// TIA Portal V17 export
// export: Created 2025-07-01T14:26:10.6416357Z, ExportSetting WithDefaults, DisplayName Totally Integrated Automation Portal, DisplayVersion V17 Update 8, DisplayName TIA Portal Openness, DisplayVersion V17 Update 8, DisplayName TIA Portal Version Control Interface, DisplayVersion V17, DisplayName SINAMICS Startdrive Advanced, DisplayVersion V17 SP2, DisplayName SINAMICS Startdrive G110M, G120, G120C, G120D, G120P, G115D, DisplayVersion V17 SP2, DisplayName SINAMICS Startdrive G130, G150, S120, S150, SINAMICS MV, S210, DisplayVersion V17 SP2, DisplayName STEP 7 Professional, DisplayVersion V17 Update 8, DisplayName SINUMERIK ONE STEP 7 Toolbox, DisplayVersion V17 Update 12, DisplayName SINUMERIK ONE PLC Basic Program Plus, DisplayVersion V17 Update 12, DisplayName SINUMERIK 840D sl STEP 7 Toolbox, DisplayVersion V17 Update 12, DisplayName STEP 7 Safety, DisplayVersion V17 Update 6, DisplayName WinCC Advanced, DisplayVersion V17 Update 8
FUNCTION "FC16016_METHOD_CALLS_U3_MEAS_STA_MEAS_R" : Void   // FC16016, LAD
{ S7_Optimized_Access := 'FALSE' }
VERSION : 0.1
// STATUS VALUES:
// 0 = IDLE
// 1 = ANALYZING
// 2 = CALIBRATING
// -1 = ERROR
// stored: AutoNumber false, IsIECCheckEnabled false, SetENOAutomatically false, UDAEnableTagReadback false
   VAR_TEMP
      AUX_WSTRING_PART_ID_MEAS_STA : WString;
      AUX_WCHARS : Array[0..63] of WChar;
      index : Int;
      AUX_ALARMS : Bool;
      STATUS_BLKMOV : Int;   // STATUS BLKMOV
      ZERO : Int;
   END_VAR
   VAR CONSTANT
      VERSIONS_MAJOR : UInt := 2;
      VERSIONS_MINOR : UInt;
      FC_NUMBER : DInt := 16016;
   END_VAR
   VAR_TEMP   // added for the SCL form of the ladder/FBD networks
      _w1 : Bool;
      _w2 : Bool;
      _w3 : Bool;
   END_VAR
BEGIN

REGION Network 1: ZERO
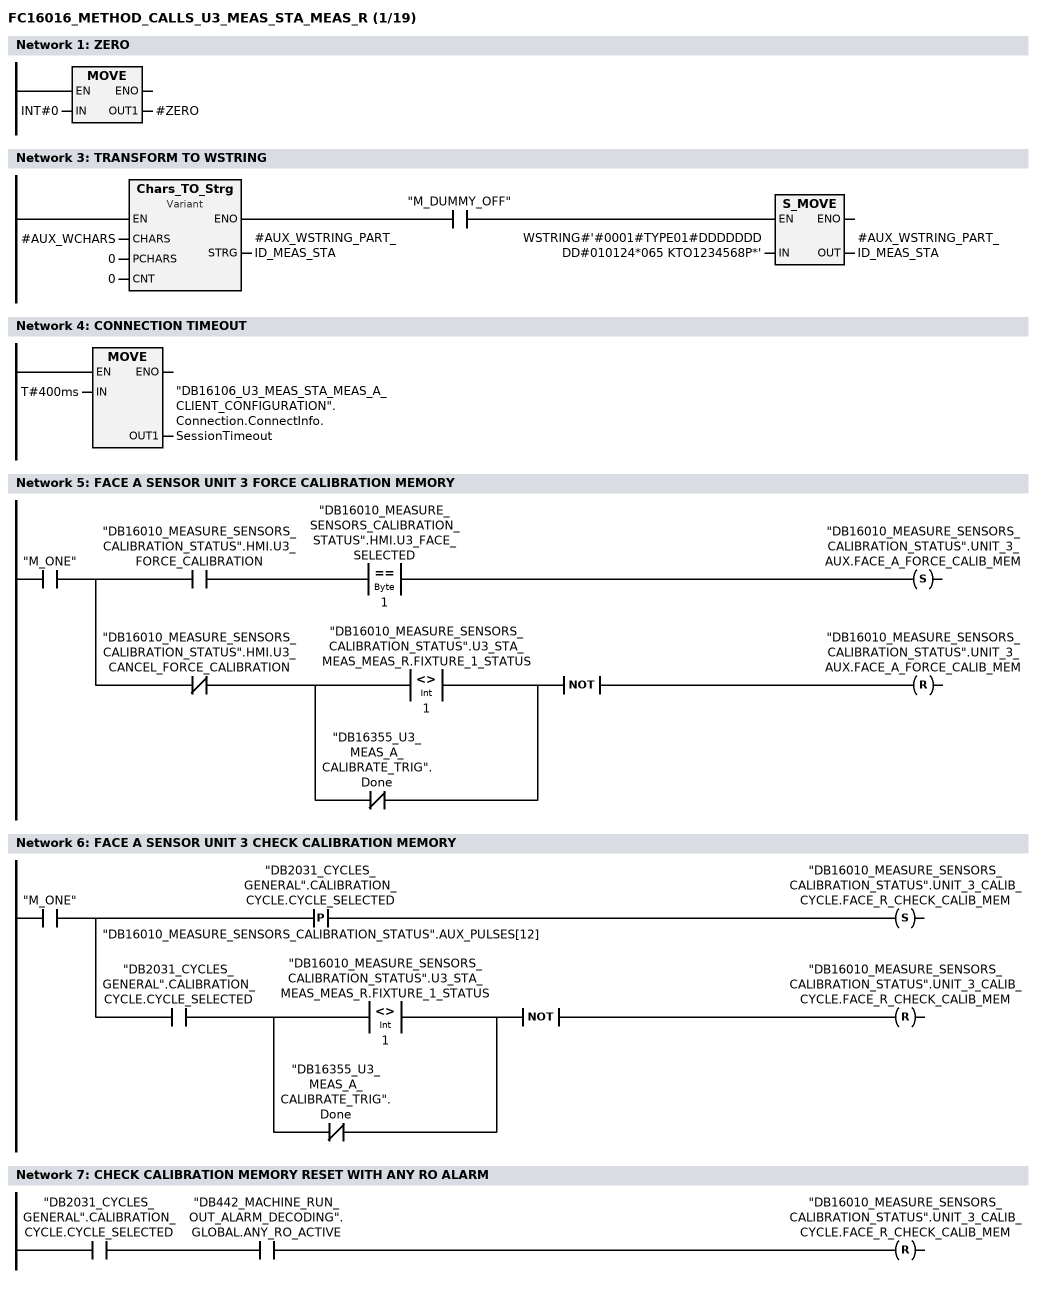
   RUNG wire#powerrail
      { S7_GenerateENO := "TRUE" } Move(in := INT#0, out1 => #ZERO)
   END_RUNG
   // the same network as SCL:
   #ZERO := INT#0;
END_REGION

REGION Network 2 (SCL): TRANSFORM TO WCHARS
   FOR #index := 0 TO 63 DO
       #AUX_WCHARS[#index] := CHAR_TO_WCHAR("DB8000_PART_STATUS".UNIT_3.FIXTURE_1.PART_A.PART_ID[#index]);
   END_FOR;
END_REGION

REGION Network 3: TRANSFORM TO WSTRING
   RUNG wire#powerrail
      { S7_Templates := "[ptr_type := Variant, str_type := WString]" } Chars_TO_Strg(Chars := #AUX_WCHARS, pChars := 0, Cnt := 0, Strg => #AUX_WSTRING_PART_ID_MEAS_STA)
      Contact( "M_DUMMY_OFF" )
      S_Move(in := WSTRING#'#0001#TYPE01#DDDDDDDDD#010124*065 KTO1234568P*', out => #AUX_WSTRING_PART_ID_MEAS_STA)
   END_RUNG
   // the same network as SCL:
   Chars_TO_Strg(Chars := #AUX_WCHARS,
                 pChars := 0,
                 Cnt := 0,
                 Strg => #AUX_WSTRING_PART_ID_MEAS_STA,
                 ENO => #_w1);
   IF #_w1 AND "M_DUMMY_OFF" THEN
       #AUX_WSTRING_PART_ID_MEAS_STA := WSTRING#'#0001#TYPE01#DDDDDDDDD#010124*065 KTO1234568P*';
   END_IF;
END_REGION

REGION Network 4: CONNECTION TIMEOUT
   RUNG wire#powerrail
      Move(in := T#400ms, out1 => "DB16106_U3_MEAS_STA_MEAS_A_CLIENT_CONFIGURATION".Connection.ConnectInfo.SessionTimeout)
   END_RUNG
   // the same network as SCL:
   "DB16106_U3_MEAS_STA_MEAS_A_CLIENT_CONFIGURATION".Connection.ConnectInfo.SessionTimeout := T#400ms;
END_REGION

REGION Network 5: FACE A SENSOR UNIT 3 FORCE CALIBRATION MEMORY
   RUNG wire#powerrail
      Contact( "M_ONE" )
      wire#w1
      Contact( "DB16010_MEASURE_SENSORS_CALIBRATION_STATUS".HMI.U3_FORCE_CALIBRATION )
      { S7_Templates := "SrcType := Byte" } EQ_Contact(in1 := "DB16010_MEASURE_SENSORS_CALIBRATION_STATUS".HMI.U3_FACE_SELECTED, in2 := 1)
      S_Coil( "DB16010_MEASURE_SENSORS_CALIBRATION_STATUS".UNIT_3_AUX.FACE_A_FORCE_CALIB_MEM )
   END_RUNG
   RUNG wire#w1
      I_Contact( "DB16010_MEASURE_SENSORS_CALIBRATION_STATUS".HMI.U3_CANCEL_FORCE_CALIBRATION )
      wire#w2
      { S7_Templates := "SrcType := Int" } NE_Contact(in1 := "DB16010_MEASURE_SENSORS_CALIBRATION_STATUS".U3_STA_MEAS_MEAS_R.FIXTURE_1_STATUS, in2 := 1)
      wire#w3
      Not()
      R_Coil( "DB16010_MEASURE_SENSORS_CALIBRATION_STATUS".UNIT_3_AUX.FACE_A_FORCE_CALIB_MEM )
   END_RUNG
   RUNG wire#w2
      I_Contact( "DB16355_U3_MEAS_A_CALIBRATE_TRIG".Done )
   END_RUNG wire#w3
   // the same network as SCL:
   IF "M_ONE" AND "DB16010_MEASURE_SENSORS_CALIBRATION_STATUS".HMI.U3_FORCE_CALIBRATION AND ("DB16010_MEASURE_SENSORS_CALIBRATION_STATUS".HMI.U3_FACE_SELECTED = 1) THEN
       "DB16010_MEASURE_SENSORS_CALIBRATION_STATUS".UNIT_3_AUX.FACE_A_FORCE_CALIB_MEM := TRUE;
   END_IF;
   IF NOT ("M_ONE" AND NOT "DB16010_MEASURE_SENSORS_CALIBRATION_STATUS".HMI.U3_CANCEL_FORCE_CALIBRATION AND (("DB16010_MEASURE_SENSORS_CALIBRATION_STATUS".U3_STA_MEAS_MEAS_R.FIXTURE_1_STATUS <> 1) OR NOT "DB16355_U3_MEAS_A_CALIBRATE_TRIG".Done)) THEN
       "DB16010_MEASURE_SENSORS_CALIBRATION_STATUS".UNIT_3_AUX.FACE_A_FORCE_CALIB_MEM := FALSE;
   END_IF;
END_REGION

REGION Network 6: FACE A SENSOR UNIT 3 CHECK CALIBRATION MEMORY
   RUNG wire#powerrail
      Contact( "M_ONE" )
      wire#w1
      P_Contact(operand := "DB2031_CYCLES_GENERAL".CALIBRATION_CYCLE.CYCLE_SELECTED, bit := "DB16010_MEASURE_SENSORS_CALIBRATION_STATUS".AUX_PULSES[12])
      S_Coil( "DB16010_MEASURE_SENSORS_CALIBRATION_STATUS".UNIT_3_CALIB_CYCLE.FACE_R_CHECK_CALIB_MEM )
   END_RUNG
   RUNG wire#w1
      Contact( "DB2031_CYCLES_GENERAL".CALIBRATION_CYCLE.CYCLE_SELECTED )
      wire#w2
      { S7_Templates := "SrcType := Int" } NE_Contact(in1 := "DB16010_MEASURE_SENSORS_CALIBRATION_STATUS".U3_STA_MEAS_MEAS_R.FIXTURE_1_STATUS, in2 := 1)
      wire#w3
      Not()
      R_Coil( "DB16010_MEASURE_SENSORS_CALIBRATION_STATUS".UNIT_3_CALIB_CYCLE.FACE_R_CHECK_CALIB_MEM )
   END_RUNG
   RUNG wire#w2
      I_Contact( "DB16355_U3_MEAS_A_CALIBRATE_TRIG".Done )
   END_RUNG wire#w3
   // the same network as SCL:
   #_w1 := "M_ONE" AND "DB2031_CYCLES_GENERAL".CALIBRATION_CYCLE.CYCLE_SELECTED AND NOT "DB16010_MEASURE_SENSORS_CALIBRATION_STATUS".AUX_PULSES[12];   // rising edge of "DB2031_CYCLES_GENERAL".CALIBRATION_CYCLE.CYCLE_SELECTED
   "DB16010_MEASURE_SENSORS_CALIBRATION_STATUS".AUX_PULSES[12] := "DB2031_CYCLES_GENERAL".CALIBRATION_CYCLE.CYCLE_SELECTED;
   IF #_w1 THEN
       "DB16010_MEASURE_SENSORS_CALIBRATION_STATUS".UNIT_3_CALIB_CYCLE.FACE_R_CHECK_CALIB_MEM := TRUE;
   END_IF;
   IF NOT ("M_ONE" AND "DB2031_CYCLES_GENERAL".CALIBRATION_CYCLE.CYCLE_SELECTED AND (("DB16010_MEASURE_SENSORS_CALIBRATION_STATUS".U3_STA_MEAS_MEAS_R.FIXTURE_1_STATUS <> 1) OR NOT "DB16355_U3_MEAS_A_CALIBRATE_TRIG".Done)) THEN
       "DB16010_MEASURE_SENSORS_CALIBRATION_STATUS".UNIT_3_CALIB_CYCLE.FACE_R_CHECK_CALIB_MEM := FALSE;
   END_IF;
END_REGION

REGION Network 7: CHECK CALIBRATION MEMORY RESET WITH ANY RO ALARM
   RUNG wire#powerrail
      Contact( "DB2031_CYCLES_GENERAL".CALIBRATION_CYCLE.CYCLE_SELECTED )
      Contact( "DB442_MACHINE_RUN_OUT_ALARM_DECODING".GLOBAL.ANY_RO_ACTIVE )
      R_Coil( "DB16010_MEASURE_SENSORS_CALIBRATION_STATUS".UNIT_3_CALIB_CYCLE.FACE_R_CHECK_CALIB_MEM )
   END_RUNG
   // the same network as SCL:
   IF "DB2031_CYCLES_GENERAL".CALIBRATION_CYCLE.CYCLE_SELECTED AND "DB442_MACHINE_RUN_OUT_ALARM_DECODING".GLOBAL.ANY_RO_ACTIVE THEN
       "DB16010_MEASURE_SENSORS_CALIBRATION_STATUS".UNIT_3_CALIB_CYCLE.FACE_R_CHECK_CALIB_MEM := FALSE;
   END_IF;
END_REGION

REGION Network 8: UNIT 3 MEASURING START CONNECTION TRIGGER
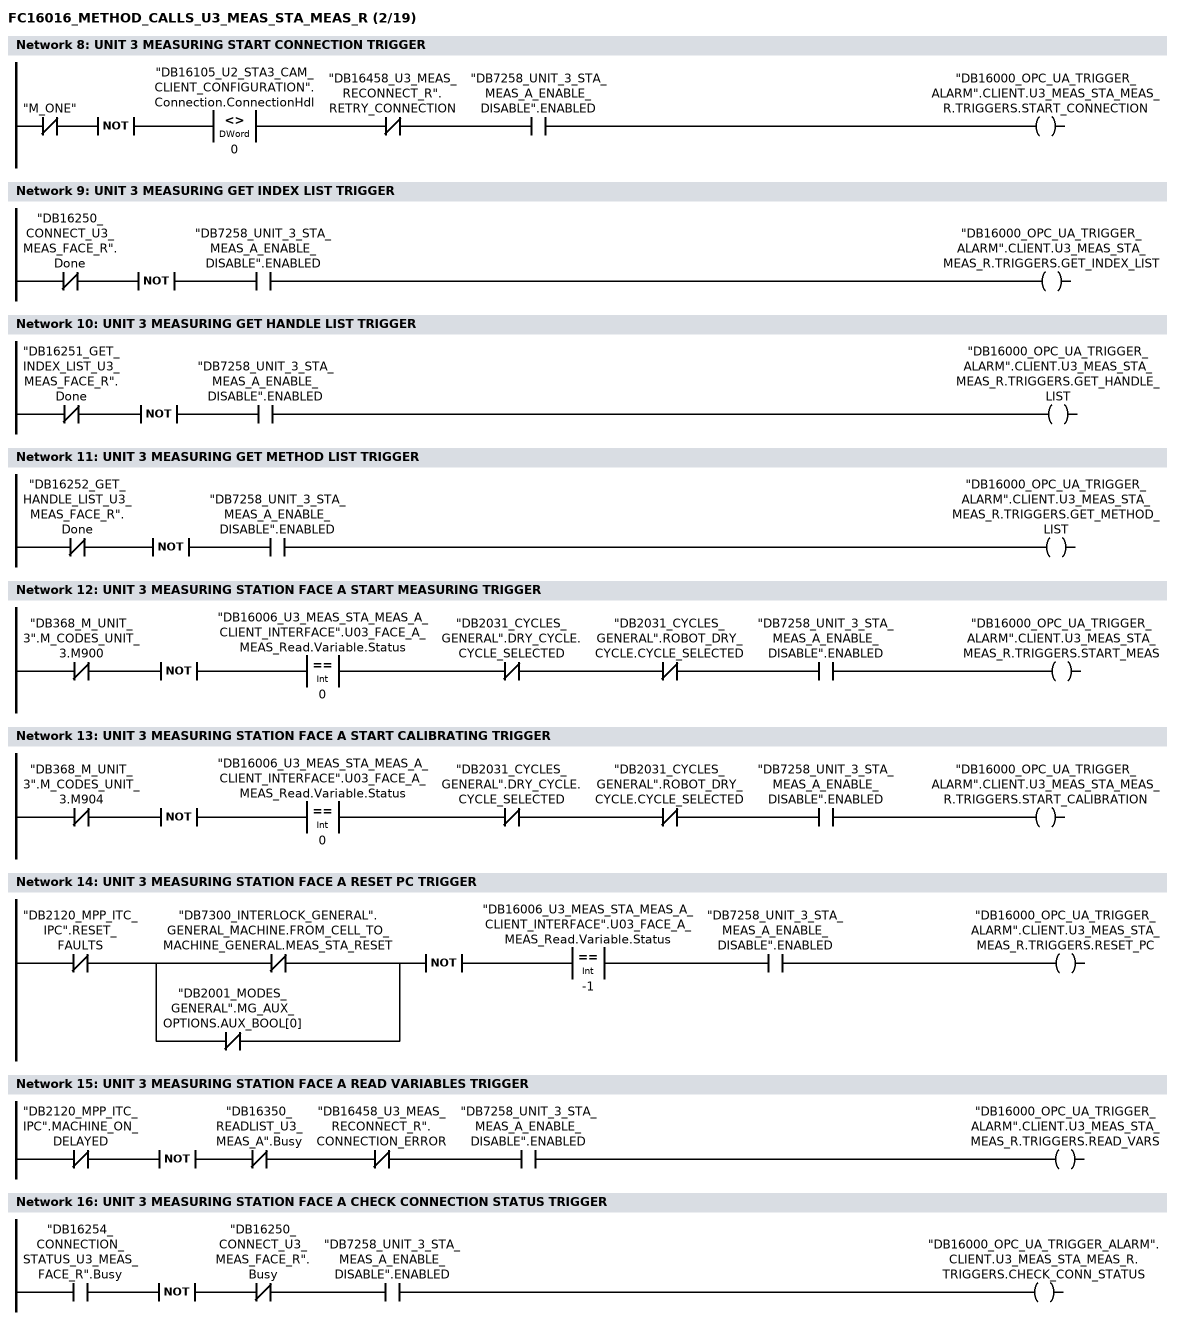
   RUNG wire#powerrail
      I_Contact( "M_ONE" )
      Not()
      { S7_Templates := "SrcType := DWord" } NE_Contact(in1 := "DB16105_U2_STA3_CAM_CLIENT_CONFIGURATION".Connection.ConnectionHdl, in2 := 0)
      I_Contact( "DB16458_U3_MEAS_RECONNECT_R".RETRY_CONNECTION )
      Contact( "DB7258_UNIT_3_STA_MEAS_A_ENABLE_DISABLE".ENABLED )
      Coil( "DB16000_OPC_UA_TRIGGER_ALARM".CLIENT.U3_MEAS_STA_MEAS_R.TRIGGERS.START_CONNECTION )
   END_RUNG
   // the same network as SCL:
   "DB16000_OPC_UA_TRIGGER_ALARM".CLIENT.U3_MEAS_STA_MEAS_R.TRIGGERS.START_CONNECTION := NOT (NOT "M_ONE") AND ("DB16105_U2_STA3_CAM_CLIENT_CONFIGURATION".Connection.ConnectionHdl <> 0) AND NOT "DB16458_U3_MEAS_RECONNECT_R".RETRY_CONNECTION AND "DB7258_UNIT_3_STA_MEAS_A_ENABLE_DISABLE".ENABLED;
END_REGION

REGION Network 9: UNIT 3 MEASURING GET INDEX LIST TRIGGER
   RUNG wire#powerrail
      I_Contact( "DB16250_CONNECT_U3_MEAS_FACE_R".Done )
      Not()
      Contact( "DB7258_UNIT_3_STA_MEAS_A_ENABLE_DISABLE".ENABLED )
      Coil( "DB16000_OPC_UA_TRIGGER_ALARM".CLIENT.U3_MEAS_STA_MEAS_R.TRIGGERS.GET_INDEX_LIST )
   END_RUNG
   // the same network as SCL:
   "DB16000_OPC_UA_TRIGGER_ALARM".CLIENT.U3_MEAS_STA_MEAS_R.TRIGGERS.GET_INDEX_LIST := NOT (NOT "DB16250_CONNECT_U3_MEAS_FACE_R".Done) AND "DB7258_UNIT_3_STA_MEAS_A_ENABLE_DISABLE".ENABLED;
END_REGION

REGION Network 10: UNIT 3 MEASURING GET HANDLE LIST TRIGGER
   RUNG wire#powerrail
      I_Contact( "DB16251_GET_INDEX_LIST_U3_MEAS_FACE_R".Done )
      Not()
      Contact( "DB7258_UNIT_3_STA_MEAS_A_ENABLE_DISABLE".ENABLED )
      Coil( "DB16000_OPC_UA_TRIGGER_ALARM".CLIENT.U3_MEAS_STA_MEAS_R.TRIGGERS.GET_HANDLE_LIST )
   END_RUNG
   // the same network as SCL:
   "DB16000_OPC_UA_TRIGGER_ALARM".CLIENT.U3_MEAS_STA_MEAS_R.TRIGGERS.GET_HANDLE_LIST := NOT (NOT "DB16251_GET_INDEX_LIST_U3_MEAS_FACE_R".Done) AND "DB7258_UNIT_3_STA_MEAS_A_ENABLE_DISABLE".ENABLED;
END_REGION

REGION Network 11: UNIT 3 MEASURING GET METHOD LIST TRIGGER
   RUNG wire#powerrail
      I_Contact( "DB16252_GET_HANDLE_LIST_U3_MEAS_FACE_R".Done )
      Not()
      Contact( "DB7258_UNIT_3_STA_MEAS_A_ENABLE_DISABLE".ENABLED )
      Coil( "DB16000_OPC_UA_TRIGGER_ALARM".CLIENT.U3_MEAS_STA_MEAS_R.TRIGGERS.GET_METHOD_LIST )
   END_RUNG
   // the same network as SCL:
   "DB16000_OPC_UA_TRIGGER_ALARM".CLIENT.U3_MEAS_STA_MEAS_R.TRIGGERS.GET_METHOD_LIST := NOT (NOT "DB16252_GET_HANDLE_LIST_U3_MEAS_FACE_R".Done) AND "DB7258_UNIT_3_STA_MEAS_A_ENABLE_DISABLE".ENABLED;
END_REGION

REGION Network 12: UNIT 3 MEASURING STATION FACE A START MEASURING TRIGGER
   RUNG wire#powerrail
      I_Contact( "DB368_M_UNIT_3".M_CODES_UNIT_3.M900 )
      Not()
      { S7_Templates := "SrcType := Int" } EQ_Contact(in1 := "DB16006_U3_MEAS_STA_MEAS_A_CLIENT_INTERFACE".U03_FACE_A_MEAS_Read.Variable.Status, in2 := 0)
      I_Contact( "DB2031_CYCLES_GENERAL".DRY_CYCLE.CYCLE_SELECTED )
      I_Contact( "DB2031_CYCLES_GENERAL".ROBOT_DRY_CYCLE.CYCLE_SELECTED )
      Contact( "DB7258_UNIT_3_STA_MEAS_A_ENABLE_DISABLE".ENABLED )
      Coil( "DB16000_OPC_UA_TRIGGER_ALARM".CLIENT.U3_MEAS_STA_MEAS_R.TRIGGERS.START_MEAS )
   END_RUNG
   // the same network as SCL:
   "DB16000_OPC_UA_TRIGGER_ALARM".CLIENT.U3_MEAS_STA_MEAS_R.TRIGGERS.START_MEAS := NOT (NOT "DB368_M_UNIT_3".M_CODES_UNIT_3.M900) AND ("DB16006_U3_MEAS_STA_MEAS_A_CLIENT_INTERFACE".U03_FACE_A_MEAS_Read.Variable.Status = 0) AND NOT "DB2031_CYCLES_GENERAL".DRY_CYCLE.CYCLE_SELECTED AND NOT "DB2031_CYCLES_GENERAL".ROBOT_DRY_CYCLE.CYCLE_SELECTED AND "DB7258_UNIT_3_STA_MEAS_A_ENABLE_DISABLE".ENABLED;
END_REGION

REGION Network 13: UNIT 3 MEASURING STATION FACE A START CALIBRATING TRIGGER
   RUNG wire#powerrail
      I_Contact( "DB368_M_UNIT_3".M_CODES_UNIT_3.M904 )
      Not()
      { S7_Templates := "SrcType := Int" } EQ_Contact(in1 := "DB16006_U3_MEAS_STA_MEAS_A_CLIENT_INTERFACE".U03_FACE_A_MEAS_Read.Variable.Status, in2 := 0)
      I_Contact( "DB2031_CYCLES_GENERAL".DRY_CYCLE.CYCLE_SELECTED )
      I_Contact( "DB2031_CYCLES_GENERAL".ROBOT_DRY_CYCLE.CYCLE_SELECTED )
      Contact( "DB7258_UNIT_3_STA_MEAS_A_ENABLE_DISABLE".ENABLED )
      Coil( "DB16000_OPC_UA_TRIGGER_ALARM".CLIENT.U3_MEAS_STA_MEAS_R.TRIGGERS.START_CALIBRATION )
   END_RUNG
   // the same network as SCL:
   "DB16000_OPC_UA_TRIGGER_ALARM".CLIENT.U3_MEAS_STA_MEAS_R.TRIGGERS.START_CALIBRATION := NOT (NOT "DB368_M_UNIT_3".M_CODES_UNIT_3.M904) AND ("DB16006_U3_MEAS_STA_MEAS_A_CLIENT_INTERFACE".U03_FACE_A_MEAS_Read.Variable.Status = 0) AND NOT "DB2031_CYCLES_GENERAL".DRY_CYCLE.CYCLE_SELECTED AND NOT "DB2031_CYCLES_GENERAL".ROBOT_DRY_CYCLE.CYCLE_SELECTED AND "DB7258_UNIT_3_STA_MEAS_A_ENABLE_DISABLE".ENABLED;
END_REGION

REGION Network 14: UNIT 3 MEASURING STATION FACE A RESET PC TRIGGER
   RUNG wire#powerrail
      I_Contact( "DB2120_MPP_ITC_IPC".RESET_FAULTS )
      wire#w1
      I_Contact( "DB7300_INTERLOCK_GENERAL".GENERAL_MACHINE.FROM_CELL_TO_MACHINE_GENERAL.MEAS_STA_RESET )
      wire#w2
      Not()
      { S7_Templates := "SrcType := Int" } EQ_Contact(in1 := "DB16006_U3_MEAS_STA_MEAS_A_CLIENT_INTERFACE".U03_FACE_A_MEAS_Read.Variable.Status, in2 := -1)
      Contact( "DB7258_UNIT_3_STA_MEAS_A_ENABLE_DISABLE".ENABLED )
      Coil( "DB16000_OPC_UA_TRIGGER_ALARM".CLIENT.U3_MEAS_STA_MEAS_R.TRIGGERS.RESET_PC )
   END_RUNG
   RUNG wire#w1
      I_Contact( "DB2001_MODES_GENERAL".MG_AUX_OPTIONS.AUX_BOOL[0] )
   END_RUNG wire#w2
   // the same network as SCL:
   "DB16000_OPC_UA_TRIGGER_ALARM".CLIENT.U3_MEAS_STA_MEAS_R.TRIGGERS.RESET_PC := NOT (NOT "DB2120_MPP_ITC_IPC".RESET_FAULTS AND (NOT "DB7300_INTERLOCK_GENERAL".GENERAL_MACHINE.FROM_CELL_TO_MACHINE_GENERAL.MEAS_STA_RESET OR NOT "DB2001_MODES_GENERAL".MG_AUX_OPTIONS.AUX_BOOL[0])) AND ("DB16006_U3_MEAS_STA_MEAS_A_CLIENT_INTERFACE".U03_FACE_A_MEAS_Read.Variable.Status = (-1)) AND "DB7258_UNIT_3_STA_MEAS_A_ENABLE_DISABLE".ENABLED;
END_REGION

REGION Network 15: UNIT 3 MEASURING STATION FACE A READ VARIABLES TRIGGER
   RUNG wire#powerrail
      I_Contact( "DB2120_MPP_ITC_IPC".MACHINE_ON_DELAYED )
      Not()
      I_Contact( "DB16350_READLIST_U3_MEAS_A".Busy )
      I_Contact( "DB16458_U3_MEAS_RECONNECT_R".CONNECTION_ERROR )
      Contact( "DB7258_UNIT_3_STA_MEAS_A_ENABLE_DISABLE".ENABLED )
      Coil( "DB16000_OPC_UA_TRIGGER_ALARM".CLIENT.U3_MEAS_STA_MEAS_R.TRIGGERS.READ_VARS )
   END_RUNG
   // the same network as SCL:
   "DB16000_OPC_UA_TRIGGER_ALARM".CLIENT.U3_MEAS_STA_MEAS_R.TRIGGERS.READ_VARS := NOT (NOT "DB2120_MPP_ITC_IPC".MACHINE_ON_DELAYED) AND NOT "DB16350_READLIST_U3_MEAS_A".Busy AND NOT "DB16458_U3_MEAS_RECONNECT_R".CONNECTION_ERROR AND "DB7258_UNIT_3_STA_MEAS_A_ENABLE_DISABLE".ENABLED;
END_REGION

REGION Network 16: UNIT 3 MEASURING STATION FACE A CHECK CONNECTION STATUS TRIGGER
   RUNG wire#powerrail
      Contact( "DB16254_CONNECTION_STATUS_U3_MEAS_FACE_R".Busy )
      Not()
      I_Contact( "DB16250_CONNECT_U3_MEAS_FACE_R".Busy )
      Contact( "DB7258_UNIT_3_STA_MEAS_A_ENABLE_DISABLE".ENABLED )
      Coil( "DB16000_OPC_UA_TRIGGER_ALARM".CLIENT.U3_MEAS_STA_MEAS_R.TRIGGERS.CHECK_CONN_STATUS )
   END_RUNG
   // the same network as SCL:
   "DB16000_OPC_UA_TRIGGER_ALARM".CLIENT.U3_MEAS_STA_MEAS_R.TRIGGERS.CHECK_CONN_STATUS := NOT "DB16254_CONNECTION_STATUS_U3_MEAS_FACE_R".Busy AND NOT "DB16250_CONNECT_U3_MEAS_FACE_R".Busy AND "DB7258_UNIT_3_STA_MEAS_A_ENABLE_DISABLE".ENABLED;
END_REGION

REGION Network 17: UNIT 3 MEASURING STATION FACE A RELEASE HANDLE LIST TRIGGER
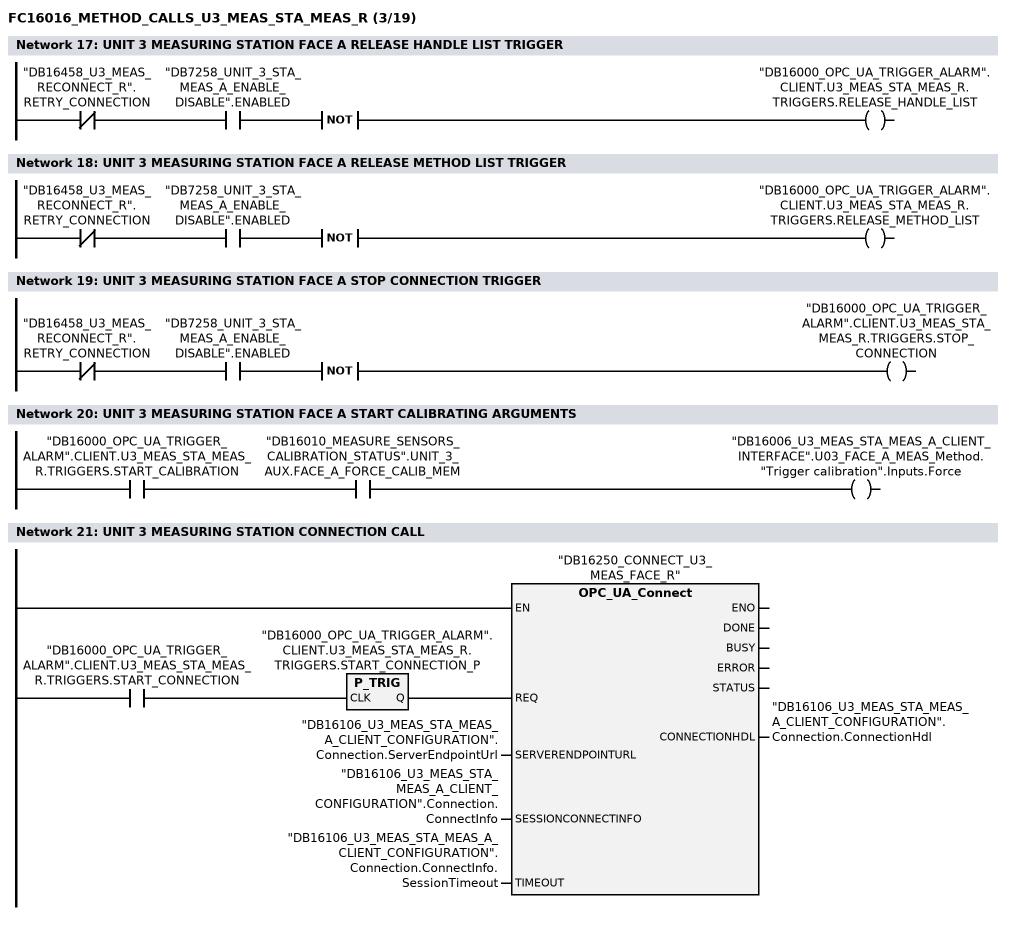
   RUNG wire#powerrail
      I_Contact( "DB16458_U3_MEAS_RECONNECT_R".RETRY_CONNECTION )
      Contact( "DB7258_UNIT_3_STA_MEAS_A_ENABLE_DISABLE".ENABLED )
      Not()
      Coil( "DB16000_OPC_UA_TRIGGER_ALARM".CLIENT.U3_MEAS_STA_MEAS_R.TRIGGERS.RELEASE_HANDLE_LIST )
   END_RUNG
   // the same network as SCL:
   "DB16000_OPC_UA_TRIGGER_ALARM".CLIENT.U3_MEAS_STA_MEAS_R.TRIGGERS.RELEASE_HANDLE_LIST := NOT (NOT "DB16458_U3_MEAS_RECONNECT_R".RETRY_CONNECTION AND "DB7258_UNIT_3_STA_MEAS_A_ENABLE_DISABLE".ENABLED);
END_REGION

REGION Network 18: UNIT 3 MEASURING STATION FACE A RELEASE METHOD LIST TRIGGER
   RUNG wire#powerrail
      I_Contact( "DB16458_U3_MEAS_RECONNECT_R".RETRY_CONNECTION )
      Contact( "DB7258_UNIT_3_STA_MEAS_A_ENABLE_DISABLE".ENABLED )
      Not()
      Coil( "DB16000_OPC_UA_TRIGGER_ALARM".CLIENT.U3_MEAS_STA_MEAS_R.TRIGGERS.RELEASE_METHOD_LIST )
   END_RUNG
   // the same network as SCL:
   "DB16000_OPC_UA_TRIGGER_ALARM".CLIENT.U3_MEAS_STA_MEAS_R.TRIGGERS.RELEASE_METHOD_LIST := NOT (NOT "DB16458_U3_MEAS_RECONNECT_R".RETRY_CONNECTION AND "DB7258_UNIT_3_STA_MEAS_A_ENABLE_DISABLE".ENABLED);
END_REGION

REGION Network 19: UNIT 3 MEASURING STATION FACE A STOP CONNECTION TRIGGER
   RUNG wire#powerrail
      I_Contact( "DB16458_U3_MEAS_RECONNECT_R".RETRY_CONNECTION )
      Contact( "DB7258_UNIT_3_STA_MEAS_A_ENABLE_DISABLE".ENABLED )
      Not()
      Coil( "DB16000_OPC_UA_TRIGGER_ALARM".CLIENT.U3_MEAS_STA_MEAS_R.TRIGGERS.STOP_CONNECTION )
   END_RUNG
   // the same network as SCL:
   "DB16000_OPC_UA_TRIGGER_ALARM".CLIENT.U3_MEAS_STA_MEAS_R.TRIGGERS.STOP_CONNECTION := NOT (NOT "DB16458_U3_MEAS_RECONNECT_R".RETRY_CONNECTION AND "DB7258_UNIT_3_STA_MEAS_A_ENABLE_DISABLE".ENABLED);
END_REGION

REGION Network 20: UNIT 3 MEASURING STATION FACE A START CALIBRATING ARGUMENTS
   RUNG wire#powerrail
      Contact( "DB16000_OPC_UA_TRIGGER_ALARM".CLIENT.U3_MEAS_STA_MEAS_R.TRIGGERS.START_CALIBRATION )
      Contact( "DB16010_MEASURE_SENSORS_CALIBRATION_STATUS".UNIT_3_AUX.FACE_A_FORCE_CALIB_MEM )
      Coil( "DB16006_U3_MEAS_STA_MEAS_A_CLIENT_INTERFACE".U03_FACE_A_MEAS_Method."Trigger calibration".Inputs.Force )
   END_RUNG
   // the same network as SCL:
   "DB16006_U3_MEAS_STA_MEAS_A_CLIENT_INTERFACE".U03_FACE_A_MEAS_Method."Trigger calibration".Inputs.Force := "DB16000_OPC_UA_TRIGGER_ALARM".CLIENT.U3_MEAS_STA_MEAS_R.TRIGGERS.START_CALIBRATION AND "DB16010_MEASURE_SENSORS_CALIBRATION_STATUS".UNIT_3_AUX.FACE_A_FORCE_CALIB_MEM;
END_REGION

REGION Network 21: UNIT 3 MEASURING STATION CONNECTION CALL
   RUNG wire#powerrail
      "DB16250_CONNECT_U3_MEAS_FACE_R".OPC_UA_Connect(REQ := wire#w1, ServerEndpointUrl := "DB16106_U3_MEAS_STA_MEAS_A_CLIENT_CONFIGURATION".Connection.ServerEndpointUrl, SessionConnectInfo := "DB16106_U3_MEAS_STA_MEAS_A_CLIENT_CONFIGURATION".Connection.ConnectInfo, Timeout := "DB16106_U3_MEAS_STA_MEAS_A_CLIENT_CONFIGURATION".Connection.ConnectInfo.SessionTimeout, Done =>, Busy =>, Error =>, Status =>, ConnectionHdl => "DB16106_U3_MEAS_STA_MEAS_A_CLIENT_CONFIGURATION".Connection.ConnectionHdl)
   END_RUNG
   RUNG wire#powerrail
      Contact( "DB16000_OPC_UA_TRIGGER_ALARM".CLIENT.U3_MEAS_STA_MEAS_R.TRIGGERS.START_CONNECTION )
      P_Trig( "DB16000_OPC_UA_TRIGGER_ALARM".CLIENT.U3_MEAS_STA_MEAS_R.TRIGGERS.START_CONNECTION_P )
   END_RUNG wire#w1
   // the same network as SCL:
   #_w1 := "DB16000_OPC_UA_TRIGGER_ALARM".CLIENT.U3_MEAS_STA_MEAS_R.TRIGGERS.START_CONNECTION AND NOT "DB16000_OPC_UA_TRIGGER_ALARM".CLIENT.U3_MEAS_STA_MEAS_R.TRIGGERS.START_CONNECTION_P;   // rising edge
   "DB16000_OPC_UA_TRIGGER_ALARM".CLIENT.U3_MEAS_STA_MEAS_R.TRIGGERS.START_CONNECTION_P := "DB16000_OPC_UA_TRIGGER_ALARM".CLIENT.U3_MEAS_STA_MEAS_R.TRIGGERS.START_CONNECTION;
   "DB16250_CONNECT_U3_MEAS_FACE_R"(REQ := #_w1,   // OPC_UA_Connect
                           ServerEndpointUrl := "DB16106_U3_MEAS_STA_MEAS_A_CLIENT_CONFIGURATION".Connection.ServerEndpointUrl,
                           SessionConnectInfo := "DB16106_U3_MEAS_STA_MEAS_A_CLIENT_CONFIGURATION".Connection.ConnectInfo,
                           Timeout := "DB16106_U3_MEAS_STA_MEAS_A_CLIENT_CONFIGURATION".Connection.ConnectInfo.SessionTimeout,
                           ConnectionHdl => "DB16106_U3_MEAS_STA_MEAS_A_CLIENT_CONFIGURATION".Connection.ConnectionHdl);
END_REGION

REGION Network 22: UNIT 3 MEASURING STATION FACE A GET INDEX LIST CALL
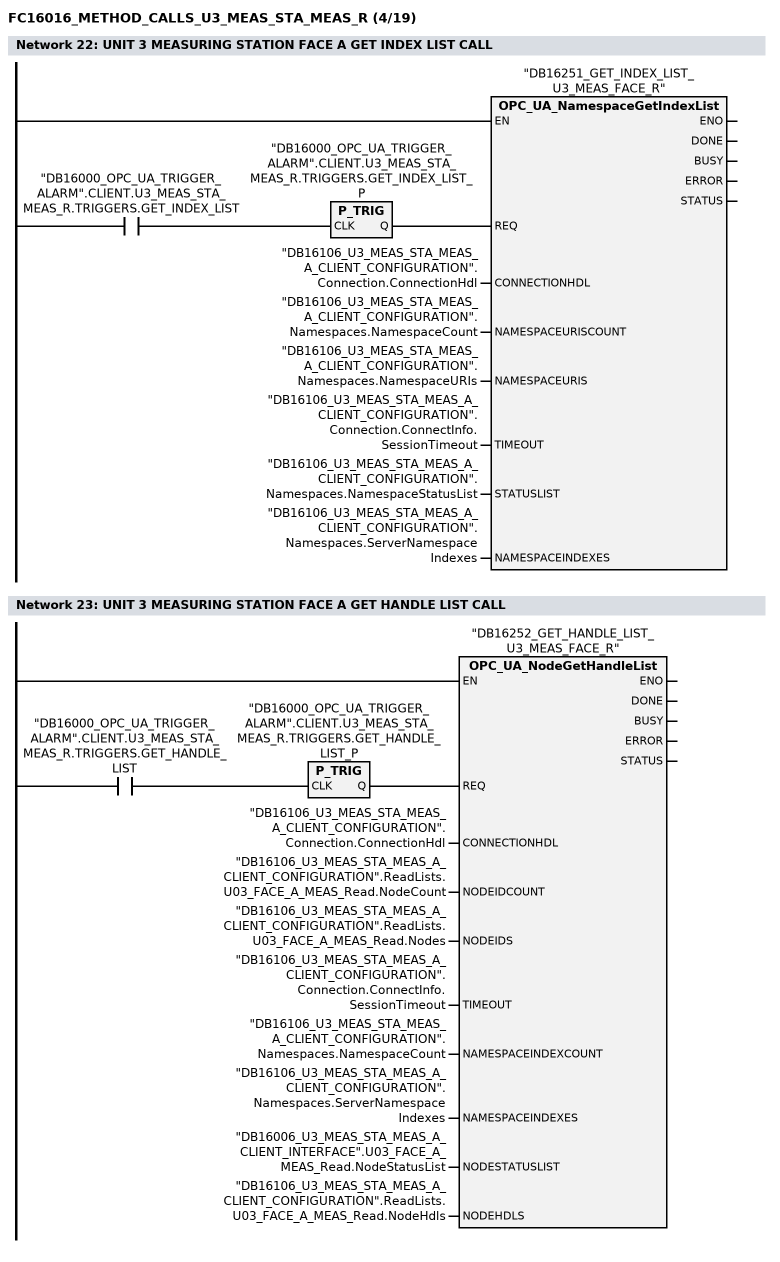
   RUNG wire#powerrail
      "DB16251_GET_INDEX_LIST_U3_MEAS_FACE_R".OPC_UA_NamespaceGetIndexList(REQ := wire#w1, ConnectionHdl := "DB16106_U3_MEAS_STA_MEAS_A_CLIENT_CONFIGURATION".Connection.ConnectionHdl, NamespaceUrisCount := "DB16106_U3_MEAS_STA_MEAS_A_CLIENT_CONFIGURATION".Namespaces.NamespaceCount, NamespaceUris := "DB16106_U3_MEAS_STA_MEAS_A_CLIENT_CONFIGURATION".Namespaces.NamespaceURIs, Timeout := "DB16106_U3_MEAS_STA_MEAS_A_CLIENT_CONFIGURATION".Connection.ConnectInfo.SessionTimeout, StatusList := "DB16106_U3_MEAS_STA_MEAS_A_CLIENT_CONFIGURATION".Namespaces.NamespaceStatusList, NamespaceIndexes := "DB16106_U3_MEAS_STA_MEAS_A_CLIENT_CONFIGURATION".Namespaces.ServerNamespaceIndexes, Done =>, Busy =>, Error =>, Status =>)
   END_RUNG
   RUNG wire#powerrail
      Contact( "DB16000_OPC_UA_TRIGGER_ALARM".CLIENT.U3_MEAS_STA_MEAS_R.TRIGGERS.GET_INDEX_LIST )
      P_Trig( "DB16000_OPC_UA_TRIGGER_ALARM".CLIENT.U3_MEAS_STA_MEAS_R.TRIGGERS.GET_INDEX_LIST_P )
   END_RUNG wire#w1
   // the same network as SCL:
   #_w1 := "DB16000_OPC_UA_TRIGGER_ALARM".CLIENT.U3_MEAS_STA_MEAS_R.TRIGGERS.GET_INDEX_LIST AND NOT "DB16000_OPC_UA_TRIGGER_ALARM".CLIENT.U3_MEAS_STA_MEAS_R.TRIGGERS.GET_INDEX_LIST_P;   // rising edge
   "DB16000_OPC_UA_TRIGGER_ALARM".CLIENT.U3_MEAS_STA_MEAS_R.TRIGGERS.GET_INDEX_LIST_P := "DB16000_OPC_UA_TRIGGER_ALARM".CLIENT.U3_MEAS_STA_MEAS_R.TRIGGERS.GET_INDEX_LIST;
   "DB16251_GET_INDEX_LIST_U3_MEAS_FACE_R"(REQ := #_w1,   // OPC_UA_NamespaceGetIndexList
                           ConnectionHdl := "DB16106_U3_MEAS_STA_MEAS_A_CLIENT_CONFIGURATION".Connection.ConnectionHdl,
                           NamespaceUrisCount := "DB16106_U3_MEAS_STA_MEAS_A_CLIENT_CONFIGURATION".Namespaces.NamespaceCount,
                           NamespaceUris := "DB16106_U3_MEAS_STA_MEAS_A_CLIENT_CONFIGURATION".Namespaces.NamespaceURIs,
                           Timeout := "DB16106_U3_MEAS_STA_MEAS_A_CLIENT_CONFIGURATION".Connection.ConnectInfo.SessionTimeout,
                           StatusList := "DB16106_U3_MEAS_STA_MEAS_A_CLIENT_CONFIGURATION".Namespaces.NamespaceStatusList,
                           NamespaceIndexes := "DB16106_U3_MEAS_STA_MEAS_A_CLIENT_CONFIGURATION".Namespaces.ServerNamespaceIndexes);
END_REGION

REGION Network 23: UNIT 3 MEASURING STATION FACE A GET HANDLE LIST CALL
   RUNG wire#powerrail
      "DB16252_GET_HANDLE_LIST_U3_MEAS_FACE_R".OPC_UA_NodeGetHandleList(REQ := wire#w1, ConnectionHdl := "DB16106_U3_MEAS_STA_MEAS_A_CLIENT_CONFIGURATION".Connection.ConnectionHdl, NodeIDCount := "DB16106_U3_MEAS_STA_MEAS_A_CLIENT_CONFIGURATION".ReadLists.U03_FACE_A_MEAS_Read.NodeCount, NodeIDs := "DB16106_U3_MEAS_STA_MEAS_A_CLIENT_CONFIGURATION".ReadLists.U03_FACE_A_MEAS_Read.Nodes, Timeout := "DB16106_U3_MEAS_STA_MEAS_A_CLIENT_CONFIGURATION".Connection.ConnectInfo.SessionTimeout, NamespaceIndexCount := "DB16106_U3_MEAS_STA_MEAS_A_CLIENT_CONFIGURATION".Namespaces.NamespaceCount, NamespaceIndexes := "DB16106_U3_MEAS_STA_MEAS_A_CLIENT_CONFIGURATION".Namespaces.ServerNamespaceIndexes, NodeStatusList := "DB16006_U3_MEAS_STA_MEAS_A_CLIENT_INTERFACE".U03_FACE_A_MEAS_Read.NodeStatusList, NodeHdls := "DB16106_U3_MEAS_STA_MEAS_A_CLIENT_CONFIGURATION".ReadLists.U03_FACE_A_MEAS_Read.NodeHdls, Done =>, Busy =>, Error =>, Status =>)
   END_RUNG
   RUNG wire#powerrail
      Contact( "DB16000_OPC_UA_TRIGGER_ALARM".CLIENT.U3_MEAS_STA_MEAS_R.TRIGGERS.GET_HANDLE_LIST )
      P_Trig( "DB16000_OPC_UA_TRIGGER_ALARM".CLIENT.U3_MEAS_STA_MEAS_R.TRIGGERS.GET_HANDLE_LIST_P )
   END_RUNG wire#w1
   // the same network as SCL:
   #_w1 := "DB16000_OPC_UA_TRIGGER_ALARM".CLIENT.U3_MEAS_STA_MEAS_R.TRIGGERS.GET_HANDLE_LIST AND NOT "DB16000_OPC_UA_TRIGGER_ALARM".CLIENT.U3_MEAS_STA_MEAS_R.TRIGGERS.GET_HANDLE_LIST_P;   // rising edge
   "DB16000_OPC_UA_TRIGGER_ALARM".CLIENT.U3_MEAS_STA_MEAS_R.TRIGGERS.GET_HANDLE_LIST_P := "DB16000_OPC_UA_TRIGGER_ALARM".CLIENT.U3_MEAS_STA_MEAS_R.TRIGGERS.GET_HANDLE_LIST;
   "DB16252_GET_HANDLE_LIST_U3_MEAS_FACE_R"(REQ := #_w1,   // OPC_UA_NodeGetHandleList
                           ConnectionHdl := "DB16106_U3_MEAS_STA_MEAS_A_CLIENT_CONFIGURATION".Connection.ConnectionHdl,
                           NodeIDCount := "DB16106_U3_MEAS_STA_MEAS_A_CLIENT_CONFIGURATION".ReadLists.U03_FACE_A_MEAS_Read.NodeCount,
                           NodeIDs := "DB16106_U3_MEAS_STA_MEAS_A_CLIENT_CONFIGURATION".ReadLists.U03_FACE_A_MEAS_Read.Nodes,
                           Timeout := "DB16106_U3_MEAS_STA_MEAS_A_CLIENT_CONFIGURATION".Connection.ConnectInfo.SessionTimeout,
                           NamespaceIndexCount := "DB16106_U3_MEAS_STA_MEAS_A_CLIENT_CONFIGURATION".Namespaces.NamespaceCount,
                           NamespaceIndexes := "DB16106_U3_MEAS_STA_MEAS_A_CLIENT_CONFIGURATION".Namespaces.ServerNamespaceIndexes,
                           NodeStatusList := "DB16006_U3_MEAS_STA_MEAS_A_CLIENT_INTERFACE".U03_FACE_A_MEAS_Read.NodeStatusList,
                           NodeHdls := "DB16106_U3_MEAS_STA_MEAS_A_CLIENT_CONFIGURATION".ReadLists.U03_FACE_A_MEAS_Read.NodeHdls);
END_REGION

REGION Network 24: UNIT 3 MEASURING STATION FACE A GET METHOD LIST CALL
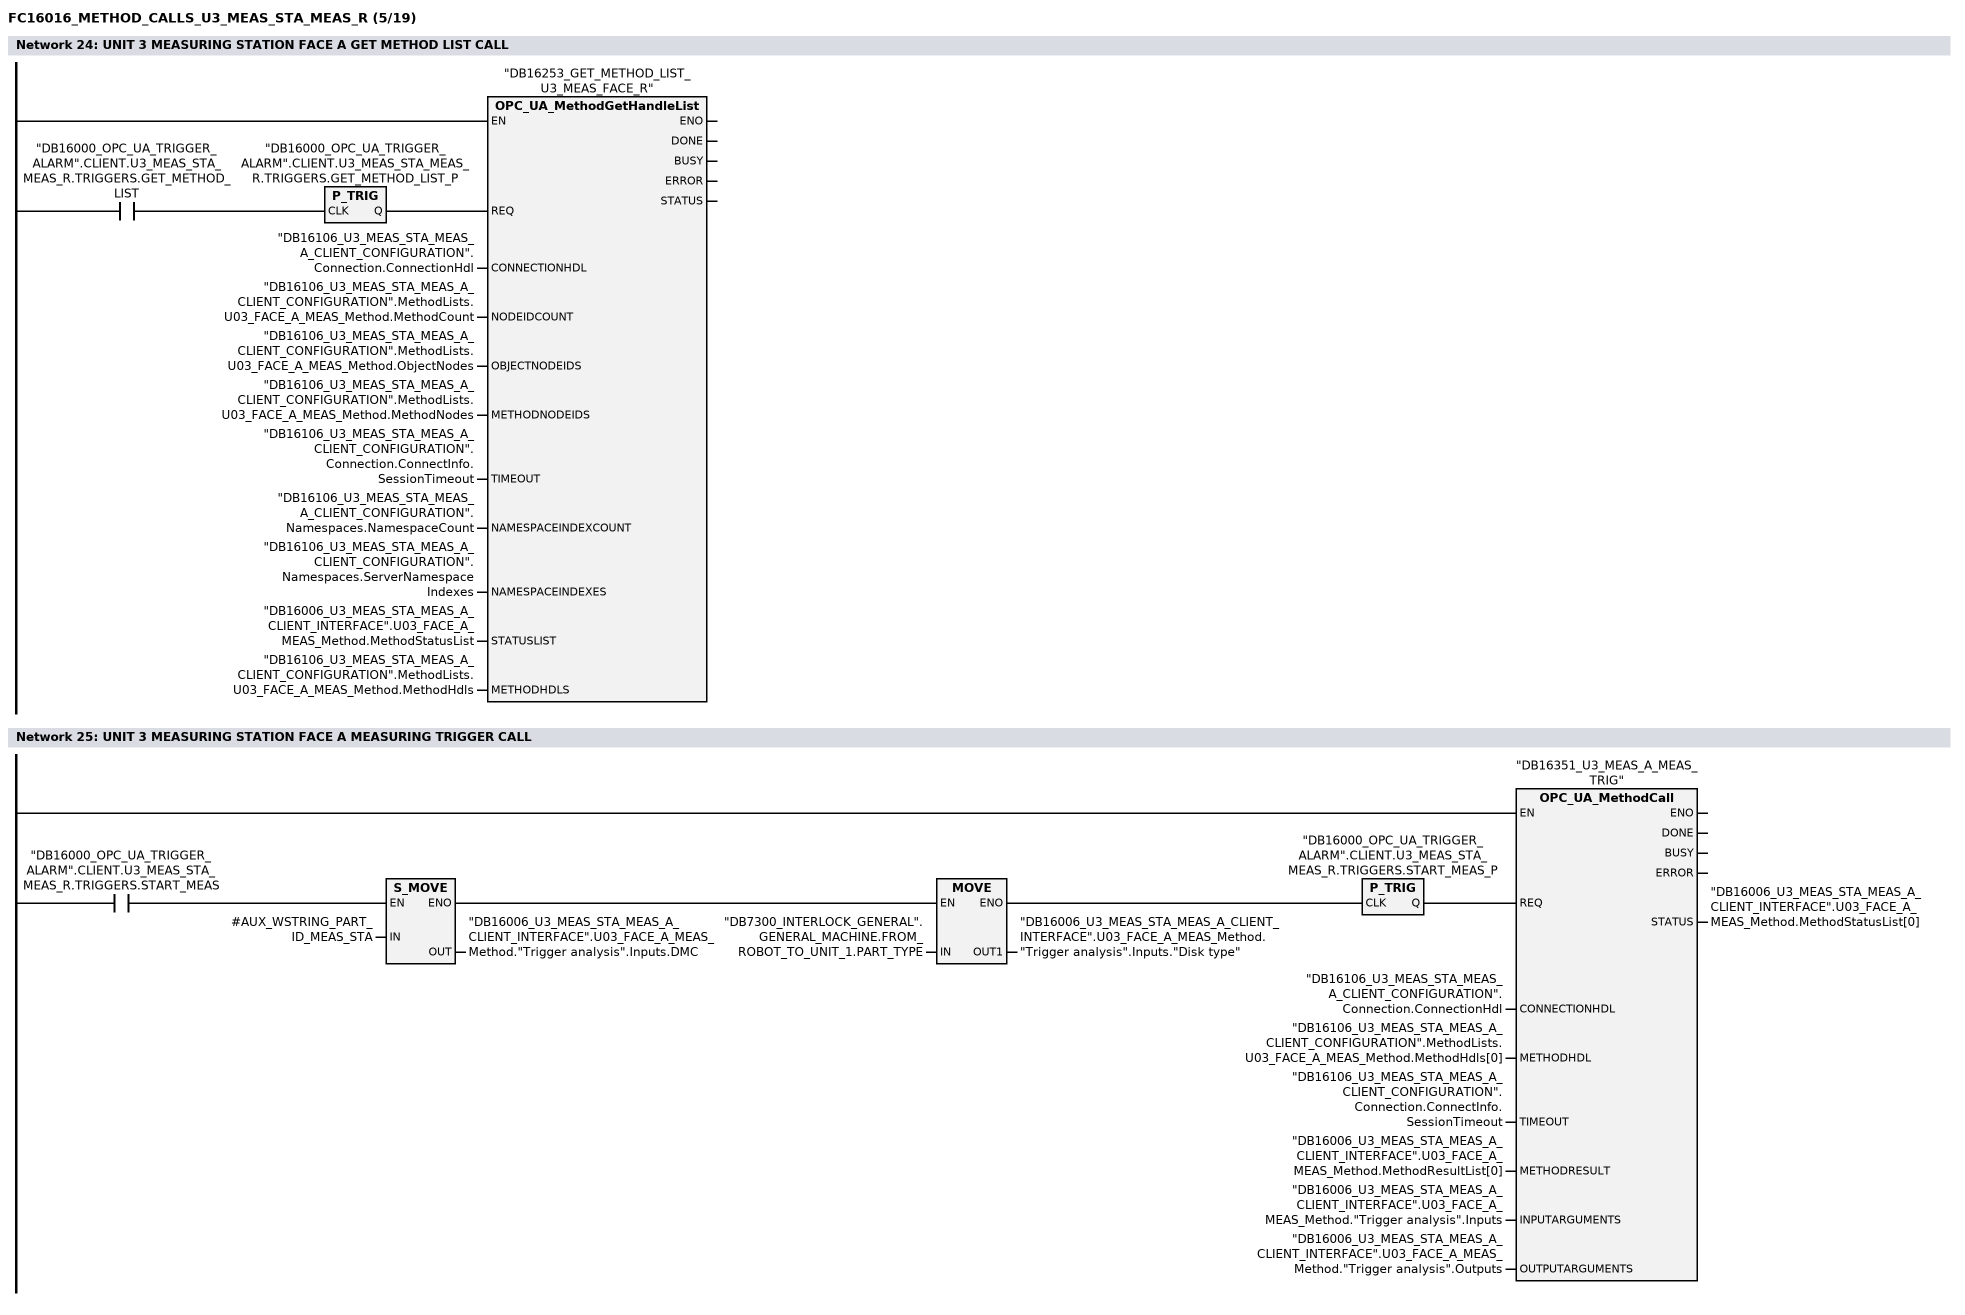
   RUNG wire#powerrail
      "DB16253_GET_METHOD_LIST_U3_MEAS_FACE_R".OPC_UA_MethodGetHandleList(REQ := wire#w1, ConnectionHdl := "DB16106_U3_MEAS_STA_MEAS_A_CLIENT_CONFIGURATION".Connection.ConnectionHdl, NodeIDCount := "DB16106_U3_MEAS_STA_MEAS_A_CLIENT_CONFIGURATION".MethodLists.U03_FACE_A_MEAS_Method.MethodCount, ObjectNodeIDs := "DB16106_U3_MEAS_STA_MEAS_A_CLIENT_CONFIGURATION".MethodLists.U03_FACE_A_MEAS_Method.ObjectNodes, MethodNodeIDs := "DB16106_U3_MEAS_STA_MEAS_A_CLIENT_CONFIGURATION".MethodLists.U03_FACE_A_MEAS_Method.MethodNodes, Timeout := "DB16106_U3_MEAS_STA_MEAS_A_CLIENT_CONFIGURATION".Connection.ConnectInfo.SessionTimeout, NamespaceIndexCount := "DB16106_U3_MEAS_STA_MEAS_A_CLIENT_CONFIGURATION".Namespaces.NamespaceCount, NamespaceIndexes := "DB16106_U3_MEAS_STA_MEAS_A_CLIENT_CONFIGURATION".Namespaces.ServerNamespaceIndexes, StatusList := "DB16006_U3_MEAS_STA_MEAS_A_CLIENT_INTERFACE".U03_FACE_A_MEAS_Method.MethodStatusList, MethodHdls := "DB16106_U3_MEAS_STA_MEAS_A_CLIENT_CONFIGURATION".MethodLists.U03_FACE_A_MEAS_Method.MethodHdls, Done =>, Busy =>, Error =>, Status =>)
   END_RUNG
   RUNG wire#powerrail
      Contact( "DB16000_OPC_UA_TRIGGER_ALARM".CLIENT.U3_MEAS_STA_MEAS_R.TRIGGERS.GET_METHOD_LIST )
      P_Trig( "DB16000_OPC_UA_TRIGGER_ALARM".CLIENT.U3_MEAS_STA_MEAS_R.TRIGGERS.GET_METHOD_LIST_P )
   END_RUNG wire#w1
   // the same network as SCL:
   #_w1 := "DB16000_OPC_UA_TRIGGER_ALARM".CLIENT.U3_MEAS_STA_MEAS_R.TRIGGERS.GET_METHOD_LIST AND NOT "DB16000_OPC_UA_TRIGGER_ALARM".CLIENT.U3_MEAS_STA_MEAS_R.TRIGGERS.GET_METHOD_LIST_P;   // rising edge
   "DB16000_OPC_UA_TRIGGER_ALARM".CLIENT.U3_MEAS_STA_MEAS_R.TRIGGERS.GET_METHOD_LIST_P := "DB16000_OPC_UA_TRIGGER_ALARM".CLIENT.U3_MEAS_STA_MEAS_R.TRIGGERS.GET_METHOD_LIST;
   "DB16253_GET_METHOD_LIST_U3_MEAS_FACE_R"(REQ := #_w1,   // OPC_UA_MethodGetHandleList
                           ConnectionHdl := "DB16106_U3_MEAS_STA_MEAS_A_CLIENT_CONFIGURATION".Connection.ConnectionHdl,
                           NodeIDCount := "DB16106_U3_MEAS_STA_MEAS_A_CLIENT_CONFIGURATION".MethodLists.U03_FACE_A_MEAS_Method.MethodCount,
                           ObjectNodeIDs := "DB16106_U3_MEAS_STA_MEAS_A_CLIENT_CONFIGURATION".MethodLists.U03_FACE_A_MEAS_Method.ObjectNodes,
                           MethodNodeIDs := "DB16106_U3_MEAS_STA_MEAS_A_CLIENT_CONFIGURATION".MethodLists.U03_FACE_A_MEAS_Method.MethodNodes,
                           Timeout := "DB16106_U3_MEAS_STA_MEAS_A_CLIENT_CONFIGURATION".Connection.ConnectInfo.SessionTimeout,
                           NamespaceIndexCount := "DB16106_U3_MEAS_STA_MEAS_A_CLIENT_CONFIGURATION".Namespaces.NamespaceCount,
                           NamespaceIndexes := "DB16106_U3_MEAS_STA_MEAS_A_CLIENT_CONFIGURATION".Namespaces.ServerNamespaceIndexes,
                           StatusList := "DB16006_U3_MEAS_STA_MEAS_A_CLIENT_INTERFACE".U03_FACE_A_MEAS_Method.MethodStatusList,
                           MethodHdls := "DB16106_U3_MEAS_STA_MEAS_A_CLIENT_CONFIGURATION".MethodLists.U03_FACE_A_MEAS_Method.MethodHdls);
END_REGION

REGION Network 25: UNIT 3 MEASURING STATION FACE A MEASURING TRIGGER CALL
   RUNG wire#powerrail
      "DB16351_U3_MEAS_A_MEAS_TRIG".OPC_UA_MethodCall(REQ := wire#w1, ConnectionHdl := "DB16106_U3_MEAS_STA_MEAS_A_CLIENT_CONFIGURATION".Connection.ConnectionHdl, MethodHdl := "DB16106_U3_MEAS_STA_MEAS_A_CLIENT_CONFIGURATION".MethodLists.U03_FACE_A_MEAS_Method.MethodHdls[0], Timeout := "DB16106_U3_MEAS_STA_MEAS_A_CLIENT_CONFIGURATION".Connection.ConnectInfo.SessionTimeout, MethodResult := "DB16006_U3_MEAS_STA_MEAS_A_CLIENT_INTERFACE".U03_FACE_A_MEAS_Method.MethodResultList[0], InputArguments := "DB16006_U3_MEAS_STA_MEAS_A_CLIENT_INTERFACE".U03_FACE_A_MEAS_Method."Trigger analysis".Inputs, OutputArguments := "DB16006_U3_MEAS_STA_MEAS_A_CLIENT_INTERFACE".U03_FACE_A_MEAS_Method."Trigger analysis".Outputs, Done =>, Busy =>, Error =>, Status => "DB16006_U3_MEAS_STA_MEAS_A_CLIENT_INTERFACE".U03_FACE_A_MEAS_Method.MethodStatusList[0])
   END_RUNG
   RUNG wire#powerrail
      Contact( "DB16000_OPC_UA_TRIGGER_ALARM".CLIENT.U3_MEAS_STA_MEAS_R.TRIGGERS.START_MEAS )
      S_Move(in := #AUX_WSTRING_PART_ID_MEAS_STA, out => "DB16006_U3_MEAS_STA_MEAS_A_CLIENT_INTERFACE".U03_FACE_A_MEAS_Method."Trigger analysis".Inputs.DMC)
      Move(in := "DB7300_INTERLOCK_GENERAL".GENERAL_MACHINE.FROM_ROBOT_TO_UNIT_1.PART_TYPE, out1 => "DB16006_U3_MEAS_STA_MEAS_A_CLIENT_INTERFACE".U03_FACE_A_MEAS_Method."Trigger analysis".Inputs."Disk type")
      P_Trig( "DB16000_OPC_UA_TRIGGER_ALARM".CLIENT.U3_MEAS_STA_MEAS_R.TRIGGERS.START_MEAS_P )
   END_RUNG wire#w1
   // the same network as SCL:
   IF "DB16000_OPC_UA_TRIGGER_ALARM".CLIENT.U3_MEAS_STA_MEAS_R.TRIGGERS.START_MEAS THEN
       "DB16006_U3_MEAS_STA_MEAS_A_CLIENT_INTERFACE".U03_FACE_A_MEAS_Method."Trigger analysis".Inputs.DMC := #AUX_WSTRING_PART_ID_MEAS_STA;
       "DB16006_U3_MEAS_STA_MEAS_A_CLIENT_INTERFACE".U03_FACE_A_MEAS_Method."Trigger analysis".Inputs."Disk type" := "DB7300_INTERLOCK_GENERAL".GENERAL_MACHINE.FROM_ROBOT_TO_UNIT_1.PART_TYPE;
   END_IF;
   #_w1 := "DB16000_OPC_UA_TRIGGER_ALARM".CLIENT.U3_MEAS_STA_MEAS_R.TRIGGERS.START_MEAS AND NOT "DB16000_OPC_UA_TRIGGER_ALARM".CLIENT.U3_MEAS_STA_MEAS_R.TRIGGERS.START_MEAS_P;   // rising edge
   "DB16000_OPC_UA_TRIGGER_ALARM".CLIENT.U3_MEAS_STA_MEAS_R.TRIGGERS.START_MEAS_P := "DB16000_OPC_UA_TRIGGER_ALARM".CLIENT.U3_MEAS_STA_MEAS_R.TRIGGERS.START_MEAS;
   "DB16351_U3_MEAS_A_MEAS_TRIG"(REQ := #_w1,   // OPC_UA_MethodCall
                           ConnectionHdl := "DB16106_U3_MEAS_STA_MEAS_A_CLIENT_CONFIGURATION".Connection.ConnectionHdl,
                           MethodHdl := "DB16106_U3_MEAS_STA_MEAS_A_CLIENT_CONFIGURATION".MethodLists.U03_FACE_A_MEAS_Method.MethodHdls[0],
                           Timeout := "DB16106_U3_MEAS_STA_MEAS_A_CLIENT_CONFIGURATION".Connection.ConnectInfo.SessionTimeout,
                           MethodResult := "DB16006_U3_MEAS_STA_MEAS_A_CLIENT_INTERFACE".U03_FACE_A_MEAS_Method.MethodResultList[0],
                           InputArguments := "DB16006_U3_MEAS_STA_MEAS_A_CLIENT_INTERFACE".U03_FACE_A_MEAS_Method."Trigger analysis".Inputs,
                           OutputArguments := "DB16006_U3_MEAS_STA_MEAS_A_CLIENT_INTERFACE".U03_FACE_A_MEAS_Method."Trigger analysis".Outputs,
                           Status => "DB16006_U3_MEAS_STA_MEAS_A_CLIENT_INTERFACE".U03_FACE_A_MEAS_Method.MethodStatusList[0]);
END_REGION

REGION Network 26: UNIT 3 MEASURING STATION FACE A CALIBRATING TRIGGER CALL
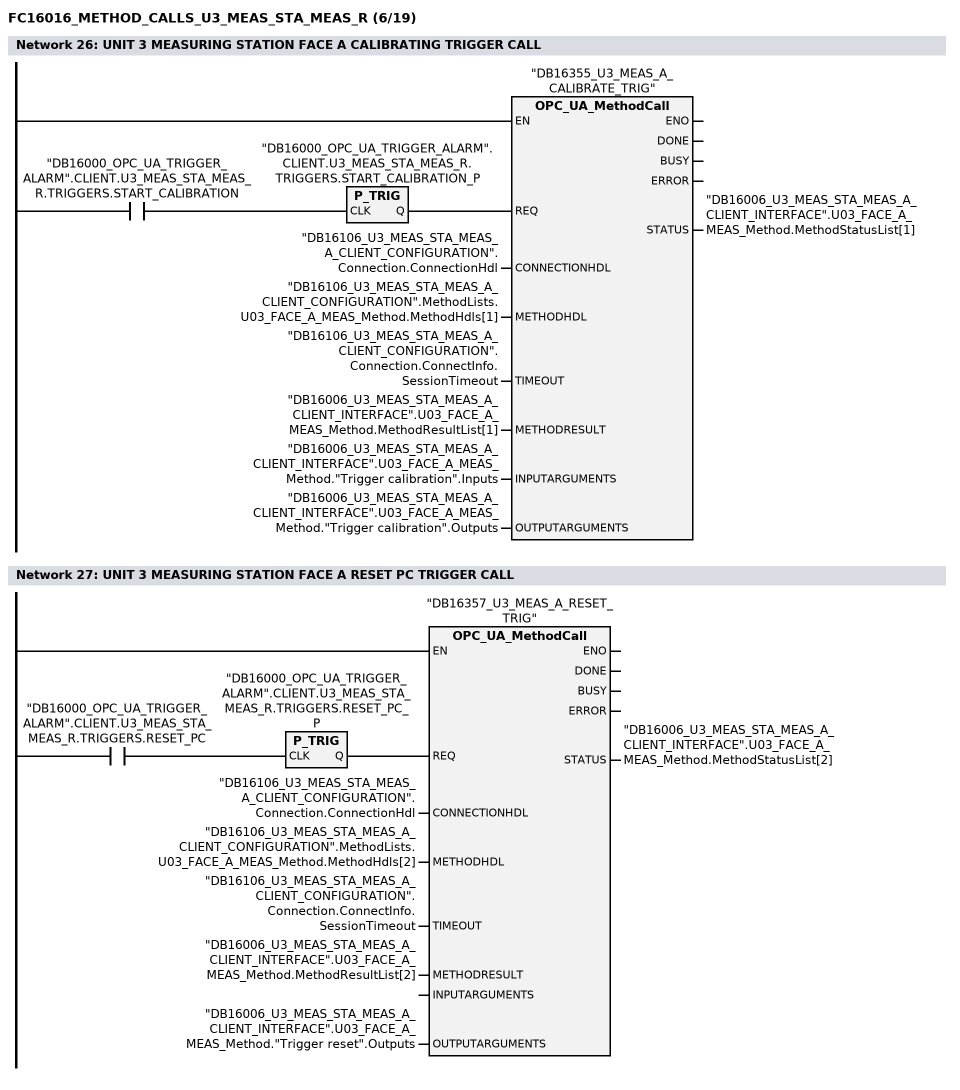
   RUNG wire#powerrail
      "DB16355_U3_MEAS_A_CALIBRATE_TRIG".OPC_UA_MethodCall(REQ := wire#w1, ConnectionHdl := "DB16106_U3_MEAS_STA_MEAS_A_CLIENT_CONFIGURATION".Connection.ConnectionHdl, MethodHdl := "DB16106_U3_MEAS_STA_MEAS_A_CLIENT_CONFIGURATION".MethodLists.U03_FACE_A_MEAS_Method.MethodHdls[1], Timeout := "DB16106_U3_MEAS_STA_MEAS_A_CLIENT_CONFIGURATION".Connection.ConnectInfo.SessionTimeout, MethodResult := "DB16006_U3_MEAS_STA_MEAS_A_CLIENT_INTERFACE".U03_FACE_A_MEAS_Method.MethodResultList[1], InputArguments := "DB16006_U3_MEAS_STA_MEAS_A_CLIENT_INTERFACE".U03_FACE_A_MEAS_Method."Trigger calibration".Inputs, OutputArguments := "DB16006_U3_MEAS_STA_MEAS_A_CLIENT_INTERFACE".U03_FACE_A_MEAS_Method."Trigger calibration".Outputs, Done =>, Busy =>, Error =>, Status => "DB16006_U3_MEAS_STA_MEAS_A_CLIENT_INTERFACE".U03_FACE_A_MEAS_Method.MethodStatusList[1])
   END_RUNG
   RUNG wire#powerrail
      Contact( "DB16000_OPC_UA_TRIGGER_ALARM".CLIENT.U3_MEAS_STA_MEAS_R.TRIGGERS.START_CALIBRATION )
      P_Trig( "DB16000_OPC_UA_TRIGGER_ALARM".CLIENT.U3_MEAS_STA_MEAS_R.TRIGGERS.START_CALIBRATION_P )
   END_RUNG wire#w1
   // the same network as SCL:
   #_w1 := "DB16000_OPC_UA_TRIGGER_ALARM".CLIENT.U3_MEAS_STA_MEAS_R.TRIGGERS.START_CALIBRATION AND NOT "DB16000_OPC_UA_TRIGGER_ALARM".CLIENT.U3_MEAS_STA_MEAS_R.TRIGGERS.START_CALIBRATION_P;   // rising edge
   "DB16000_OPC_UA_TRIGGER_ALARM".CLIENT.U3_MEAS_STA_MEAS_R.TRIGGERS.START_CALIBRATION_P := "DB16000_OPC_UA_TRIGGER_ALARM".CLIENT.U3_MEAS_STA_MEAS_R.TRIGGERS.START_CALIBRATION;
   "DB16355_U3_MEAS_A_CALIBRATE_TRIG"(REQ := #_w1,   // OPC_UA_MethodCall
                           ConnectionHdl := "DB16106_U3_MEAS_STA_MEAS_A_CLIENT_CONFIGURATION".Connection.ConnectionHdl,
                           MethodHdl := "DB16106_U3_MEAS_STA_MEAS_A_CLIENT_CONFIGURATION".MethodLists.U03_FACE_A_MEAS_Method.MethodHdls[1],
                           Timeout := "DB16106_U3_MEAS_STA_MEAS_A_CLIENT_CONFIGURATION".Connection.ConnectInfo.SessionTimeout,
                           MethodResult := "DB16006_U3_MEAS_STA_MEAS_A_CLIENT_INTERFACE".U03_FACE_A_MEAS_Method.MethodResultList[1],
                           InputArguments := "DB16006_U3_MEAS_STA_MEAS_A_CLIENT_INTERFACE".U03_FACE_A_MEAS_Method."Trigger calibration".Inputs,
                           OutputArguments := "DB16006_U3_MEAS_STA_MEAS_A_CLIENT_INTERFACE".U03_FACE_A_MEAS_Method."Trigger calibration".Outputs,
                           Status => "DB16006_U3_MEAS_STA_MEAS_A_CLIENT_INTERFACE".U03_FACE_A_MEAS_Method.MethodStatusList[1]);
END_REGION

REGION Network 27: UNIT 3 MEASURING STATION FACE A RESET PC TRIGGER CALL
   RUNG wire#powerrail
      "DB16357_U3_MEAS_A_RESET_TRIG".OPC_UA_MethodCall(REQ := wire#w1, ConnectionHdl := "DB16106_U3_MEAS_STA_MEAS_A_CLIENT_CONFIGURATION".Connection.ConnectionHdl, MethodHdl := "DB16106_U3_MEAS_STA_MEAS_A_CLIENT_CONFIGURATION".MethodLists.U03_FACE_A_MEAS_Method.MethodHdls[2], Timeout := "DB16106_U3_MEAS_STA_MEAS_A_CLIENT_CONFIGURATION".Connection.ConnectInfo.SessionTimeout, MethodResult := "DB16006_U3_MEAS_STA_MEAS_A_CLIENT_INTERFACE".U03_FACE_A_MEAS_Method.MethodResultList[2], InputArguments :=, OutputArguments := "DB16006_U3_MEAS_STA_MEAS_A_CLIENT_INTERFACE".U03_FACE_A_MEAS_Method."Trigger reset".Outputs, Done =>, Busy =>, Error =>, Status => "DB16006_U3_MEAS_STA_MEAS_A_CLIENT_INTERFACE".U03_FACE_A_MEAS_Method.MethodStatusList[2])
   END_RUNG
   RUNG wire#powerrail
      Contact( "DB16000_OPC_UA_TRIGGER_ALARM".CLIENT.U3_MEAS_STA_MEAS_R.TRIGGERS.RESET_PC )
      P_Trig( "DB16000_OPC_UA_TRIGGER_ALARM".CLIENT.U3_MEAS_STA_MEAS_R.TRIGGERS.RESET_PC_P )
   END_RUNG wire#w1
   // the same network as SCL:
   #_w1 := "DB16000_OPC_UA_TRIGGER_ALARM".CLIENT.U3_MEAS_STA_MEAS_R.TRIGGERS.RESET_PC AND NOT "DB16000_OPC_UA_TRIGGER_ALARM".CLIENT.U3_MEAS_STA_MEAS_R.TRIGGERS.RESET_PC_P;   // rising edge
   "DB16000_OPC_UA_TRIGGER_ALARM".CLIENT.U3_MEAS_STA_MEAS_R.TRIGGERS.RESET_PC_P := "DB16000_OPC_UA_TRIGGER_ALARM".CLIENT.U3_MEAS_STA_MEAS_R.TRIGGERS.RESET_PC;
   "DB16357_U3_MEAS_A_RESET_TRIG"(REQ := #_w1,   // OPC_UA_MethodCall
                           ConnectionHdl := "DB16106_U3_MEAS_STA_MEAS_A_CLIENT_CONFIGURATION".Connection.ConnectionHdl,
                           MethodHdl := "DB16106_U3_MEAS_STA_MEAS_A_CLIENT_CONFIGURATION".MethodLists.U03_FACE_A_MEAS_Method.MethodHdls[2],
                           Timeout := "DB16106_U3_MEAS_STA_MEAS_A_CLIENT_CONFIGURATION".Connection.ConnectInfo.SessionTimeout,
                           MethodResult := "DB16006_U3_MEAS_STA_MEAS_A_CLIENT_INTERFACE".U03_FACE_A_MEAS_Method.MethodResultList[2],
                           OutputArguments := "DB16006_U3_MEAS_STA_MEAS_A_CLIENT_INTERFACE".U03_FACE_A_MEAS_Method."Trigger reset".Outputs,
                           Status => "DB16006_U3_MEAS_STA_MEAS_A_CLIENT_INTERFACE".U03_FACE_A_MEAS_Method.MethodStatusList[2]);
END_REGION

REGION Network 28: UNIT 3 MEASURING STATION FACE A READ VARIABLES TRIGGER CALL
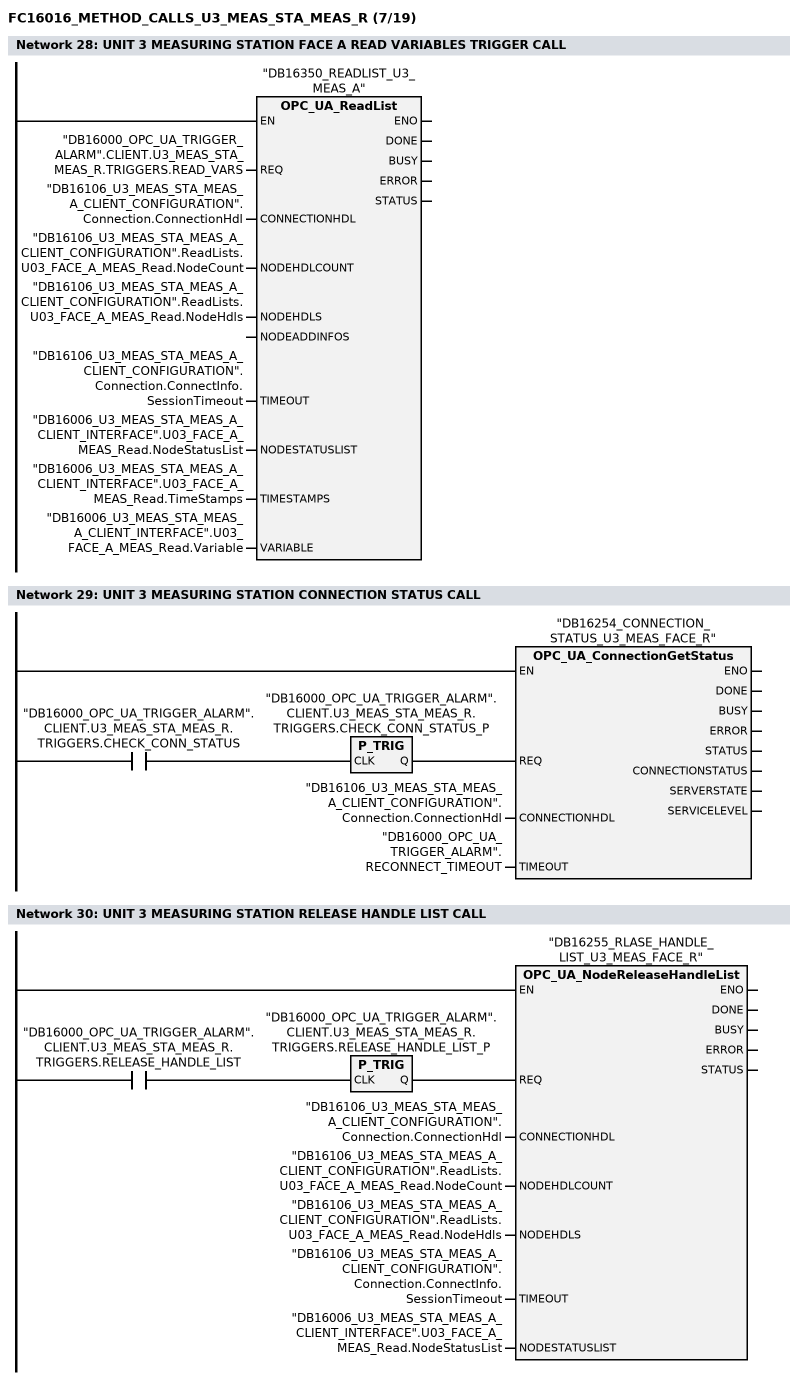
   RUNG wire#powerrail
      "DB16350_READLIST_U3_MEAS_A".OPC_UA_ReadList(REQ := "DB16000_OPC_UA_TRIGGER_ALARM".CLIENT.U3_MEAS_STA_MEAS_R.TRIGGERS.READ_VARS, ConnectionHdl := "DB16106_U3_MEAS_STA_MEAS_A_CLIENT_CONFIGURATION".Connection.ConnectionHdl, NodeHdlCount := "DB16106_U3_MEAS_STA_MEAS_A_CLIENT_CONFIGURATION".ReadLists.U03_FACE_A_MEAS_Read.NodeCount, NodeHdls := "DB16106_U3_MEAS_STA_MEAS_A_CLIENT_CONFIGURATION".ReadLists.U03_FACE_A_MEAS_Read.NodeHdls, NodeAddInfos :=, Timeout := "DB16106_U3_MEAS_STA_MEAS_A_CLIENT_CONFIGURATION".Connection.ConnectInfo.SessionTimeout, NodeStatusList := "DB16006_U3_MEAS_STA_MEAS_A_CLIENT_INTERFACE".U03_FACE_A_MEAS_Read.NodeStatusList, TimeStamps := "DB16006_U3_MEAS_STA_MEAS_A_CLIENT_INTERFACE".U03_FACE_A_MEAS_Read.TimeStamps, Variable := "DB16006_U3_MEAS_STA_MEAS_A_CLIENT_INTERFACE".U03_FACE_A_MEAS_Read.Variable, Done =>, Busy =>, Error =>, Status =>)
   END_RUNG
   // the same network as SCL:
   "DB16350_READLIST_U3_MEAS_A"(REQ := "DB16000_OPC_UA_TRIGGER_ALARM".CLIENT.U3_MEAS_STA_MEAS_R.TRIGGERS.READ_VARS,   // OPC_UA_ReadList
                           ConnectionHdl := "DB16106_U3_MEAS_STA_MEAS_A_CLIENT_CONFIGURATION".Connection.ConnectionHdl,
                           NodeHdlCount := "DB16106_U3_MEAS_STA_MEAS_A_CLIENT_CONFIGURATION".ReadLists.U03_FACE_A_MEAS_Read.NodeCount,
                           NodeHdls := "DB16106_U3_MEAS_STA_MEAS_A_CLIENT_CONFIGURATION".ReadLists.U03_FACE_A_MEAS_Read.NodeHdls,
                           Timeout := "DB16106_U3_MEAS_STA_MEAS_A_CLIENT_CONFIGURATION".Connection.ConnectInfo.SessionTimeout,
                           NodeStatusList := "DB16006_U3_MEAS_STA_MEAS_A_CLIENT_INTERFACE".U03_FACE_A_MEAS_Read.NodeStatusList,
                           TimeStamps := "DB16006_U3_MEAS_STA_MEAS_A_CLIENT_INTERFACE".U03_FACE_A_MEAS_Read.TimeStamps,
                           Variable := "DB16006_U3_MEAS_STA_MEAS_A_CLIENT_INTERFACE".U03_FACE_A_MEAS_Read.Variable);
END_REGION

REGION Network 29: UNIT 3 MEASURING STATION CONNECTION STATUS CALL
   RUNG wire#powerrail
      "DB16254_CONNECTION_STATUS_U3_MEAS_FACE_R".OPC_UA_ConnectionGetStatus(REQ := wire#w1, ConnectionHdl := "DB16106_U3_MEAS_STA_MEAS_A_CLIENT_CONFIGURATION".Connection.ConnectionHdl, Timeout := "DB16000_OPC_UA_TRIGGER_ALARM".RECONNECT_TIMEOUT, Done =>, Busy =>, Error =>, Status =>, ConnectionStatus =>, ServerState =>, ServiceLevel =>)
   END_RUNG
   RUNG wire#powerrail
      Contact( "DB16000_OPC_UA_TRIGGER_ALARM".CLIENT.U3_MEAS_STA_MEAS_R.TRIGGERS.CHECK_CONN_STATUS )
      P_Trig( "DB16000_OPC_UA_TRIGGER_ALARM".CLIENT.U3_MEAS_STA_MEAS_R.TRIGGERS.CHECK_CONN_STATUS_P )
   END_RUNG wire#w1
   // the same network as SCL:
   #_w1 := "DB16000_OPC_UA_TRIGGER_ALARM".CLIENT.U3_MEAS_STA_MEAS_R.TRIGGERS.CHECK_CONN_STATUS AND NOT "DB16000_OPC_UA_TRIGGER_ALARM".CLIENT.U3_MEAS_STA_MEAS_R.TRIGGERS.CHECK_CONN_STATUS_P;   // rising edge
   "DB16000_OPC_UA_TRIGGER_ALARM".CLIENT.U3_MEAS_STA_MEAS_R.TRIGGERS.CHECK_CONN_STATUS_P := "DB16000_OPC_UA_TRIGGER_ALARM".CLIENT.U3_MEAS_STA_MEAS_R.TRIGGERS.CHECK_CONN_STATUS;
   "DB16254_CONNECTION_STATUS_U3_MEAS_FACE_R"(REQ := #_w1,   // OPC_UA_ConnectionGetStatus
                           ConnectionHdl := "DB16106_U3_MEAS_STA_MEAS_A_CLIENT_CONFIGURATION".Connection.ConnectionHdl,
                           Timeout := "DB16000_OPC_UA_TRIGGER_ALARM".RECONNECT_TIMEOUT);
END_REGION

REGION Network 30: UNIT 3 MEASURING STATION RELEASE HANDLE LIST CALL
   RUNG wire#powerrail
      "DB16255_RLASE_HANDLE_LIST_U3_MEAS_FACE_R".OPC_UA_NodeReleaseHandleList(REQ := wire#w1, ConnectionHdl := "DB16106_U3_MEAS_STA_MEAS_A_CLIENT_CONFIGURATION".Connection.ConnectionHdl, NodeHdlCount := "DB16106_U3_MEAS_STA_MEAS_A_CLIENT_CONFIGURATION".ReadLists.U03_FACE_A_MEAS_Read.NodeCount, NodeHdls := "DB16106_U3_MEAS_STA_MEAS_A_CLIENT_CONFIGURATION".ReadLists.U03_FACE_A_MEAS_Read.NodeHdls, Timeout := "DB16106_U3_MEAS_STA_MEAS_A_CLIENT_CONFIGURATION".Connection.ConnectInfo.SessionTimeout, NodeStatusList := "DB16006_U3_MEAS_STA_MEAS_A_CLIENT_INTERFACE".U03_FACE_A_MEAS_Read.NodeStatusList, Done =>, Busy =>, Error =>, Status =>)
   END_RUNG
   RUNG wire#powerrail
      Contact( "DB16000_OPC_UA_TRIGGER_ALARM".CLIENT.U3_MEAS_STA_MEAS_R.TRIGGERS.RELEASE_HANDLE_LIST )
      P_Trig( "DB16000_OPC_UA_TRIGGER_ALARM".CLIENT.U3_MEAS_STA_MEAS_R.TRIGGERS.RELEASE_HANDLE_LIST_P )
   END_RUNG wire#w1
   // the same network as SCL:
   #_w1 := "DB16000_OPC_UA_TRIGGER_ALARM".CLIENT.U3_MEAS_STA_MEAS_R.TRIGGERS.RELEASE_HANDLE_LIST AND NOT "DB16000_OPC_UA_TRIGGER_ALARM".CLIENT.U3_MEAS_STA_MEAS_R.TRIGGERS.RELEASE_HANDLE_LIST_P;   // rising edge
   "DB16000_OPC_UA_TRIGGER_ALARM".CLIENT.U3_MEAS_STA_MEAS_R.TRIGGERS.RELEASE_HANDLE_LIST_P := "DB16000_OPC_UA_TRIGGER_ALARM".CLIENT.U3_MEAS_STA_MEAS_R.TRIGGERS.RELEASE_HANDLE_LIST;
   "DB16255_RLASE_HANDLE_LIST_U3_MEAS_FACE_R"(REQ := #_w1,   // OPC_UA_NodeReleaseHandleList
                           ConnectionHdl := "DB16106_U3_MEAS_STA_MEAS_A_CLIENT_CONFIGURATION".Connection.ConnectionHdl,
                           NodeHdlCount := "DB16106_U3_MEAS_STA_MEAS_A_CLIENT_CONFIGURATION".ReadLists.U03_FACE_A_MEAS_Read.NodeCount,
                           NodeHdls := "DB16106_U3_MEAS_STA_MEAS_A_CLIENT_CONFIGURATION".ReadLists.U03_FACE_A_MEAS_Read.NodeHdls,
                           Timeout := "DB16106_U3_MEAS_STA_MEAS_A_CLIENT_CONFIGURATION".Connection.ConnectInfo.SessionTimeout,
                           NodeStatusList := "DB16006_U3_MEAS_STA_MEAS_A_CLIENT_INTERFACE".U03_FACE_A_MEAS_Read.NodeStatusList);
END_REGION

REGION Network 31: UNIT 3 MEASURING STATION RELEASE METHOD HANDLE LIST CALL
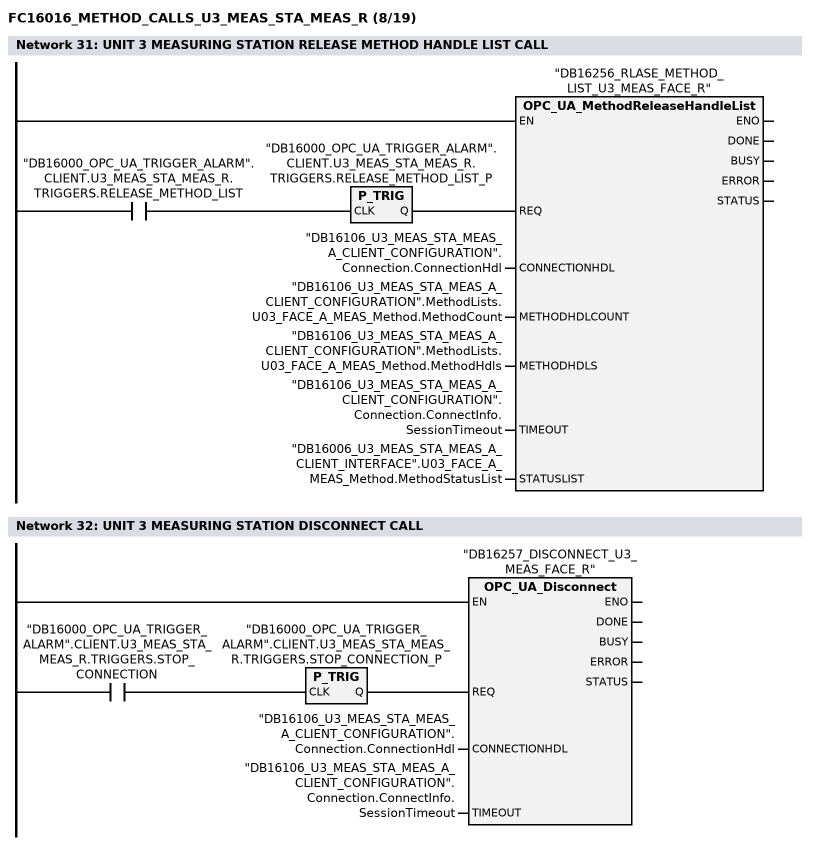
   RUNG wire#powerrail
      "DB16256_RLASE_METHOD_LIST_U3_MEAS_FACE_R".OPC_UA_MethodReleaseHandleList(REQ := wire#w1, ConnectionHdl := "DB16106_U3_MEAS_STA_MEAS_A_CLIENT_CONFIGURATION".Connection.ConnectionHdl, MethodHdlCount := "DB16106_U3_MEAS_STA_MEAS_A_CLIENT_CONFIGURATION".MethodLists.U03_FACE_A_MEAS_Method.MethodCount, MethodHdls := "DB16106_U3_MEAS_STA_MEAS_A_CLIENT_CONFIGURATION".MethodLists.U03_FACE_A_MEAS_Method.MethodHdls, Timeout := "DB16106_U3_MEAS_STA_MEAS_A_CLIENT_CONFIGURATION".Connection.ConnectInfo.SessionTimeout, StatusList := "DB16006_U3_MEAS_STA_MEAS_A_CLIENT_INTERFACE".U03_FACE_A_MEAS_Method.MethodStatusList, Done =>, Busy =>, Error =>, Status =>)
   END_RUNG
   RUNG wire#powerrail
      Contact( "DB16000_OPC_UA_TRIGGER_ALARM".CLIENT.U3_MEAS_STA_MEAS_R.TRIGGERS.RELEASE_METHOD_LIST )
      P_Trig( "DB16000_OPC_UA_TRIGGER_ALARM".CLIENT.U3_MEAS_STA_MEAS_R.TRIGGERS.RELEASE_METHOD_LIST_P )
   END_RUNG wire#w1
   // the same network as SCL:
   #_w1 := "DB16000_OPC_UA_TRIGGER_ALARM".CLIENT.U3_MEAS_STA_MEAS_R.TRIGGERS.RELEASE_METHOD_LIST AND NOT "DB16000_OPC_UA_TRIGGER_ALARM".CLIENT.U3_MEAS_STA_MEAS_R.TRIGGERS.RELEASE_METHOD_LIST_P;   // rising edge
   "DB16000_OPC_UA_TRIGGER_ALARM".CLIENT.U3_MEAS_STA_MEAS_R.TRIGGERS.RELEASE_METHOD_LIST_P := "DB16000_OPC_UA_TRIGGER_ALARM".CLIENT.U3_MEAS_STA_MEAS_R.TRIGGERS.RELEASE_METHOD_LIST;
   "DB16256_RLASE_METHOD_LIST_U3_MEAS_FACE_R"(REQ := #_w1,   // OPC_UA_MethodReleaseHandleList
                           ConnectionHdl := "DB16106_U3_MEAS_STA_MEAS_A_CLIENT_CONFIGURATION".Connection.ConnectionHdl,
                           MethodHdlCount := "DB16106_U3_MEAS_STA_MEAS_A_CLIENT_CONFIGURATION".MethodLists.U03_FACE_A_MEAS_Method.MethodCount,
                           MethodHdls := "DB16106_U3_MEAS_STA_MEAS_A_CLIENT_CONFIGURATION".MethodLists.U03_FACE_A_MEAS_Method.MethodHdls,
                           Timeout := "DB16106_U3_MEAS_STA_MEAS_A_CLIENT_CONFIGURATION".Connection.ConnectInfo.SessionTimeout,
                           StatusList := "DB16006_U3_MEAS_STA_MEAS_A_CLIENT_INTERFACE".U03_FACE_A_MEAS_Method.MethodStatusList);
END_REGION

REGION Network 32: UNIT 3 MEASURING STATION DISCONNECT CALL
   RUNG wire#powerrail
      "DB16257_DISCONNECT_U3_MEAS_FACE_R".OPC_UA_Disconnect(REQ := wire#w1, ConnectionHdl := "DB16106_U3_MEAS_STA_MEAS_A_CLIENT_CONFIGURATION".Connection.ConnectionHdl, Timeout := "DB16106_U3_MEAS_STA_MEAS_A_CLIENT_CONFIGURATION".Connection.ConnectInfo.SessionTimeout, Done =>, Busy =>, Error =>, Status =>)
   END_RUNG
   RUNG wire#powerrail
      Contact( "DB16000_OPC_UA_TRIGGER_ALARM".CLIENT.U3_MEAS_STA_MEAS_R.TRIGGERS.STOP_CONNECTION )
      P_Trig( "DB16000_OPC_UA_TRIGGER_ALARM".CLIENT.U3_MEAS_STA_MEAS_R.TRIGGERS.STOP_CONNECTION_P )
   END_RUNG wire#w1
   // the same network as SCL:
   #_w1 := "DB16000_OPC_UA_TRIGGER_ALARM".CLIENT.U3_MEAS_STA_MEAS_R.TRIGGERS.STOP_CONNECTION AND NOT "DB16000_OPC_UA_TRIGGER_ALARM".CLIENT.U3_MEAS_STA_MEAS_R.TRIGGERS.STOP_CONNECTION_P;   // rising edge
   "DB16000_OPC_UA_TRIGGER_ALARM".CLIENT.U3_MEAS_STA_MEAS_R.TRIGGERS.STOP_CONNECTION_P := "DB16000_OPC_UA_TRIGGER_ALARM".CLIENT.U3_MEAS_STA_MEAS_R.TRIGGERS.STOP_CONNECTION;
   "DB16257_DISCONNECT_U3_MEAS_FACE_R"(REQ := #_w1,   // OPC_UA_Disconnect
                           ConnectionHdl := "DB16106_U3_MEAS_STA_MEAS_A_CLIENT_CONFIGURATION".Connection.ConnectionHdl,
                           Timeout := "DB16106_U3_MEAS_STA_MEAS_A_CLIENT_CONFIGURATION".Connection.ConnectInfo.SessionTimeout);
END_REGION

REGION Network 33: UNIT 3 STATION 2 MEAS RECONNECT
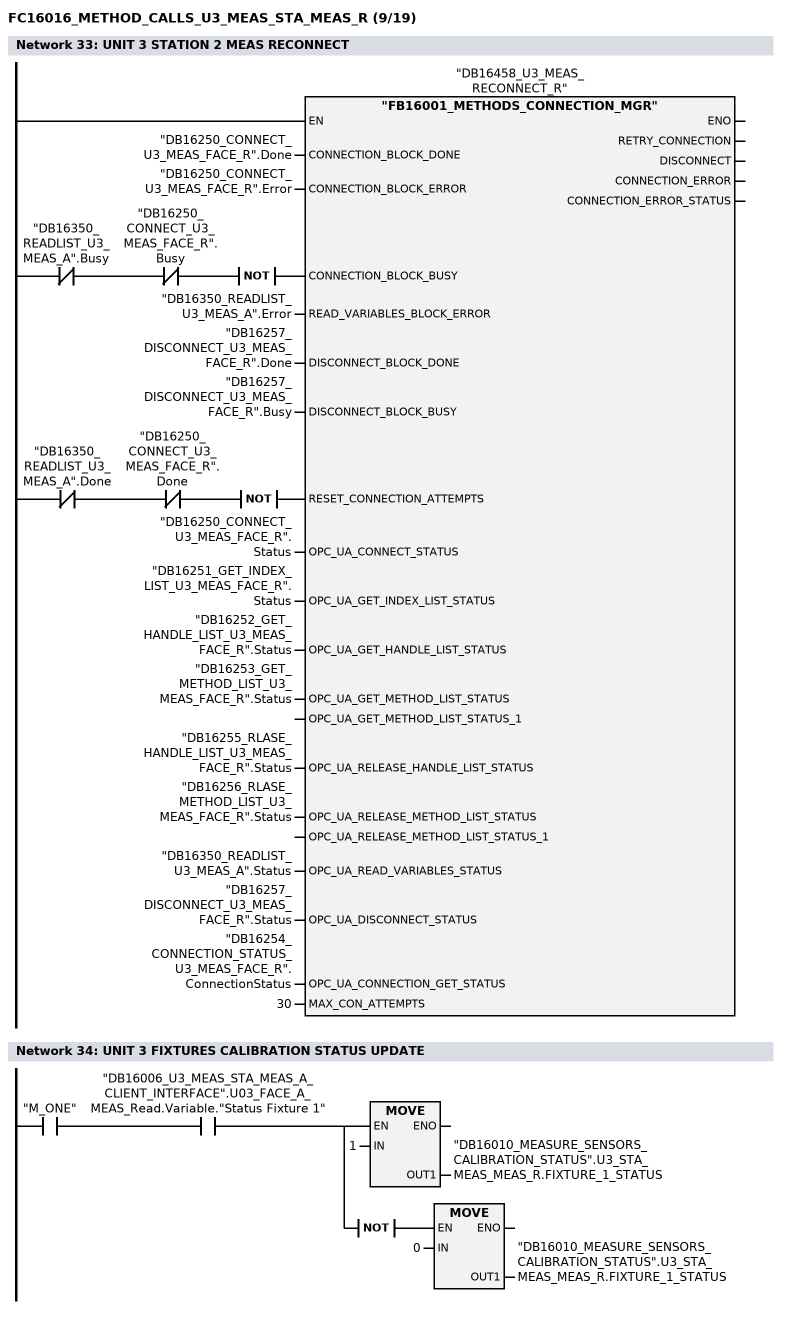
   RUNG wire#powerrail
      "DB16458_U3_MEAS_RECONNECT_R"(CONNECTION_BLOCK_BUSY := wire#w1, RESET_CONNECTION_ATTEMPTS := wire#w2, CONNECTION_BLOCK_DONE := "DB16250_CONNECT_U3_MEAS_FACE_R".Done, CONNECTION_BLOCK_ERROR := "DB16250_CONNECT_U3_MEAS_FACE_R".Error, READ_VARIABLES_BLOCK_ERROR := "DB16350_READLIST_U3_MEAS_A".Error, DISCONNECT_BLOCK_DONE := "DB16257_DISCONNECT_U3_MEAS_FACE_R".Done, DISCONNECT_BLOCK_BUSY := "DB16257_DISCONNECT_U3_MEAS_FACE_R".Busy, OPC_UA_CONNECT_STATUS := "DB16250_CONNECT_U3_MEAS_FACE_R".Status, OPC_UA_GET_INDEX_LIST_STATUS := "DB16251_GET_INDEX_LIST_U3_MEAS_FACE_R".Status, OPC_UA_GET_HANDLE_LIST_STATUS := "DB16252_GET_HANDLE_LIST_U3_MEAS_FACE_R".Status, OPC_UA_GET_METHOD_LIST_STATUS := "DB16253_GET_METHOD_LIST_U3_MEAS_FACE_R".Status, OPC_UA_GET_METHOD_LIST_STATUS_1 :=, OPC_UA_RELEASE_HANDLE_LIST_STATUS := "DB16255_RLASE_HANDLE_LIST_U3_MEAS_FACE_R".Status, OPC_UA_RELEASE_METHOD_LIST_STATUS := "DB16256_RLASE_METHOD_LIST_U3_MEAS_FACE_R".Status, OPC_UA_RELEASE_METHOD_LIST_STATUS_1 :=, OPC_UA_READ_VARIABLES_STATUS := "DB16350_READLIST_U3_MEAS_A".Status, OPC_UA_DISCONNECT_STATUS := "DB16257_DISCONNECT_U3_MEAS_FACE_R".Status, OPC_UA_CONNECTION_GET_STATUS := "DB16254_CONNECTION_STATUS_U3_MEAS_FACE_R".ConnectionStatus, MAX_CON_ATTEMPTS := 30, RETRY_CONNECTION =>, DISCONNECT =>, CONNECTION_ERROR =>, CONNECTION_ERROR_STATUS =>)
   END_RUNG
   RUNG wire#powerrail
      I_Contact( "DB16350_READLIST_U3_MEAS_A".Busy )
      I_Contact( "DB16250_CONNECT_U3_MEAS_FACE_R".Busy )
      Not()
   END_RUNG wire#w1
   RUNG wire#powerrail
      I_Contact( "DB16350_READLIST_U3_MEAS_A".Done )
      I_Contact( "DB16250_CONNECT_U3_MEAS_FACE_R".Done )
      Not()
   END_RUNG wire#w2
   // the same network as SCL:
   "DB16458_U3_MEAS_RECONNECT_R"(CONNECTION_BLOCK_DONE := "DB16250_CONNECT_U3_MEAS_FACE_R".Done,   // "FB16001_METHODS_CONNECTION_MGR"
                           CONNECTION_BLOCK_ERROR := "DB16250_CONNECT_U3_MEAS_FACE_R".Error,
                           CONNECTION_BLOCK_BUSY := NOT (NOT "DB16350_READLIST_U3_MEAS_A".Busy AND NOT "DB16250_CONNECT_U3_MEAS_FACE_R".Busy),
                           READ_VARIABLES_BLOCK_ERROR := "DB16350_READLIST_U3_MEAS_A".Error,
                           DISCONNECT_BLOCK_DONE := "DB16257_DISCONNECT_U3_MEAS_FACE_R".Done,
                           DISCONNECT_BLOCK_BUSY := "DB16257_DISCONNECT_U3_MEAS_FACE_R".Busy,
                           RESET_CONNECTION_ATTEMPTS := NOT (NOT "DB16350_READLIST_U3_MEAS_A".Done AND NOT "DB16250_CONNECT_U3_MEAS_FACE_R".Done),
                           OPC_UA_CONNECT_STATUS := "DB16250_CONNECT_U3_MEAS_FACE_R".Status,
                           OPC_UA_GET_INDEX_LIST_STATUS := "DB16251_GET_INDEX_LIST_U3_MEAS_FACE_R".Status,
                           OPC_UA_GET_HANDLE_LIST_STATUS := "DB16252_GET_HANDLE_LIST_U3_MEAS_FACE_R".Status,
                           OPC_UA_GET_METHOD_LIST_STATUS := "DB16253_GET_METHOD_LIST_U3_MEAS_FACE_R".Status,
                           OPC_UA_RELEASE_HANDLE_LIST_STATUS := "DB16255_RLASE_HANDLE_LIST_U3_MEAS_FACE_R".Status,
                           OPC_UA_RELEASE_METHOD_LIST_STATUS := "DB16256_RLASE_METHOD_LIST_U3_MEAS_FACE_R".Status,
                           OPC_UA_READ_VARIABLES_STATUS := "DB16350_READLIST_U3_MEAS_A".Status,
                           OPC_UA_DISCONNECT_STATUS := "DB16257_DISCONNECT_U3_MEAS_FACE_R".Status,
                           OPC_UA_CONNECTION_GET_STATUS := "DB16254_CONNECTION_STATUS_U3_MEAS_FACE_R".ConnectionStatus,
                           MAX_CON_ATTEMPTS := 30);
END_REGION

REGION Network 34: UNIT 3 FIXTURES CALIBRATION STATUS UPDATE
   RUNG wire#powerrail
      Contact( "M_ONE" )
      Contact( "DB16006_U3_MEAS_STA_MEAS_A_CLIENT_INTERFACE".U03_FACE_A_MEAS_Read.Variable."Status Fixture 1" )
      wire#w1
      Move(in := 1, out1 => "DB16010_MEASURE_SENSORS_CALIBRATION_STATUS".U3_STA_MEAS_MEAS_R.FIXTURE_1_STATUS)
   END_RUNG
   RUNG wire#w1
      Not()
      Move(in := 0, out1 => "DB16010_MEASURE_SENSORS_CALIBRATION_STATUS".U3_STA_MEAS_MEAS_R.FIXTURE_1_STATUS)
   END_RUNG
   // the same network as SCL:
   #_w1 := "M_ONE" AND "DB16006_U3_MEAS_STA_MEAS_A_CLIENT_INTERFACE".U03_FACE_A_MEAS_Read.Variable."Status Fixture 1";
   IF #_w1 THEN
       "DB16010_MEASURE_SENSORS_CALIBRATION_STATUS".U3_STA_MEAS_MEAS_R.FIXTURE_1_STATUS := 1;
   END_IF;
   IF NOT #_w1 THEN
       "DB16010_MEASURE_SENSORS_CALIBRATION_STATUS".U3_STA_MEAS_MEAS_R.FIXTURE_1_STATUS := 0;
   END_IF;
END_REGION

REGION Network 35: UNIT 3 MEASURING STATION FACE A COMPUTER CONNECTION ALARM
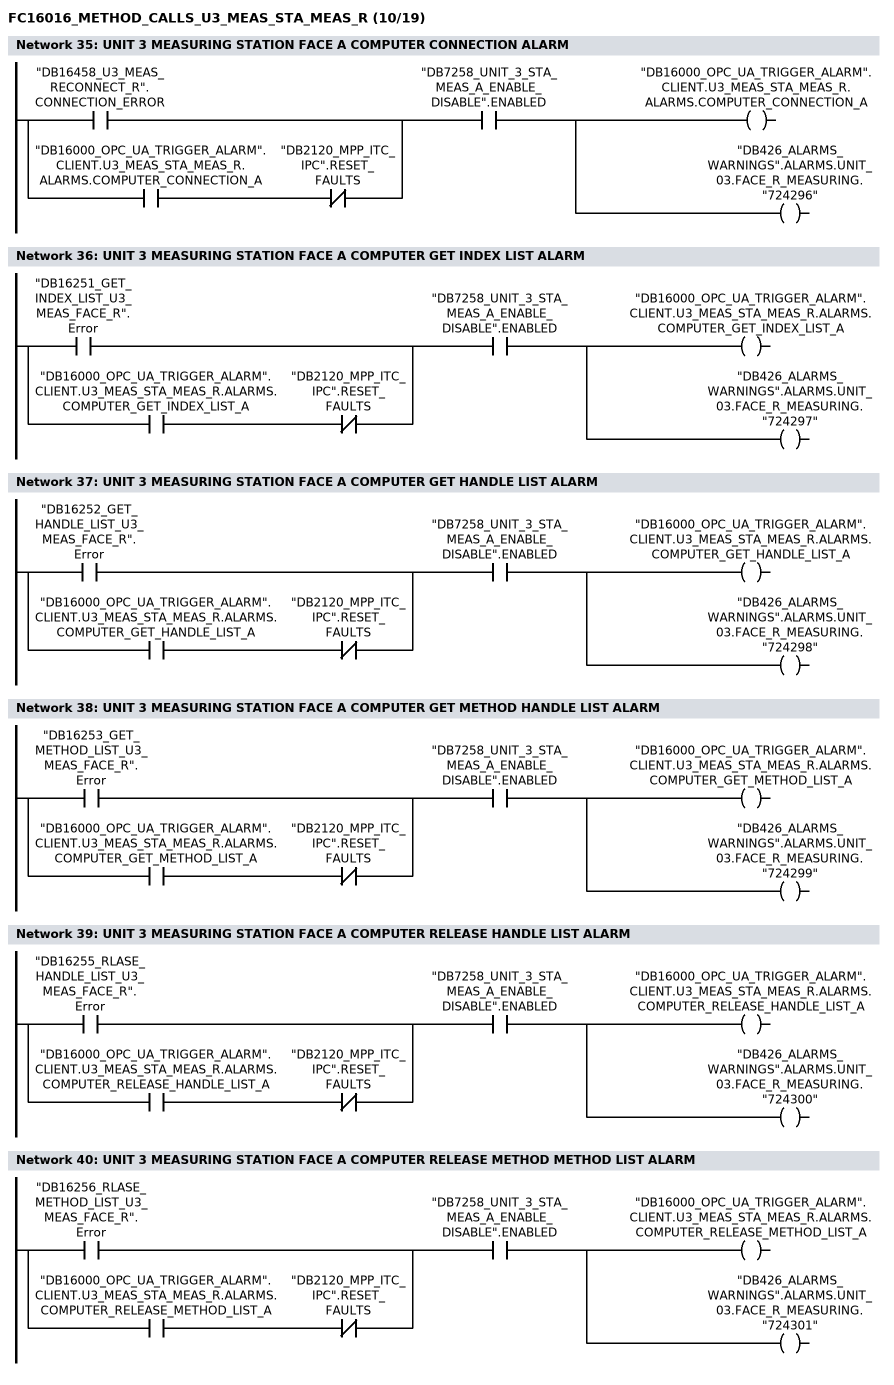
   RUNG wire#powerrail
      Contact( "DB16458_U3_MEAS_RECONNECT_R".CONNECTION_ERROR )
      wire#w1
      Contact( "DB7258_UNIT_3_STA_MEAS_A_ENABLE_DISABLE".ENABLED )
      wire#w2
      Coil( "DB16000_OPC_UA_TRIGGER_ALARM".CLIENT.U3_MEAS_STA_MEAS_R.ALARMS.COMPUTER_CONNECTION_A )
   END_RUNG
   RUNG wire#powerrail
      Contact( "DB16000_OPC_UA_TRIGGER_ALARM".CLIENT.U3_MEAS_STA_MEAS_R.ALARMS.COMPUTER_CONNECTION_A )
      I_Contact( "DB2120_MPP_ITC_IPC".RESET_FAULTS )
   END_RUNG wire#w1
   RUNG wire#w2
      Coil( "DB426_ALARMS_WARNINGS".ALARMS.UNIT_03.FACE_R_MEASURING."724296" )
   END_RUNG
   // the same network as SCL:
   "DB16000_OPC_UA_TRIGGER_ALARM".CLIENT.U3_MEAS_STA_MEAS_R.ALARMS.COMPUTER_CONNECTION_A := ("DB16458_U3_MEAS_RECONNECT_R".CONNECTION_ERROR OR ("DB16000_OPC_UA_TRIGGER_ALARM".CLIENT.U3_MEAS_STA_MEAS_R.ALARMS.COMPUTER_CONNECTION_A AND NOT "DB2120_MPP_ITC_IPC".RESET_FAULTS)) AND "DB7258_UNIT_3_STA_MEAS_A_ENABLE_DISABLE".ENABLED;
   "DB426_ALARMS_WARNINGS".ALARMS.UNIT_03.FACE_R_MEASURING."724296" := "DB16000_OPC_UA_TRIGGER_ALARM".CLIENT.U3_MEAS_STA_MEAS_R.ALARMS.COMPUTER_CONNECTION_A;
END_REGION

REGION Network 36: UNIT 3 MEASURING STATION FACE A COMPUTER GET INDEX LIST ALARM
   RUNG wire#powerrail
      Contact( "DB16251_GET_INDEX_LIST_U3_MEAS_FACE_R".Error )
      wire#w1
      Contact( "DB7258_UNIT_3_STA_MEAS_A_ENABLE_DISABLE".ENABLED )
      wire#w2
      Coil( "DB16000_OPC_UA_TRIGGER_ALARM".CLIENT.U3_MEAS_STA_MEAS_R.ALARMS.COMPUTER_GET_INDEX_LIST_A )
   END_RUNG
   RUNG wire#powerrail
      Contact( "DB16000_OPC_UA_TRIGGER_ALARM".CLIENT.U3_MEAS_STA_MEAS_R.ALARMS.COMPUTER_GET_INDEX_LIST_A )
      I_Contact( "DB2120_MPP_ITC_IPC".RESET_FAULTS )
   END_RUNG wire#w1
   RUNG wire#w2
      Coil( "DB426_ALARMS_WARNINGS".ALARMS.UNIT_03.FACE_R_MEASURING."724297" )
   END_RUNG
   // the same network as SCL:
   "DB16000_OPC_UA_TRIGGER_ALARM".CLIENT.U3_MEAS_STA_MEAS_R.ALARMS.COMPUTER_GET_INDEX_LIST_A := ("DB16251_GET_INDEX_LIST_U3_MEAS_FACE_R".Error OR ("DB16000_OPC_UA_TRIGGER_ALARM".CLIENT.U3_MEAS_STA_MEAS_R.ALARMS.COMPUTER_GET_INDEX_LIST_A AND NOT "DB2120_MPP_ITC_IPC".RESET_FAULTS)) AND "DB7258_UNIT_3_STA_MEAS_A_ENABLE_DISABLE".ENABLED;
   "DB426_ALARMS_WARNINGS".ALARMS.UNIT_03.FACE_R_MEASURING."724297" := "DB16000_OPC_UA_TRIGGER_ALARM".CLIENT.U3_MEAS_STA_MEAS_R.ALARMS.COMPUTER_GET_INDEX_LIST_A;
END_REGION

REGION Network 37: UNIT 3 MEASURING STATION FACE A COMPUTER GET HANDLE LIST ALARM
   RUNG wire#powerrail
      Contact( "DB16252_GET_HANDLE_LIST_U3_MEAS_FACE_R".Error )
      wire#w1
      Contact( "DB7258_UNIT_3_STA_MEAS_A_ENABLE_DISABLE".ENABLED )
      wire#w2
      Coil( "DB16000_OPC_UA_TRIGGER_ALARM".CLIENT.U3_MEAS_STA_MEAS_R.ALARMS.COMPUTER_GET_HANDLE_LIST_A )
   END_RUNG
   RUNG wire#powerrail
      Contact( "DB16000_OPC_UA_TRIGGER_ALARM".CLIENT.U3_MEAS_STA_MEAS_R.ALARMS.COMPUTER_GET_HANDLE_LIST_A )
      I_Contact( "DB2120_MPP_ITC_IPC".RESET_FAULTS )
   END_RUNG wire#w1
   RUNG wire#w2
      Coil( "DB426_ALARMS_WARNINGS".ALARMS.UNIT_03.FACE_R_MEASURING."724298" )
   END_RUNG
   // the same network as SCL:
   "DB16000_OPC_UA_TRIGGER_ALARM".CLIENT.U3_MEAS_STA_MEAS_R.ALARMS.COMPUTER_GET_HANDLE_LIST_A := ("DB16252_GET_HANDLE_LIST_U3_MEAS_FACE_R".Error OR ("DB16000_OPC_UA_TRIGGER_ALARM".CLIENT.U3_MEAS_STA_MEAS_R.ALARMS.COMPUTER_GET_HANDLE_LIST_A AND NOT "DB2120_MPP_ITC_IPC".RESET_FAULTS)) AND "DB7258_UNIT_3_STA_MEAS_A_ENABLE_DISABLE".ENABLED;
   "DB426_ALARMS_WARNINGS".ALARMS.UNIT_03.FACE_R_MEASURING."724298" := "DB16000_OPC_UA_TRIGGER_ALARM".CLIENT.U3_MEAS_STA_MEAS_R.ALARMS.COMPUTER_GET_HANDLE_LIST_A;
END_REGION

REGION Network 38: UNIT 3 MEASURING STATION FACE A COMPUTER GET METHOD HANDLE LIST ALARM
   RUNG wire#powerrail
      Contact( "DB16253_GET_METHOD_LIST_U3_MEAS_FACE_R".Error )
      wire#w1
      Contact( "DB7258_UNIT_3_STA_MEAS_A_ENABLE_DISABLE".ENABLED )
      wire#w2
      Coil( "DB16000_OPC_UA_TRIGGER_ALARM".CLIENT.U3_MEAS_STA_MEAS_R.ALARMS.COMPUTER_GET_METHOD_LIST_A )
   END_RUNG
   RUNG wire#powerrail
      Contact( "DB16000_OPC_UA_TRIGGER_ALARM".CLIENT.U3_MEAS_STA_MEAS_R.ALARMS.COMPUTER_GET_METHOD_LIST_A )
      I_Contact( "DB2120_MPP_ITC_IPC".RESET_FAULTS )
   END_RUNG wire#w1
   RUNG wire#w2
      Coil( "DB426_ALARMS_WARNINGS".ALARMS.UNIT_03.FACE_R_MEASURING."724299" )
   END_RUNG
   // the same network as SCL:
   "DB16000_OPC_UA_TRIGGER_ALARM".CLIENT.U3_MEAS_STA_MEAS_R.ALARMS.COMPUTER_GET_METHOD_LIST_A := ("DB16253_GET_METHOD_LIST_U3_MEAS_FACE_R".Error OR ("DB16000_OPC_UA_TRIGGER_ALARM".CLIENT.U3_MEAS_STA_MEAS_R.ALARMS.COMPUTER_GET_METHOD_LIST_A AND NOT "DB2120_MPP_ITC_IPC".RESET_FAULTS)) AND "DB7258_UNIT_3_STA_MEAS_A_ENABLE_DISABLE".ENABLED;
   "DB426_ALARMS_WARNINGS".ALARMS.UNIT_03.FACE_R_MEASURING."724299" := "DB16000_OPC_UA_TRIGGER_ALARM".CLIENT.U3_MEAS_STA_MEAS_R.ALARMS.COMPUTER_GET_METHOD_LIST_A;
END_REGION

REGION Network 39: UNIT 3 MEASURING STATION FACE A COMPUTER RELEASE HANDLE LIST ALARM
   RUNG wire#powerrail
      Contact( "DB16255_RLASE_HANDLE_LIST_U3_MEAS_FACE_R".Error )
      wire#w1
      Contact( "DB7258_UNIT_3_STA_MEAS_A_ENABLE_DISABLE".ENABLED )
      wire#w2
      Coil( "DB16000_OPC_UA_TRIGGER_ALARM".CLIENT.U3_MEAS_STA_MEAS_R.ALARMS.COMPUTER_RELEASE_HANDLE_LIST_A )
   END_RUNG
   RUNG wire#powerrail
      Contact( "DB16000_OPC_UA_TRIGGER_ALARM".CLIENT.U3_MEAS_STA_MEAS_R.ALARMS.COMPUTER_RELEASE_HANDLE_LIST_A )
      I_Contact( "DB2120_MPP_ITC_IPC".RESET_FAULTS )
   END_RUNG wire#w1
   RUNG wire#w2
      Coil( "DB426_ALARMS_WARNINGS".ALARMS.UNIT_03.FACE_R_MEASURING."724300" )
   END_RUNG
   // the same network as SCL:
   "DB16000_OPC_UA_TRIGGER_ALARM".CLIENT.U3_MEAS_STA_MEAS_R.ALARMS.COMPUTER_RELEASE_HANDLE_LIST_A := ("DB16255_RLASE_HANDLE_LIST_U3_MEAS_FACE_R".Error OR ("DB16000_OPC_UA_TRIGGER_ALARM".CLIENT.U3_MEAS_STA_MEAS_R.ALARMS.COMPUTER_RELEASE_HANDLE_LIST_A AND NOT "DB2120_MPP_ITC_IPC".RESET_FAULTS)) AND "DB7258_UNIT_3_STA_MEAS_A_ENABLE_DISABLE".ENABLED;
   "DB426_ALARMS_WARNINGS".ALARMS.UNIT_03.FACE_R_MEASURING."724300" := "DB16000_OPC_UA_TRIGGER_ALARM".CLIENT.U3_MEAS_STA_MEAS_R.ALARMS.COMPUTER_RELEASE_HANDLE_LIST_A;
END_REGION

REGION Network 40: UNIT 3 MEASURING STATION FACE A COMPUTER RELEASE METHOD METHOD LIST ALARM
   RUNG wire#powerrail
      Contact( "DB16256_RLASE_METHOD_LIST_U3_MEAS_FACE_R".Error )
      wire#w1
      Contact( "DB7258_UNIT_3_STA_MEAS_A_ENABLE_DISABLE".ENABLED )
      wire#w2
      Coil( "DB16000_OPC_UA_TRIGGER_ALARM".CLIENT.U3_MEAS_STA_MEAS_R.ALARMS.COMPUTER_RELEASE_METHOD_LIST_A )
   END_RUNG
   RUNG wire#powerrail
      Contact( "DB16000_OPC_UA_TRIGGER_ALARM".CLIENT.U3_MEAS_STA_MEAS_R.ALARMS.COMPUTER_RELEASE_METHOD_LIST_A )
      I_Contact( "DB2120_MPP_ITC_IPC".RESET_FAULTS )
   END_RUNG wire#w1
   RUNG wire#w2
      Coil( "DB426_ALARMS_WARNINGS".ALARMS.UNIT_03.FACE_R_MEASURING."724301" )
   END_RUNG
   // the same network as SCL:
   "DB16000_OPC_UA_TRIGGER_ALARM".CLIENT.U3_MEAS_STA_MEAS_R.ALARMS.COMPUTER_RELEASE_METHOD_LIST_A := ("DB16256_RLASE_METHOD_LIST_U3_MEAS_FACE_R".Error OR ("DB16000_OPC_UA_TRIGGER_ALARM".CLIENT.U3_MEAS_STA_MEAS_R.ALARMS.COMPUTER_RELEASE_METHOD_LIST_A AND NOT "DB2120_MPP_ITC_IPC".RESET_FAULTS)) AND "DB7258_UNIT_3_STA_MEAS_A_ENABLE_DISABLE".ENABLED;
   "DB426_ALARMS_WARNINGS".ALARMS.UNIT_03.FACE_R_MEASURING."724301" := "DB16000_OPC_UA_TRIGGER_ALARM".CLIENT.U3_MEAS_STA_MEAS_R.ALARMS.COMPUTER_RELEASE_METHOD_LIST_A;
END_REGION

REGION Network 41: UNIT 3 MEASURING STATION FACE A COMPUTER DISCONNECT ALARM
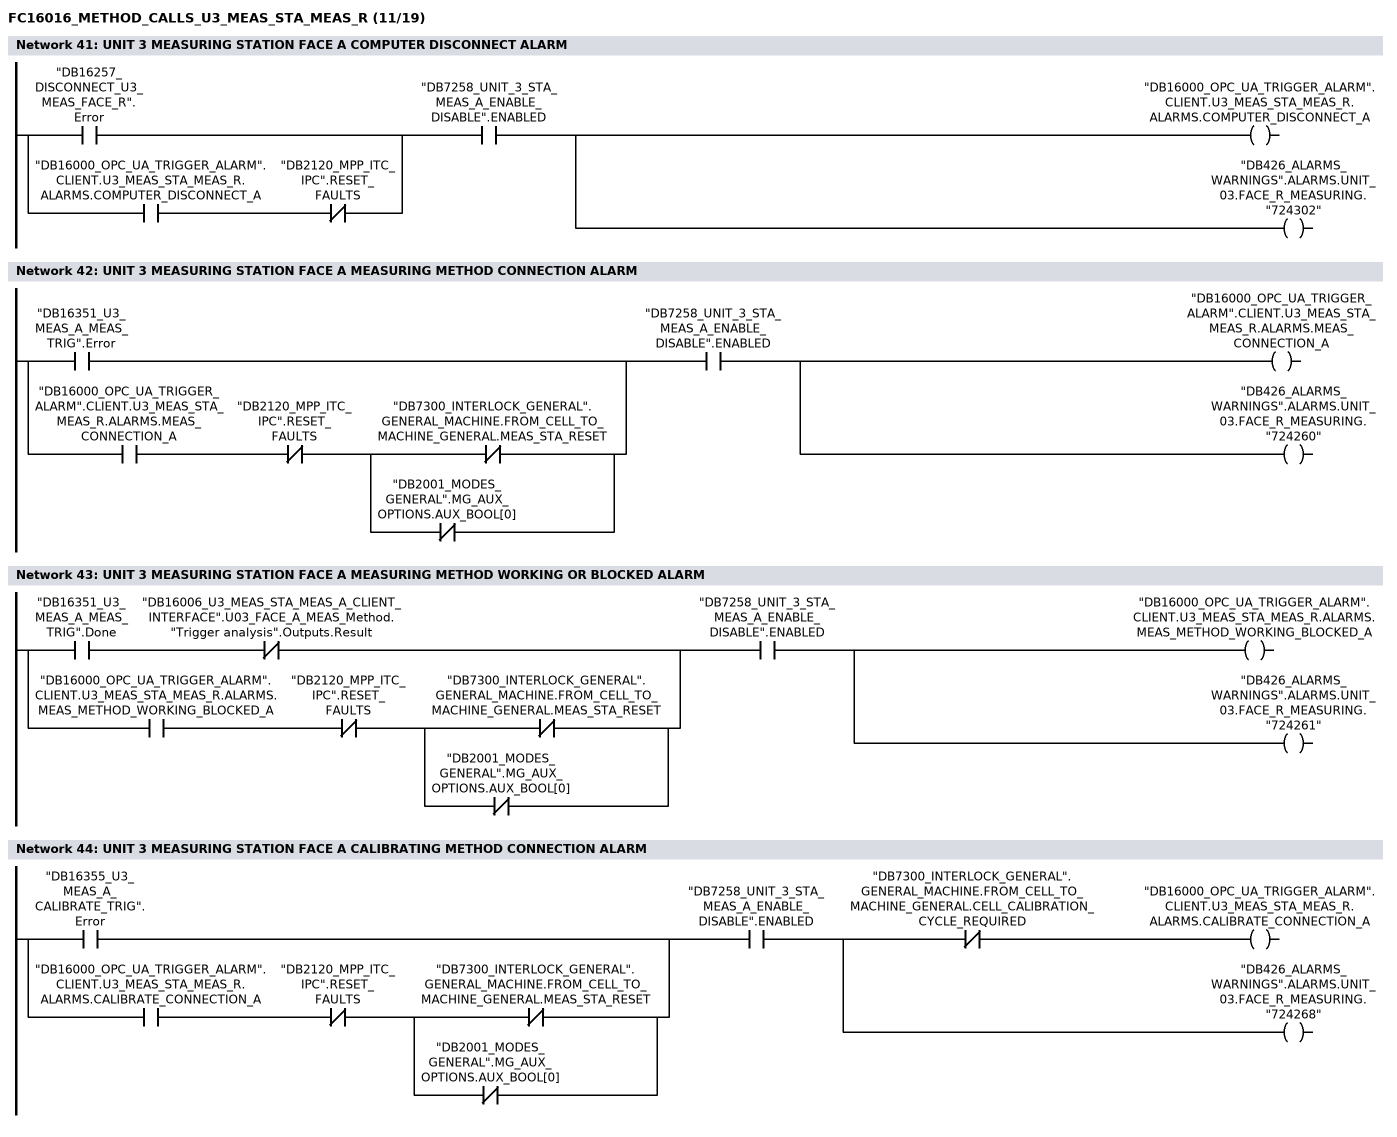
   RUNG wire#powerrail
      Contact( "DB16257_DISCONNECT_U3_MEAS_FACE_R".Error )
      wire#w1
      Contact( "DB7258_UNIT_3_STA_MEAS_A_ENABLE_DISABLE".ENABLED )
      wire#w2
      Coil( "DB16000_OPC_UA_TRIGGER_ALARM".CLIENT.U3_MEAS_STA_MEAS_R.ALARMS.COMPUTER_DISCONNECT_A )
   END_RUNG
   RUNG wire#powerrail
      Contact( "DB16000_OPC_UA_TRIGGER_ALARM".CLIENT.U3_MEAS_STA_MEAS_R.ALARMS.COMPUTER_DISCONNECT_A )
      I_Contact( "DB2120_MPP_ITC_IPC".RESET_FAULTS )
   END_RUNG wire#w1
   RUNG wire#w2
      Coil( "DB426_ALARMS_WARNINGS".ALARMS.UNIT_03.FACE_R_MEASURING."724302" )
   END_RUNG
   // the same network as SCL:
   "DB16000_OPC_UA_TRIGGER_ALARM".CLIENT.U3_MEAS_STA_MEAS_R.ALARMS.COMPUTER_DISCONNECT_A := ("DB16257_DISCONNECT_U3_MEAS_FACE_R".Error OR ("DB16000_OPC_UA_TRIGGER_ALARM".CLIENT.U3_MEAS_STA_MEAS_R.ALARMS.COMPUTER_DISCONNECT_A AND NOT "DB2120_MPP_ITC_IPC".RESET_FAULTS)) AND "DB7258_UNIT_3_STA_MEAS_A_ENABLE_DISABLE".ENABLED;
   "DB426_ALARMS_WARNINGS".ALARMS.UNIT_03.FACE_R_MEASURING."724302" := "DB16000_OPC_UA_TRIGGER_ALARM".CLIENT.U3_MEAS_STA_MEAS_R.ALARMS.COMPUTER_DISCONNECT_A;
END_REGION

REGION Network 42: UNIT 3 MEASURING STATION FACE A MEASURING METHOD CONNECTION ALARM
   RUNG wire#powerrail
      Contact( "DB16351_U3_MEAS_A_MEAS_TRIG".Error )
      wire#w1
      Contact( "DB7258_UNIT_3_STA_MEAS_A_ENABLE_DISABLE".ENABLED )
      wire#w3
      Coil( "DB16000_OPC_UA_TRIGGER_ALARM".CLIENT.U3_MEAS_STA_MEAS_R.ALARMS.MEAS_CONNECTION_A )
   END_RUNG
   RUNG wire#powerrail
      Contact( "DB16000_OPC_UA_TRIGGER_ALARM".CLIENT.U3_MEAS_STA_MEAS_R.ALARMS.MEAS_CONNECTION_A )
      I_Contact( "DB2120_MPP_ITC_IPC".RESET_FAULTS )
      wire#w2
      I_Contact( "DB7300_INTERLOCK_GENERAL".GENERAL_MACHINE.FROM_CELL_TO_MACHINE_GENERAL.MEAS_STA_RESET )
   END_RUNG wire#w1
   RUNG wire#w2
      I_Contact( "DB2001_MODES_GENERAL".MG_AUX_OPTIONS.AUX_BOOL[0] )
   END_RUNG wire#w1
   RUNG wire#w3
      Coil( "DB426_ALARMS_WARNINGS".ALARMS.UNIT_03.FACE_R_MEASURING."724260" )
   END_RUNG
   // the same network as SCL:
   "DB16000_OPC_UA_TRIGGER_ALARM".CLIENT.U3_MEAS_STA_MEAS_R.ALARMS.MEAS_CONNECTION_A := ("DB16351_U3_MEAS_A_MEAS_TRIG".Error OR ("DB16000_OPC_UA_TRIGGER_ALARM".CLIENT.U3_MEAS_STA_MEAS_R.ALARMS.MEAS_CONNECTION_A AND NOT "DB2120_MPP_ITC_IPC".RESET_FAULTS AND (NOT "DB7300_INTERLOCK_GENERAL".GENERAL_MACHINE.FROM_CELL_TO_MACHINE_GENERAL.MEAS_STA_RESET OR NOT "DB2001_MODES_GENERAL".MG_AUX_OPTIONS.AUX_BOOL[0]))) AND "DB7258_UNIT_3_STA_MEAS_A_ENABLE_DISABLE".ENABLED;
   "DB426_ALARMS_WARNINGS".ALARMS.UNIT_03.FACE_R_MEASURING."724260" := "DB16000_OPC_UA_TRIGGER_ALARM".CLIENT.U3_MEAS_STA_MEAS_R.ALARMS.MEAS_CONNECTION_A;
END_REGION

REGION Network 43: UNIT 3 MEASURING STATION FACE A MEASURING METHOD WORKING OR BLOCKED ALARM
   RUNG wire#powerrail
      Contact( "DB16351_U3_MEAS_A_MEAS_TRIG".Done )
      I_Contact( "DB16006_U3_MEAS_STA_MEAS_A_CLIENT_INTERFACE".U03_FACE_A_MEAS_Method."Trigger analysis".Outputs.Result )
      wire#w1
      Contact( "DB7258_UNIT_3_STA_MEAS_A_ENABLE_DISABLE".ENABLED )
      wire#w3
      Coil( "DB16000_OPC_UA_TRIGGER_ALARM".CLIENT.U3_MEAS_STA_MEAS_R.ALARMS.MEAS_METHOD_WORKING_BLOCKED_A )
   END_RUNG
   RUNG wire#powerrail
      Contact( "DB16000_OPC_UA_TRIGGER_ALARM".CLIENT.U3_MEAS_STA_MEAS_R.ALARMS.MEAS_METHOD_WORKING_BLOCKED_A )
      I_Contact( "DB2120_MPP_ITC_IPC".RESET_FAULTS )
      wire#w2
      I_Contact( "DB7300_INTERLOCK_GENERAL".GENERAL_MACHINE.FROM_CELL_TO_MACHINE_GENERAL.MEAS_STA_RESET )
   END_RUNG wire#w1
   RUNG wire#w2
      I_Contact( "DB2001_MODES_GENERAL".MG_AUX_OPTIONS.AUX_BOOL[0] )
   END_RUNG wire#w1
   RUNG wire#w3
      Coil( "DB426_ALARMS_WARNINGS".ALARMS.UNIT_03.FACE_R_MEASURING."724261" )
   END_RUNG
   // the same network as SCL:
   "DB16000_OPC_UA_TRIGGER_ALARM".CLIENT.U3_MEAS_STA_MEAS_R.ALARMS.MEAS_METHOD_WORKING_BLOCKED_A := (("DB16351_U3_MEAS_A_MEAS_TRIG".Done AND NOT "DB16006_U3_MEAS_STA_MEAS_A_CLIENT_INTERFACE".U03_FACE_A_MEAS_Method."Trigger analysis".Outputs.Result) OR ("DB16000_OPC_UA_TRIGGER_ALARM".CLIENT.U3_MEAS_STA_MEAS_R.ALARMS.MEAS_METHOD_WORKING_BLOCKED_A AND NOT "DB2120_MPP_ITC_IPC".RESET_FAULTS AND (NOT "DB7300_INTERLOCK_GENERAL".GENERAL_MACHINE.FROM_CELL_TO_MACHINE_GENERAL.MEAS_STA_RESET OR NOT "DB2001_MODES_GENERAL".MG_AUX_OPTIONS.AUX_BOOL[0]))) AND "DB7258_UNIT_3_STA_MEAS_A_ENABLE_DISABLE".ENABLED;
   "DB426_ALARMS_WARNINGS".ALARMS.UNIT_03.FACE_R_MEASURING."724261" := "DB16000_OPC_UA_TRIGGER_ALARM".CLIENT.U3_MEAS_STA_MEAS_R.ALARMS.MEAS_METHOD_WORKING_BLOCKED_A;
END_REGION

REGION Network 44: UNIT 3 MEASURING STATION FACE A CALIBRATING METHOD CONNECTION ALARM
   RUNG wire#powerrail
      Contact( "DB16355_U3_MEAS_A_CALIBRATE_TRIG".Error )
      wire#w1
      Contact( "DB7258_UNIT_3_STA_MEAS_A_ENABLE_DISABLE".ENABLED )
      wire#w3
      I_Contact( "DB7300_INTERLOCK_GENERAL".GENERAL_MACHINE.FROM_CELL_TO_MACHINE_GENERAL.CELL_CALIBRATION_CYCLE_REQUIRED )
      Coil( "DB16000_OPC_UA_TRIGGER_ALARM".CLIENT.U3_MEAS_STA_MEAS_R.ALARMS.CALIBRATE_CONNECTION_A )
   END_RUNG
   RUNG wire#powerrail
      Contact( "DB16000_OPC_UA_TRIGGER_ALARM".CLIENT.U3_MEAS_STA_MEAS_R.ALARMS.CALIBRATE_CONNECTION_A )
      I_Contact( "DB2120_MPP_ITC_IPC".RESET_FAULTS )
      wire#w2
      I_Contact( "DB7300_INTERLOCK_GENERAL".GENERAL_MACHINE.FROM_CELL_TO_MACHINE_GENERAL.MEAS_STA_RESET )
   END_RUNG wire#w1
   RUNG wire#w2
      I_Contact( "DB2001_MODES_GENERAL".MG_AUX_OPTIONS.AUX_BOOL[0] )
   END_RUNG wire#w1
   RUNG wire#w3
      Coil( "DB426_ALARMS_WARNINGS".ALARMS.UNIT_03.FACE_R_MEASURING."724268" )
   END_RUNG
   // the same network as SCL:
   #_w1 := ("DB16355_U3_MEAS_A_CALIBRATE_TRIG".Error OR ("DB16000_OPC_UA_TRIGGER_ALARM".CLIENT.U3_MEAS_STA_MEAS_R.ALARMS.CALIBRATE_CONNECTION_A AND NOT "DB2120_MPP_ITC_IPC".RESET_FAULTS AND (NOT "DB7300_INTERLOCK_GENERAL".GENERAL_MACHINE.FROM_CELL_TO_MACHINE_GENERAL.MEAS_STA_RESET OR NOT "DB2001_MODES_GENERAL".MG_AUX_OPTIONS.AUX_BOOL[0]))) AND "DB7258_UNIT_3_STA_MEAS_A_ENABLE_DISABLE".ENABLED;
   "DB16000_OPC_UA_TRIGGER_ALARM".CLIENT.U3_MEAS_STA_MEAS_R.ALARMS.CALIBRATE_CONNECTION_A := #_w1 AND NOT "DB7300_INTERLOCK_GENERAL".GENERAL_MACHINE.FROM_CELL_TO_MACHINE_GENERAL.CELL_CALIBRATION_CYCLE_REQUIRED;
   "DB426_ALARMS_WARNINGS".ALARMS.UNIT_03.FACE_R_MEASURING."724268" := #_w1;
END_REGION

REGION Network 45: UNIT 3 MEASURING STATION FACE A CALIBRATING METHOD WORKING OR BLOCKED ALARM
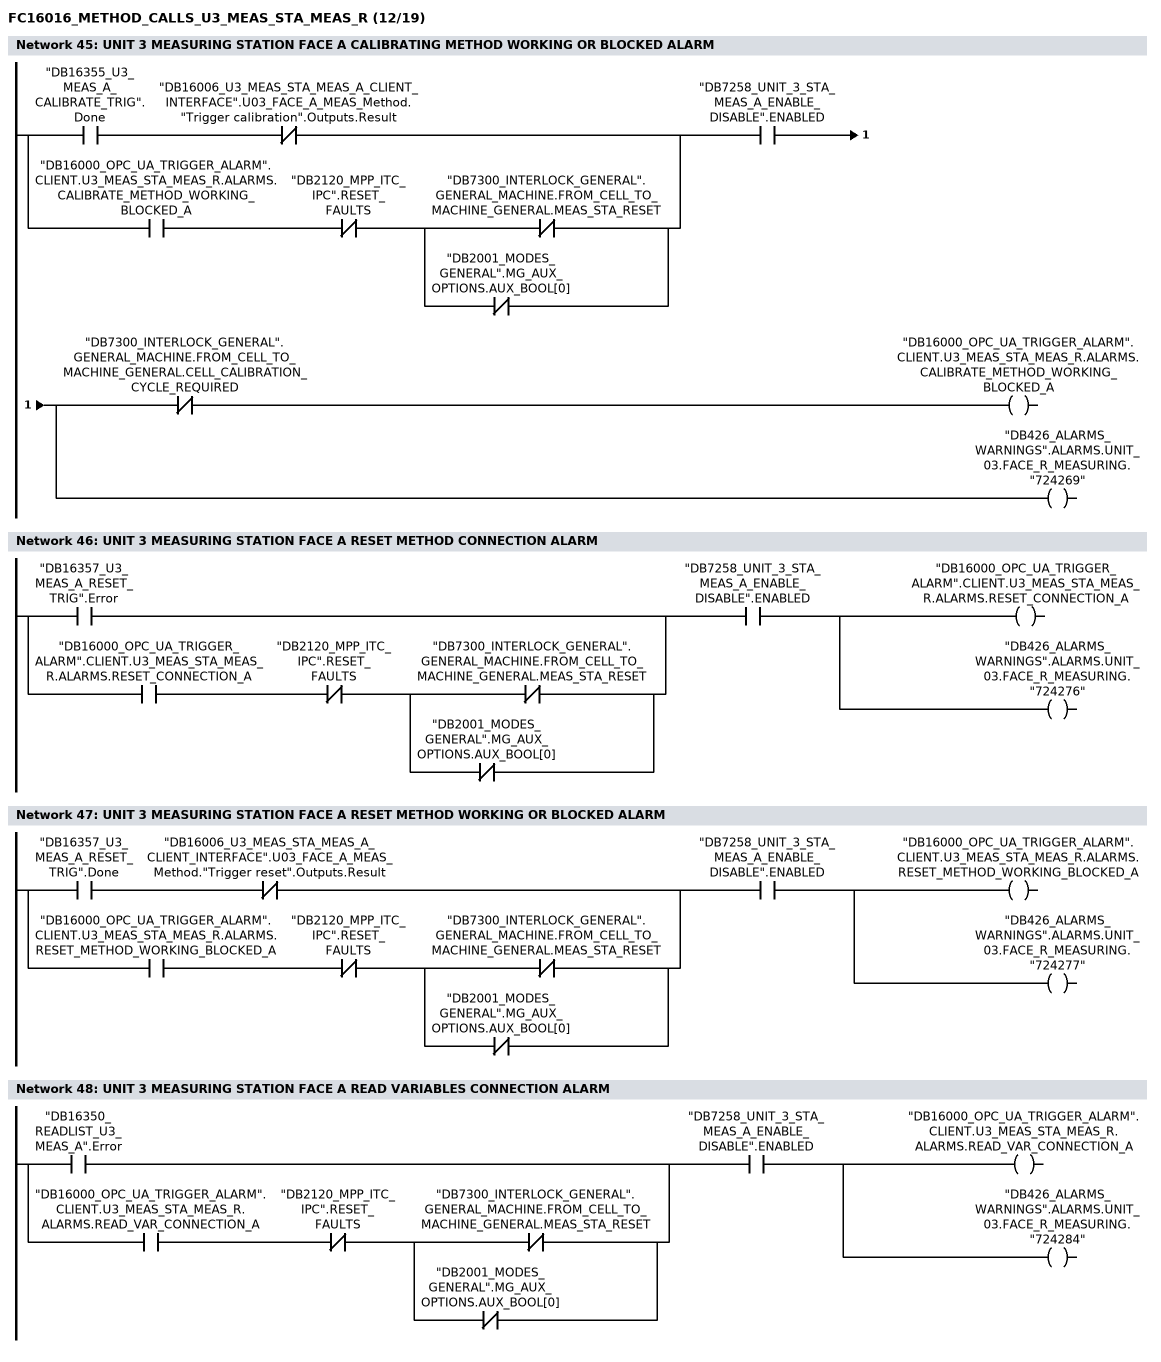
   RUNG wire#powerrail
      Contact( "DB16355_U3_MEAS_A_CALIBRATE_TRIG".Done )
      I_Contact( "DB16006_U3_MEAS_STA_MEAS_A_CLIENT_INTERFACE".U03_FACE_A_MEAS_Method."Trigger calibration".Outputs.Result )
      wire#w1
      Contact( "DB7258_UNIT_3_STA_MEAS_A_ENABLE_DISABLE".ENABLED )
      wire#w3
      I_Contact( "DB7300_INTERLOCK_GENERAL".GENERAL_MACHINE.FROM_CELL_TO_MACHINE_GENERAL.CELL_CALIBRATION_CYCLE_REQUIRED )
      Coil( "DB16000_OPC_UA_TRIGGER_ALARM".CLIENT.U3_MEAS_STA_MEAS_R.ALARMS.CALIBRATE_METHOD_WORKING_BLOCKED_A )
   END_RUNG
   RUNG wire#powerrail
      Contact( "DB16000_OPC_UA_TRIGGER_ALARM".CLIENT.U3_MEAS_STA_MEAS_R.ALARMS.CALIBRATE_METHOD_WORKING_BLOCKED_A )
      I_Contact( "DB2120_MPP_ITC_IPC".RESET_FAULTS )
      wire#w2
      I_Contact( "DB7300_INTERLOCK_GENERAL".GENERAL_MACHINE.FROM_CELL_TO_MACHINE_GENERAL.MEAS_STA_RESET )
   END_RUNG wire#w1
   RUNG wire#w2
      I_Contact( "DB2001_MODES_GENERAL".MG_AUX_OPTIONS.AUX_BOOL[0] )
   END_RUNG wire#w1
   RUNG wire#w3
      Coil( "DB426_ALARMS_WARNINGS".ALARMS.UNIT_03.FACE_R_MEASURING."724269" )
   END_RUNG
   // the same network as SCL:
   #_w1 := (("DB16355_U3_MEAS_A_CALIBRATE_TRIG".Done AND NOT "DB16006_U3_MEAS_STA_MEAS_A_CLIENT_INTERFACE".U03_FACE_A_MEAS_Method."Trigger calibration".Outputs.Result) OR ("DB16000_OPC_UA_TRIGGER_ALARM".CLIENT.U3_MEAS_STA_MEAS_R.ALARMS.CALIBRATE_METHOD_WORKING_BLOCKED_A AND NOT "DB2120_MPP_ITC_IPC".RESET_FAULTS AND (NOT "DB7300_INTERLOCK_GENERAL".GENERAL_MACHINE.FROM_CELL_TO_MACHINE_GENERAL.MEAS_STA_RESET OR NOT "DB2001_MODES_GENERAL".MG_AUX_OPTIONS.AUX_BOOL[0]))) AND "DB7258_UNIT_3_STA_MEAS_A_ENABLE_DISABLE".ENABLED;
   "DB16000_OPC_UA_TRIGGER_ALARM".CLIENT.U3_MEAS_STA_MEAS_R.ALARMS.CALIBRATE_METHOD_WORKING_BLOCKED_A := #_w1 AND NOT "DB7300_INTERLOCK_GENERAL".GENERAL_MACHINE.FROM_CELL_TO_MACHINE_GENERAL.CELL_CALIBRATION_CYCLE_REQUIRED;
   "DB426_ALARMS_WARNINGS".ALARMS.UNIT_03.FACE_R_MEASURING."724269" := #_w1;
END_REGION

REGION Network 46: UNIT 3 MEASURING STATION FACE A RESET METHOD CONNECTION ALARM
   RUNG wire#powerrail
      Contact( "DB16357_U3_MEAS_A_RESET_TRIG".Error )
      wire#w1
      Contact( "DB7258_UNIT_3_STA_MEAS_A_ENABLE_DISABLE".ENABLED )
      wire#w3
      Coil( "DB16000_OPC_UA_TRIGGER_ALARM".CLIENT.U3_MEAS_STA_MEAS_R.ALARMS.RESET_CONNECTION_A )
   END_RUNG
   RUNG wire#powerrail
      Contact( "DB16000_OPC_UA_TRIGGER_ALARM".CLIENT.U3_MEAS_STA_MEAS_R.ALARMS.RESET_CONNECTION_A )
      I_Contact( "DB2120_MPP_ITC_IPC".RESET_FAULTS )
      wire#w2
      I_Contact( "DB7300_INTERLOCK_GENERAL".GENERAL_MACHINE.FROM_CELL_TO_MACHINE_GENERAL.MEAS_STA_RESET )
   END_RUNG wire#w1
   RUNG wire#w2
      I_Contact( "DB2001_MODES_GENERAL".MG_AUX_OPTIONS.AUX_BOOL[0] )
   END_RUNG wire#w1
   RUNG wire#w3
      Coil( "DB426_ALARMS_WARNINGS".ALARMS.UNIT_03.FACE_R_MEASURING."724276" )
   END_RUNG
   // the same network as SCL:
   "DB16000_OPC_UA_TRIGGER_ALARM".CLIENT.U3_MEAS_STA_MEAS_R.ALARMS.RESET_CONNECTION_A := ("DB16357_U3_MEAS_A_RESET_TRIG".Error OR ("DB16000_OPC_UA_TRIGGER_ALARM".CLIENT.U3_MEAS_STA_MEAS_R.ALARMS.RESET_CONNECTION_A AND NOT "DB2120_MPP_ITC_IPC".RESET_FAULTS AND (NOT "DB7300_INTERLOCK_GENERAL".GENERAL_MACHINE.FROM_CELL_TO_MACHINE_GENERAL.MEAS_STA_RESET OR NOT "DB2001_MODES_GENERAL".MG_AUX_OPTIONS.AUX_BOOL[0]))) AND "DB7258_UNIT_3_STA_MEAS_A_ENABLE_DISABLE".ENABLED;
   "DB426_ALARMS_WARNINGS".ALARMS.UNIT_03.FACE_R_MEASURING."724276" := "DB16000_OPC_UA_TRIGGER_ALARM".CLIENT.U3_MEAS_STA_MEAS_R.ALARMS.RESET_CONNECTION_A;
END_REGION

REGION Network 47: UNIT 3 MEASURING STATION FACE A RESET METHOD WORKING OR BLOCKED ALARM
   RUNG wire#powerrail
      Contact( "DB16357_U3_MEAS_A_RESET_TRIG".Done )
      I_Contact( "DB16006_U3_MEAS_STA_MEAS_A_CLIENT_INTERFACE".U03_FACE_A_MEAS_Method."Trigger reset".Outputs.Result )
      wire#w1
      Contact( "DB7258_UNIT_3_STA_MEAS_A_ENABLE_DISABLE".ENABLED )
      wire#w3
      Coil( "DB16000_OPC_UA_TRIGGER_ALARM".CLIENT.U3_MEAS_STA_MEAS_R.ALARMS.RESET_METHOD_WORKING_BLOCKED_A )
   END_RUNG
   RUNG wire#powerrail
      Contact( "DB16000_OPC_UA_TRIGGER_ALARM".CLIENT.U3_MEAS_STA_MEAS_R.ALARMS.RESET_METHOD_WORKING_BLOCKED_A )
      I_Contact( "DB2120_MPP_ITC_IPC".RESET_FAULTS )
      wire#w2
      I_Contact( "DB7300_INTERLOCK_GENERAL".GENERAL_MACHINE.FROM_CELL_TO_MACHINE_GENERAL.MEAS_STA_RESET )
   END_RUNG wire#w1
   RUNG wire#w2
      I_Contact( "DB2001_MODES_GENERAL".MG_AUX_OPTIONS.AUX_BOOL[0] )
   END_RUNG wire#w1
   RUNG wire#w3
      Coil( "DB426_ALARMS_WARNINGS".ALARMS.UNIT_03.FACE_R_MEASURING."724277" )
   END_RUNG
   // the same network as SCL:
   "DB16000_OPC_UA_TRIGGER_ALARM".CLIENT.U3_MEAS_STA_MEAS_R.ALARMS.RESET_METHOD_WORKING_BLOCKED_A := (("DB16357_U3_MEAS_A_RESET_TRIG".Done AND NOT "DB16006_U3_MEAS_STA_MEAS_A_CLIENT_INTERFACE".U03_FACE_A_MEAS_Method."Trigger reset".Outputs.Result) OR ("DB16000_OPC_UA_TRIGGER_ALARM".CLIENT.U3_MEAS_STA_MEAS_R.ALARMS.RESET_METHOD_WORKING_BLOCKED_A AND NOT "DB2120_MPP_ITC_IPC".RESET_FAULTS AND (NOT "DB7300_INTERLOCK_GENERAL".GENERAL_MACHINE.FROM_CELL_TO_MACHINE_GENERAL.MEAS_STA_RESET OR NOT "DB2001_MODES_GENERAL".MG_AUX_OPTIONS.AUX_BOOL[0]))) AND "DB7258_UNIT_3_STA_MEAS_A_ENABLE_DISABLE".ENABLED;
   "DB426_ALARMS_WARNINGS".ALARMS.UNIT_03.FACE_R_MEASURING."724277" := "DB16000_OPC_UA_TRIGGER_ALARM".CLIENT.U3_MEAS_STA_MEAS_R.ALARMS.RESET_METHOD_WORKING_BLOCKED_A;
END_REGION

REGION Network 48: UNIT 3 MEASURING STATION FACE A READ VARIABLES CONNECTION ALARM
   RUNG wire#powerrail
      Contact( "DB16350_READLIST_U3_MEAS_A".Error )
      wire#w1
      Contact( "DB7258_UNIT_3_STA_MEAS_A_ENABLE_DISABLE".ENABLED )
      wire#w3
      Coil( "DB16000_OPC_UA_TRIGGER_ALARM".CLIENT.U3_MEAS_STA_MEAS_R.ALARMS.READ_VAR_CONNECTION_A )
   END_RUNG
   RUNG wire#powerrail
      Contact( "DB16000_OPC_UA_TRIGGER_ALARM".CLIENT.U3_MEAS_STA_MEAS_R.ALARMS.READ_VAR_CONNECTION_A )
      I_Contact( "DB2120_MPP_ITC_IPC".RESET_FAULTS )
      wire#w2
      I_Contact( "DB7300_INTERLOCK_GENERAL".GENERAL_MACHINE.FROM_CELL_TO_MACHINE_GENERAL.MEAS_STA_RESET )
   END_RUNG wire#w1
   RUNG wire#w2
      I_Contact( "DB2001_MODES_GENERAL".MG_AUX_OPTIONS.AUX_BOOL[0] )
   END_RUNG wire#w1
   RUNG wire#w3
      Coil( "DB426_ALARMS_WARNINGS".ALARMS.UNIT_03.FACE_R_MEASURING."724284" )
   END_RUNG
   // the same network as SCL:
   "DB16000_OPC_UA_TRIGGER_ALARM".CLIENT.U3_MEAS_STA_MEAS_R.ALARMS.READ_VAR_CONNECTION_A := ("DB16350_READLIST_U3_MEAS_A".Error OR ("DB16000_OPC_UA_TRIGGER_ALARM".CLIENT.U3_MEAS_STA_MEAS_R.ALARMS.READ_VAR_CONNECTION_A AND NOT "DB2120_MPP_ITC_IPC".RESET_FAULTS AND (NOT "DB7300_INTERLOCK_GENERAL".GENERAL_MACHINE.FROM_CELL_TO_MACHINE_GENERAL.MEAS_STA_RESET OR NOT "DB2001_MODES_GENERAL".MG_AUX_OPTIONS.AUX_BOOL[0]))) AND "DB7258_UNIT_3_STA_MEAS_A_ENABLE_DISABLE".ENABLED;
   "DB426_ALARMS_WARNINGS".ALARMS.UNIT_03.FACE_R_MEASURING."724284" := "DB16000_OPC_UA_TRIGGER_ALARM".CLIENT.U3_MEAS_STA_MEAS_R.ALARMS.READ_VAR_CONNECTION_A;
END_REGION

REGION Network 49: UNIT 3 MEASURING STATION FACE A READ VARIABLES WORKING OR BLOCKED ALARM
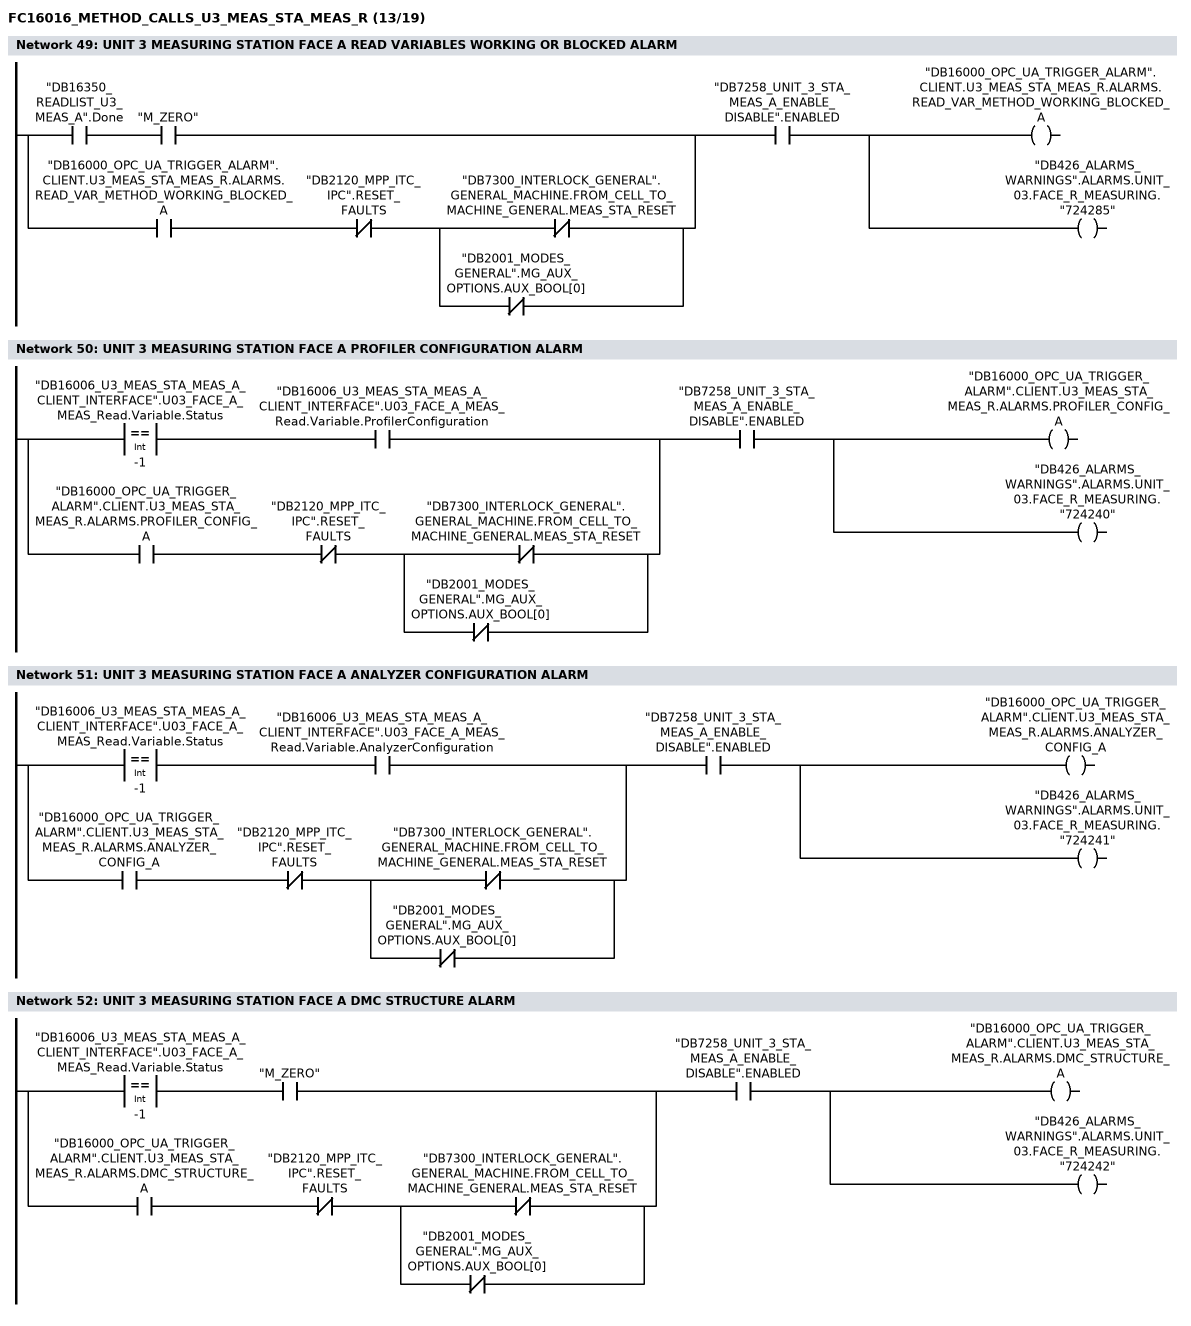
   RUNG wire#powerrail
      Contact( "DB16350_READLIST_U3_MEAS_A".Done )
      Contact( "M_ZERO" )
      wire#w1
      Contact( "DB7258_UNIT_3_STA_MEAS_A_ENABLE_DISABLE".ENABLED )
      wire#w3
      Coil( "DB16000_OPC_UA_TRIGGER_ALARM".CLIENT.U3_MEAS_STA_MEAS_R.ALARMS.READ_VAR_METHOD_WORKING_BLOCKED_A )
   END_RUNG
   RUNG wire#powerrail
      Contact( "DB16000_OPC_UA_TRIGGER_ALARM".CLIENT.U3_MEAS_STA_MEAS_R.ALARMS.READ_VAR_METHOD_WORKING_BLOCKED_A )
      I_Contact( "DB2120_MPP_ITC_IPC".RESET_FAULTS )
      wire#w2
      I_Contact( "DB7300_INTERLOCK_GENERAL".GENERAL_MACHINE.FROM_CELL_TO_MACHINE_GENERAL.MEAS_STA_RESET )
   END_RUNG wire#w1
   RUNG wire#w2
      I_Contact( "DB2001_MODES_GENERAL".MG_AUX_OPTIONS.AUX_BOOL[0] )
   END_RUNG wire#w1
   RUNG wire#w3
      Coil( "DB426_ALARMS_WARNINGS".ALARMS.UNIT_03.FACE_R_MEASURING."724285" )
   END_RUNG
   // the same network as SCL:
   "DB16000_OPC_UA_TRIGGER_ALARM".CLIENT.U3_MEAS_STA_MEAS_R.ALARMS.READ_VAR_METHOD_WORKING_BLOCKED_A := (("DB16350_READLIST_U3_MEAS_A".Done AND "M_ZERO") OR ("DB16000_OPC_UA_TRIGGER_ALARM".CLIENT.U3_MEAS_STA_MEAS_R.ALARMS.READ_VAR_METHOD_WORKING_BLOCKED_A AND NOT "DB2120_MPP_ITC_IPC".RESET_FAULTS AND (NOT "DB7300_INTERLOCK_GENERAL".GENERAL_MACHINE.FROM_CELL_TO_MACHINE_GENERAL.MEAS_STA_RESET OR NOT "DB2001_MODES_GENERAL".MG_AUX_OPTIONS.AUX_BOOL[0]))) AND "DB7258_UNIT_3_STA_MEAS_A_ENABLE_DISABLE".ENABLED;
   "DB426_ALARMS_WARNINGS".ALARMS.UNIT_03.FACE_R_MEASURING."724285" := "DB16000_OPC_UA_TRIGGER_ALARM".CLIENT.U3_MEAS_STA_MEAS_R.ALARMS.READ_VAR_METHOD_WORKING_BLOCKED_A;
END_REGION

REGION Network 50: UNIT 3 MEASURING STATION FACE A PROFILER CONFIGURATION ALARM
   RUNG wire#powerrail
      { S7_Templates := "SrcType := Int" } EQ_Contact(in1 := "DB16006_U3_MEAS_STA_MEAS_A_CLIENT_INTERFACE".U03_FACE_A_MEAS_Read.Variable.Status, in2 := -1)
      Contact( "DB16006_U3_MEAS_STA_MEAS_A_CLIENT_INTERFACE".U03_FACE_A_MEAS_Read.Variable.ProfilerConfiguration )
      wire#w1
      Contact( "DB7258_UNIT_3_STA_MEAS_A_ENABLE_DISABLE".ENABLED )
      wire#w3
      Coil( "DB16000_OPC_UA_TRIGGER_ALARM".CLIENT.U3_MEAS_STA_MEAS_R.ALARMS.PROFILER_CONFIG_A )
   END_RUNG
   RUNG wire#powerrail
      Contact( "DB16000_OPC_UA_TRIGGER_ALARM".CLIENT.U3_MEAS_STA_MEAS_R.ALARMS.PROFILER_CONFIG_A )
      I_Contact( "DB2120_MPP_ITC_IPC".RESET_FAULTS )
      wire#w2
      I_Contact( "DB7300_INTERLOCK_GENERAL".GENERAL_MACHINE.FROM_CELL_TO_MACHINE_GENERAL.MEAS_STA_RESET )
   END_RUNG wire#w1
   RUNG wire#w2
      I_Contact( "DB2001_MODES_GENERAL".MG_AUX_OPTIONS.AUX_BOOL[0] )
   END_RUNG wire#w1
   RUNG wire#w3
      Coil( "DB426_ALARMS_WARNINGS".ALARMS.UNIT_03.FACE_R_MEASURING."724240" )
   END_RUNG
   // the same network as SCL:
   "DB16000_OPC_UA_TRIGGER_ALARM".CLIENT.U3_MEAS_STA_MEAS_R.ALARMS.PROFILER_CONFIG_A := ((("DB16006_U3_MEAS_STA_MEAS_A_CLIENT_INTERFACE".U03_FACE_A_MEAS_Read.Variable.Status = (-1)) AND "DB16006_U3_MEAS_STA_MEAS_A_CLIENT_INTERFACE".U03_FACE_A_MEAS_Read.Variable.ProfilerConfiguration) OR ("DB16000_OPC_UA_TRIGGER_ALARM".CLIENT.U3_MEAS_STA_MEAS_R.ALARMS.PROFILER_CONFIG_A AND NOT "DB2120_MPP_ITC_IPC".RESET_FAULTS AND (NOT "DB7300_INTERLOCK_GENERAL".GENERAL_MACHINE.FROM_CELL_TO_MACHINE_GENERAL.MEAS_STA_RESET OR NOT "DB2001_MODES_GENERAL".MG_AUX_OPTIONS.AUX_BOOL[0]))) AND "DB7258_UNIT_3_STA_MEAS_A_ENABLE_DISABLE".ENABLED;
   "DB426_ALARMS_WARNINGS".ALARMS.UNIT_03.FACE_R_MEASURING."724240" := "DB16000_OPC_UA_TRIGGER_ALARM".CLIENT.U3_MEAS_STA_MEAS_R.ALARMS.PROFILER_CONFIG_A;
END_REGION

REGION Network 51: UNIT 3 MEASURING STATION FACE A ANALYZER CONFIGURATION ALARM
   RUNG wire#powerrail
      { S7_Templates := "SrcType := Int" } EQ_Contact(in1 := "DB16006_U3_MEAS_STA_MEAS_A_CLIENT_INTERFACE".U03_FACE_A_MEAS_Read.Variable.Status, in2 := -1)
      Contact( "DB16006_U3_MEAS_STA_MEAS_A_CLIENT_INTERFACE".U03_FACE_A_MEAS_Read.Variable.AnalyzerConfiguration )
      wire#w1
      Contact( "DB7258_UNIT_3_STA_MEAS_A_ENABLE_DISABLE".ENABLED )
      wire#w3
      Coil( "DB16000_OPC_UA_TRIGGER_ALARM".CLIENT.U3_MEAS_STA_MEAS_R.ALARMS.ANALYZER_CONFIG_A )
   END_RUNG
   RUNG wire#powerrail
      Contact( "DB16000_OPC_UA_TRIGGER_ALARM".CLIENT.U3_MEAS_STA_MEAS_R.ALARMS.ANALYZER_CONFIG_A )
      I_Contact( "DB2120_MPP_ITC_IPC".RESET_FAULTS )
      wire#w2
      I_Contact( "DB7300_INTERLOCK_GENERAL".GENERAL_MACHINE.FROM_CELL_TO_MACHINE_GENERAL.MEAS_STA_RESET )
   END_RUNG wire#w1
   RUNG wire#w2
      I_Contact( "DB2001_MODES_GENERAL".MG_AUX_OPTIONS.AUX_BOOL[0] )
   END_RUNG wire#w1
   RUNG wire#w3
      Coil( "DB426_ALARMS_WARNINGS".ALARMS.UNIT_03.FACE_R_MEASURING."724241" )
   END_RUNG
   // the same network as SCL:
   "DB16000_OPC_UA_TRIGGER_ALARM".CLIENT.U3_MEAS_STA_MEAS_R.ALARMS.ANALYZER_CONFIG_A := ((("DB16006_U3_MEAS_STA_MEAS_A_CLIENT_INTERFACE".U03_FACE_A_MEAS_Read.Variable.Status = (-1)) AND "DB16006_U3_MEAS_STA_MEAS_A_CLIENT_INTERFACE".U03_FACE_A_MEAS_Read.Variable.AnalyzerConfiguration) OR ("DB16000_OPC_UA_TRIGGER_ALARM".CLIENT.U3_MEAS_STA_MEAS_R.ALARMS.ANALYZER_CONFIG_A AND NOT "DB2120_MPP_ITC_IPC".RESET_FAULTS AND (NOT "DB7300_INTERLOCK_GENERAL".GENERAL_MACHINE.FROM_CELL_TO_MACHINE_GENERAL.MEAS_STA_RESET OR NOT "DB2001_MODES_GENERAL".MG_AUX_OPTIONS.AUX_BOOL[0]))) AND "DB7258_UNIT_3_STA_MEAS_A_ENABLE_DISABLE".ENABLED;
   "DB426_ALARMS_WARNINGS".ALARMS.UNIT_03.FACE_R_MEASURING."724241" := "DB16000_OPC_UA_TRIGGER_ALARM".CLIENT.U3_MEAS_STA_MEAS_R.ALARMS.ANALYZER_CONFIG_A;
END_REGION

REGION Network 52: UNIT 3 MEASURING STATION FACE A DMC STRUCTURE ALARM
   RUNG wire#powerrail
      { S7_Templates := "SrcType := Int" } EQ_Contact(in1 := "DB16006_U3_MEAS_STA_MEAS_A_CLIENT_INTERFACE".U03_FACE_A_MEAS_Read.Variable.Status, in2 := -1)
      Contact( "M_ZERO" )
      wire#w1
      Contact( "DB7258_UNIT_3_STA_MEAS_A_ENABLE_DISABLE".ENABLED )
      wire#w3
      Coil( "DB16000_OPC_UA_TRIGGER_ALARM".CLIENT.U3_MEAS_STA_MEAS_R.ALARMS.DMC_STRUCTURE_A )
   END_RUNG
   RUNG wire#powerrail
      Contact( "DB16000_OPC_UA_TRIGGER_ALARM".CLIENT.U3_MEAS_STA_MEAS_R.ALARMS.DMC_STRUCTURE_A )
      I_Contact( "DB2120_MPP_ITC_IPC".RESET_FAULTS )
      wire#w2
      I_Contact( "DB7300_INTERLOCK_GENERAL".GENERAL_MACHINE.FROM_CELL_TO_MACHINE_GENERAL.MEAS_STA_RESET )
   END_RUNG wire#w1
   RUNG wire#w2
      I_Contact( "DB2001_MODES_GENERAL".MG_AUX_OPTIONS.AUX_BOOL[0] )
   END_RUNG wire#w1
   RUNG wire#w3
      Coil( "DB426_ALARMS_WARNINGS".ALARMS.UNIT_03.FACE_R_MEASURING."724242" )
   END_RUNG
   // the same network as SCL:
   "DB16000_OPC_UA_TRIGGER_ALARM".CLIENT.U3_MEAS_STA_MEAS_R.ALARMS.DMC_STRUCTURE_A := ((("DB16006_U3_MEAS_STA_MEAS_A_CLIENT_INTERFACE".U03_FACE_A_MEAS_Read.Variable.Status = (-1)) AND "M_ZERO") OR ("DB16000_OPC_UA_TRIGGER_ALARM".CLIENT.U3_MEAS_STA_MEAS_R.ALARMS.DMC_STRUCTURE_A AND NOT "DB2120_MPP_ITC_IPC".RESET_FAULTS AND (NOT "DB7300_INTERLOCK_GENERAL".GENERAL_MACHINE.FROM_CELL_TO_MACHINE_GENERAL.MEAS_STA_RESET OR NOT "DB2001_MODES_GENERAL".MG_AUX_OPTIONS.AUX_BOOL[0]))) AND "DB7258_UNIT_3_STA_MEAS_A_ENABLE_DISABLE".ENABLED;
   "DB426_ALARMS_WARNINGS".ALARMS.UNIT_03.FACE_R_MEASURING."724242" := "DB16000_OPC_UA_TRIGGER_ALARM".CLIENT.U3_MEAS_STA_MEAS_R.ALARMS.DMC_STRUCTURE_A;
END_REGION

REGION Network 53: UNIT 3 MEASURING STATION FACE A ACQUISITON ALARM
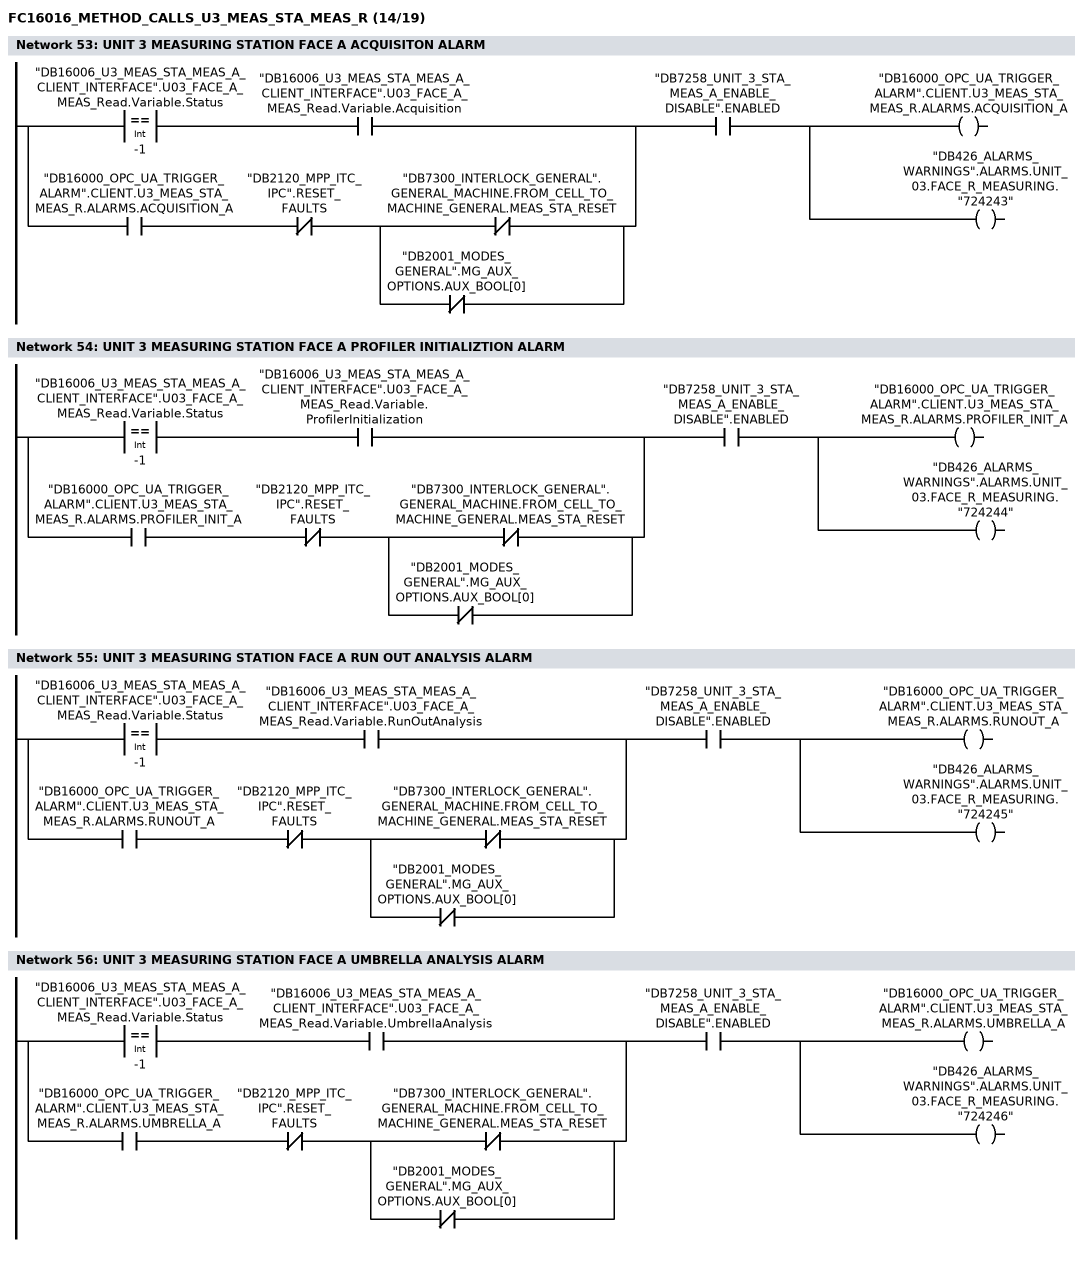
   RUNG wire#powerrail
      { S7_Templates := "SrcType := Int" } EQ_Contact(in1 := "DB16006_U3_MEAS_STA_MEAS_A_CLIENT_INTERFACE".U03_FACE_A_MEAS_Read.Variable.Status, in2 := -1)
      Contact( "DB16006_U3_MEAS_STA_MEAS_A_CLIENT_INTERFACE".U03_FACE_A_MEAS_Read.Variable.Acquisition )
      wire#w1
      Contact( "DB7258_UNIT_3_STA_MEAS_A_ENABLE_DISABLE".ENABLED )
      wire#w3
      Coil( "DB16000_OPC_UA_TRIGGER_ALARM".CLIENT.U3_MEAS_STA_MEAS_R.ALARMS.ACQUISITION_A )
   END_RUNG
   RUNG wire#powerrail
      Contact( "DB16000_OPC_UA_TRIGGER_ALARM".CLIENT.U3_MEAS_STA_MEAS_R.ALARMS.ACQUISITION_A )
      I_Contact( "DB2120_MPP_ITC_IPC".RESET_FAULTS )
      wire#w2
      I_Contact( "DB7300_INTERLOCK_GENERAL".GENERAL_MACHINE.FROM_CELL_TO_MACHINE_GENERAL.MEAS_STA_RESET )
   END_RUNG wire#w1
   RUNG wire#w2
      I_Contact( "DB2001_MODES_GENERAL".MG_AUX_OPTIONS.AUX_BOOL[0] )
   END_RUNG wire#w1
   RUNG wire#w3
      Coil( "DB426_ALARMS_WARNINGS".ALARMS.UNIT_03.FACE_R_MEASURING."724243" )
   END_RUNG
   // the same network as SCL:
   "DB16000_OPC_UA_TRIGGER_ALARM".CLIENT.U3_MEAS_STA_MEAS_R.ALARMS.ACQUISITION_A := ((("DB16006_U3_MEAS_STA_MEAS_A_CLIENT_INTERFACE".U03_FACE_A_MEAS_Read.Variable.Status = (-1)) AND "DB16006_U3_MEAS_STA_MEAS_A_CLIENT_INTERFACE".U03_FACE_A_MEAS_Read.Variable.Acquisition) OR ("DB16000_OPC_UA_TRIGGER_ALARM".CLIENT.U3_MEAS_STA_MEAS_R.ALARMS.ACQUISITION_A AND NOT "DB2120_MPP_ITC_IPC".RESET_FAULTS AND (NOT "DB7300_INTERLOCK_GENERAL".GENERAL_MACHINE.FROM_CELL_TO_MACHINE_GENERAL.MEAS_STA_RESET OR NOT "DB2001_MODES_GENERAL".MG_AUX_OPTIONS.AUX_BOOL[0]))) AND "DB7258_UNIT_3_STA_MEAS_A_ENABLE_DISABLE".ENABLED;
   "DB426_ALARMS_WARNINGS".ALARMS.UNIT_03.FACE_R_MEASURING."724243" := "DB16000_OPC_UA_TRIGGER_ALARM".CLIENT.U3_MEAS_STA_MEAS_R.ALARMS.ACQUISITION_A;
END_REGION

REGION Network 54: UNIT 3 MEASURING STATION FACE A PROFILER INITIALIZTION ALARM
   RUNG wire#powerrail
      { S7_Templates := "SrcType := Int" } EQ_Contact(in1 := "DB16006_U3_MEAS_STA_MEAS_A_CLIENT_INTERFACE".U03_FACE_A_MEAS_Read.Variable.Status, in2 := -1)
      Contact( "DB16006_U3_MEAS_STA_MEAS_A_CLIENT_INTERFACE".U03_FACE_A_MEAS_Read.Variable.ProfilerInitialization )
      wire#w1
      Contact( "DB7258_UNIT_3_STA_MEAS_A_ENABLE_DISABLE".ENABLED )
      wire#w3
      Coil( "DB16000_OPC_UA_TRIGGER_ALARM".CLIENT.U3_MEAS_STA_MEAS_R.ALARMS.PROFILER_INIT_A )
   END_RUNG
   RUNG wire#powerrail
      Contact( "DB16000_OPC_UA_TRIGGER_ALARM".CLIENT.U3_MEAS_STA_MEAS_R.ALARMS.PROFILER_INIT_A )
      I_Contact( "DB2120_MPP_ITC_IPC".RESET_FAULTS )
      wire#w2
      I_Contact( "DB7300_INTERLOCK_GENERAL".GENERAL_MACHINE.FROM_CELL_TO_MACHINE_GENERAL.MEAS_STA_RESET )
   END_RUNG wire#w1
   RUNG wire#w2
      I_Contact( "DB2001_MODES_GENERAL".MG_AUX_OPTIONS.AUX_BOOL[0] )
   END_RUNG wire#w1
   RUNG wire#w3
      Coil( "DB426_ALARMS_WARNINGS".ALARMS.UNIT_03.FACE_R_MEASURING."724244" )
   END_RUNG
   // the same network as SCL:
   "DB16000_OPC_UA_TRIGGER_ALARM".CLIENT.U3_MEAS_STA_MEAS_R.ALARMS.PROFILER_INIT_A := ((("DB16006_U3_MEAS_STA_MEAS_A_CLIENT_INTERFACE".U03_FACE_A_MEAS_Read.Variable.Status = (-1)) AND "DB16006_U3_MEAS_STA_MEAS_A_CLIENT_INTERFACE".U03_FACE_A_MEAS_Read.Variable.ProfilerInitialization) OR ("DB16000_OPC_UA_TRIGGER_ALARM".CLIENT.U3_MEAS_STA_MEAS_R.ALARMS.PROFILER_INIT_A AND NOT "DB2120_MPP_ITC_IPC".RESET_FAULTS AND (NOT "DB7300_INTERLOCK_GENERAL".GENERAL_MACHINE.FROM_CELL_TO_MACHINE_GENERAL.MEAS_STA_RESET OR NOT "DB2001_MODES_GENERAL".MG_AUX_OPTIONS.AUX_BOOL[0]))) AND "DB7258_UNIT_3_STA_MEAS_A_ENABLE_DISABLE".ENABLED;
   "DB426_ALARMS_WARNINGS".ALARMS.UNIT_03.FACE_R_MEASURING."724244" := "DB16000_OPC_UA_TRIGGER_ALARM".CLIENT.U3_MEAS_STA_MEAS_R.ALARMS.PROFILER_INIT_A;
END_REGION

REGION Network 55: UNIT 3 MEASURING STATION FACE A RUN OUT ANALYSIS ALARM
   RUNG wire#powerrail
      { S7_Templates := "SrcType := Int" } EQ_Contact(in1 := "DB16006_U3_MEAS_STA_MEAS_A_CLIENT_INTERFACE".U03_FACE_A_MEAS_Read.Variable.Status, in2 := -1)
      Contact( "DB16006_U3_MEAS_STA_MEAS_A_CLIENT_INTERFACE".U03_FACE_A_MEAS_Read.Variable.RunOutAnalysis )
      wire#w1
      Contact( "DB7258_UNIT_3_STA_MEAS_A_ENABLE_DISABLE".ENABLED )
      wire#w3
      Coil( "DB16000_OPC_UA_TRIGGER_ALARM".CLIENT.U3_MEAS_STA_MEAS_R.ALARMS.RUNOUT_A )
   END_RUNG
   RUNG wire#powerrail
      Contact( "DB16000_OPC_UA_TRIGGER_ALARM".CLIENT.U3_MEAS_STA_MEAS_R.ALARMS.RUNOUT_A )
      I_Contact( "DB2120_MPP_ITC_IPC".RESET_FAULTS )
      wire#w2
      I_Contact( "DB7300_INTERLOCK_GENERAL".GENERAL_MACHINE.FROM_CELL_TO_MACHINE_GENERAL.MEAS_STA_RESET )
   END_RUNG wire#w1
   RUNG wire#w2
      I_Contact( "DB2001_MODES_GENERAL".MG_AUX_OPTIONS.AUX_BOOL[0] )
   END_RUNG wire#w1
   RUNG wire#w3
      Coil( "DB426_ALARMS_WARNINGS".ALARMS.UNIT_03.FACE_R_MEASURING."724245" )
   END_RUNG
   // the same network as SCL:
   "DB16000_OPC_UA_TRIGGER_ALARM".CLIENT.U3_MEAS_STA_MEAS_R.ALARMS.RUNOUT_A := ((("DB16006_U3_MEAS_STA_MEAS_A_CLIENT_INTERFACE".U03_FACE_A_MEAS_Read.Variable.Status = (-1)) AND "DB16006_U3_MEAS_STA_MEAS_A_CLIENT_INTERFACE".U03_FACE_A_MEAS_Read.Variable.RunOutAnalysis) OR ("DB16000_OPC_UA_TRIGGER_ALARM".CLIENT.U3_MEAS_STA_MEAS_R.ALARMS.RUNOUT_A AND NOT "DB2120_MPP_ITC_IPC".RESET_FAULTS AND (NOT "DB7300_INTERLOCK_GENERAL".GENERAL_MACHINE.FROM_CELL_TO_MACHINE_GENERAL.MEAS_STA_RESET OR NOT "DB2001_MODES_GENERAL".MG_AUX_OPTIONS.AUX_BOOL[0]))) AND "DB7258_UNIT_3_STA_MEAS_A_ENABLE_DISABLE".ENABLED;
   "DB426_ALARMS_WARNINGS".ALARMS.UNIT_03.FACE_R_MEASURING."724245" := "DB16000_OPC_UA_TRIGGER_ALARM".CLIENT.U3_MEAS_STA_MEAS_R.ALARMS.RUNOUT_A;
END_REGION

REGION Network 56: UNIT 3 MEASURING STATION FACE A UMBRELLA ANALYSIS ALARM
   RUNG wire#powerrail
      { S7_Templates := "SrcType := Int" } EQ_Contact(in1 := "DB16006_U3_MEAS_STA_MEAS_A_CLIENT_INTERFACE".U03_FACE_A_MEAS_Read.Variable.Status, in2 := -1)
      Contact( "DB16006_U3_MEAS_STA_MEAS_A_CLIENT_INTERFACE".U03_FACE_A_MEAS_Read.Variable.UmbrellaAnalysis )
      wire#w1
      Contact( "DB7258_UNIT_3_STA_MEAS_A_ENABLE_DISABLE".ENABLED )
      wire#w3
      Coil( "DB16000_OPC_UA_TRIGGER_ALARM".CLIENT.U3_MEAS_STA_MEAS_R.ALARMS.UMBRELLA_A )
   END_RUNG
   RUNG wire#powerrail
      Contact( "DB16000_OPC_UA_TRIGGER_ALARM".CLIENT.U3_MEAS_STA_MEAS_R.ALARMS.UMBRELLA_A )
      I_Contact( "DB2120_MPP_ITC_IPC".RESET_FAULTS )
      wire#w2
      I_Contact( "DB7300_INTERLOCK_GENERAL".GENERAL_MACHINE.FROM_CELL_TO_MACHINE_GENERAL.MEAS_STA_RESET )
   END_RUNG wire#w1
   RUNG wire#w2
      I_Contact( "DB2001_MODES_GENERAL".MG_AUX_OPTIONS.AUX_BOOL[0] )
   END_RUNG wire#w1
   RUNG wire#w3
      Coil( "DB426_ALARMS_WARNINGS".ALARMS.UNIT_03.FACE_R_MEASURING."724246" )
   END_RUNG
   // the same network as SCL:
   "DB16000_OPC_UA_TRIGGER_ALARM".CLIENT.U3_MEAS_STA_MEAS_R.ALARMS.UMBRELLA_A := ((("DB16006_U3_MEAS_STA_MEAS_A_CLIENT_INTERFACE".U03_FACE_A_MEAS_Read.Variable.Status = (-1)) AND "DB16006_U3_MEAS_STA_MEAS_A_CLIENT_INTERFACE".U03_FACE_A_MEAS_Read.Variable.UmbrellaAnalysis) OR ("DB16000_OPC_UA_TRIGGER_ALARM".CLIENT.U3_MEAS_STA_MEAS_R.ALARMS.UMBRELLA_A AND NOT "DB2120_MPP_ITC_IPC".RESET_FAULTS AND (NOT "DB7300_INTERLOCK_GENERAL".GENERAL_MACHINE.FROM_CELL_TO_MACHINE_GENERAL.MEAS_STA_RESET OR NOT "DB2001_MODES_GENERAL".MG_AUX_OPTIONS.AUX_BOOL[0]))) AND "DB7258_UNIT_3_STA_MEAS_A_ENABLE_DISABLE".ENABLED;
   "DB426_ALARMS_WARNINGS".ALARMS.UNIT_03.FACE_R_MEASURING."724246" := "DB16000_OPC_UA_TRIGGER_ALARM".CLIENT.U3_MEAS_STA_MEAS_R.ALARMS.UMBRELLA_A;
END_REGION

REGION Network 57: UNIT 3 MEASURING STATION FACE A LAYER GROWTH ANALYSIS ALARM
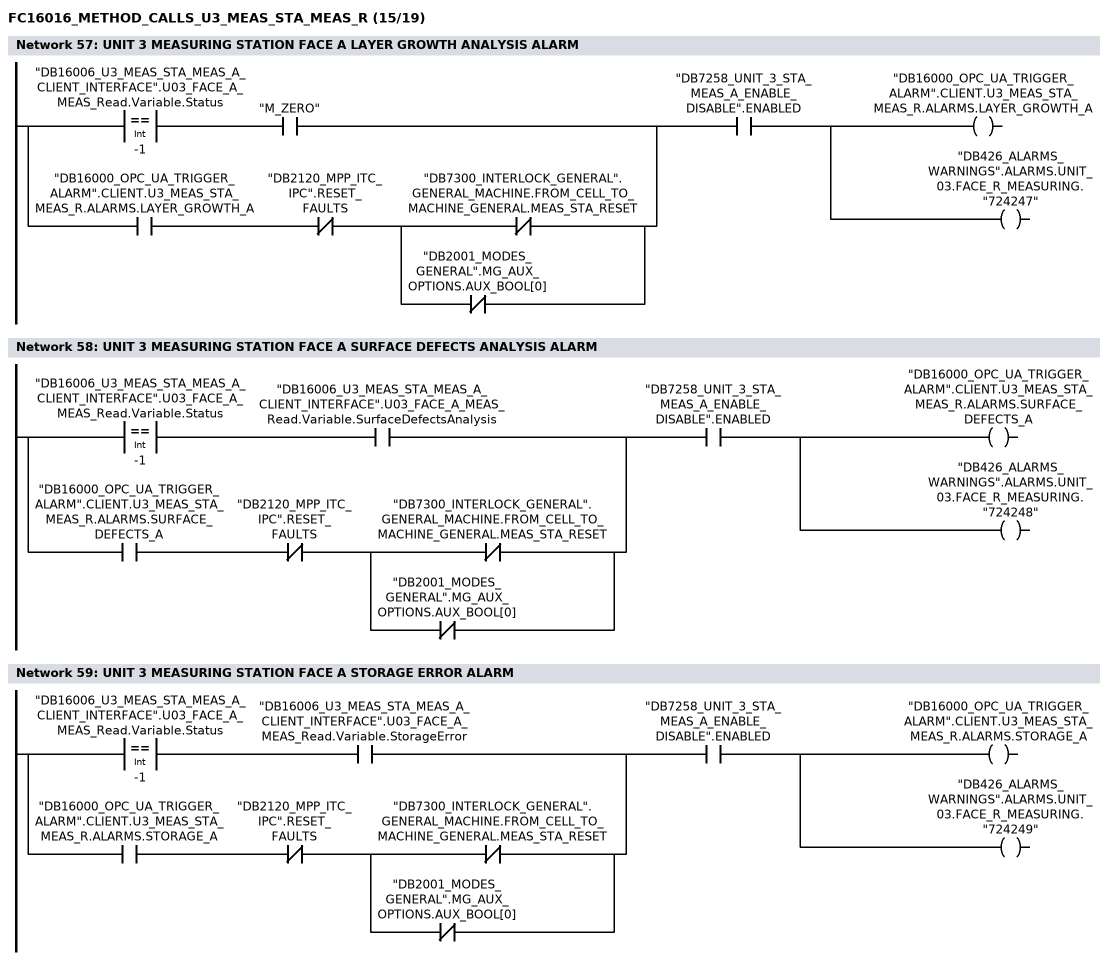
   RUNG wire#powerrail
      { S7_Templates := "SrcType := Int" } EQ_Contact(in1 := "DB16006_U3_MEAS_STA_MEAS_A_CLIENT_INTERFACE".U03_FACE_A_MEAS_Read.Variable.Status, in2 := -1)
      Contact( "M_ZERO" )
      wire#w1
      Contact( "DB7258_UNIT_3_STA_MEAS_A_ENABLE_DISABLE".ENABLED )
      wire#w3
      Coil( "DB16000_OPC_UA_TRIGGER_ALARM".CLIENT.U3_MEAS_STA_MEAS_R.ALARMS.LAYER_GROWTH_A )
   END_RUNG
   RUNG wire#powerrail
      Contact( "DB16000_OPC_UA_TRIGGER_ALARM".CLIENT.U3_MEAS_STA_MEAS_R.ALARMS.LAYER_GROWTH_A )
      I_Contact( "DB2120_MPP_ITC_IPC".RESET_FAULTS )
      wire#w2
      I_Contact( "DB7300_INTERLOCK_GENERAL".GENERAL_MACHINE.FROM_CELL_TO_MACHINE_GENERAL.MEAS_STA_RESET )
   END_RUNG wire#w1
   RUNG wire#w2
      I_Contact( "DB2001_MODES_GENERAL".MG_AUX_OPTIONS.AUX_BOOL[0] )
   END_RUNG wire#w1
   RUNG wire#w3
      Coil( "DB426_ALARMS_WARNINGS".ALARMS.UNIT_03.FACE_R_MEASURING."724247" )
   END_RUNG
   // the same network as SCL:
   "DB16000_OPC_UA_TRIGGER_ALARM".CLIENT.U3_MEAS_STA_MEAS_R.ALARMS.LAYER_GROWTH_A := ((("DB16006_U3_MEAS_STA_MEAS_A_CLIENT_INTERFACE".U03_FACE_A_MEAS_Read.Variable.Status = (-1)) AND "M_ZERO") OR ("DB16000_OPC_UA_TRIGGER_ALARM".CLIENT.U3_MEAS_STA_MEAS_R.ALARMS.LAYER_GROWTH_A AND NOT "DB2120_MPP_ITC_IPC".RESET_FAULTS AND (NOT "DB7300_INTERLOCK_GENERAL".GENERAL_MACHINE.FROM_CELL_TO_MACHINE_GENERAL.MEAS_STA_RESET OR NOT "DB2001_MODES_GENERAL".MG_AUX_OPTIONS.AUX_BOOL[0]))) AND "DB7258_UNIT_3_STA_MEAS_A_ENABLE_DISABLE".ENABLED;
   "DB426_ALARMS_WARNINGS".ALARMS.UNIT_03.FACE_R_MEASURING."724247" := "DB16000_OPC_UA_TRIGGER_ALARM".CLIENT.U3_MEAS_STA_MEAS_R.ALARMS.LAYER_GROWTH_A;
END_REGION

REGION Network 58: UNIT 3 MEASURING STATION FACE A SURFACE DEFECTS ANALYSIS ALARM
   RUNG wire#powerrail
      { S7_Templates := "SrcType := Int" } EQ_Contact(in1 := "DB16006_U3_MEAS_STA_MEAS_A_CLIENT_INTERFACE".U03_FACE_A_MEAS_Read.Variable.Status, in2 := -1)
      Contact( "DB16006_U3_MEAS_STA_MEAS_A_CLIENT_INTERFACE".U03_FACE_A_MEAS_Read.Variable.SurfaceDefectsAnalysis )
      wire#w1
      Contact( "DB7258_UNIT_3_STA_MEAS_A_ENABLE_DISABLE".ENABLED )
      wire#w3
      Coil( "DB16000_OPC_UA_TRIGGER_ALARM".CLIENT.U3_MEAS_STA_MEAS_R.ALARMS.SURFACE_DEFECTS_A )
   END_RUNG
   RUNG wire#powerrail
      Contact( "DB16000_OPC_UA_TRIGGER_ALARM".CLIENT.U3_MEAS_STA_MEAS_R.ALARMS.SURFACE_DEFECTS_A )
      I_Contact( "DB2120_MPP_ITC_IPC".RESET_FAULTS )
      wire#w2
      I_Contact( "DB7300_INTERLOCK_GENERAL".GENERAL_MACHINE.FROM_CELL_TO_MACHINE_GENERAL.MEAS_STA_RESET )
   END_RUNG wire#w1
   RUNG wire#w2
      I_Contact( "DB2001_MODES_GENERAL".MG_AUX_OPTIONS.AUX_BOOL[0] )
   END_RUNG wire#w1
   RUNG wire#w3
      Coil( "DB426_ALARMS_WARNINGS".ALARMS.UNIT_03.FACE_R_MEASURING."724248" )
   END_RUNG
   // the same network as SCL:
   "DB16000_OPC_UA_TRIGGER_ALARM".CLIENT.U3_MEAS_STA_MEAS_R.ALARMS.SURFACE_DEFECTS_A := ((("DB16006_U3_MEAS_STA_MEAS_A_CLIENT_INTERFACE".U03_FACE_A_MEAS_Read.Variable.Status = (-1)) AND "DB16006_U3_MEAS_STA_MEAS_A_CLIENT_INTERFACE".U03_FACE_A_MEAS_Read.Variable.SurfaceDefectsAnalysis) OR ("DB16000_OPC_UA_TRIGGER_ALARM".CLIENT.U3_MEAS_STA_MEAS_R.ALARMS.SURFACE_DEFECTS_A AND NOT "DB2120_MPP_ITC_IPC".RESET_FAULTS AND (NOT "DB7300_INTERLOCK_GENERAL".GENERAL_MACHINE.FROM_CELL_TO_MACHINE_GENERAL.MEAS_STA_RESET OR NOT "DB2001_MODES_GENERAL".MG_AUX_OPTIONS.AUX_BOOL[0]))) AND "DB7258_UNIT_3_STA_MEAS_A_ENABLE_DISABLE".ENABLED;
   "DB426_ALARMS_WARNINGS".ALARMS.UNIT_03.FACE_R_MEASURING."724248" := "DB16000_OPC_UA_TRIGGER_ALARM".CLIENT.U3_MEAS_STA_MEAS_R.ALARMS.SURFACE_DEFECTS_A;
END_REGION

REGION Network 59: UNIT 3 MEASURING STATION FACE A STORAGE ERROR ALARM
   RUNG wire#powerrail
      { S7_Templates := "SrcType := Int" } EQ_Contact(in1 := "DB16006_U3_MEAS_STA_MEAS_A_CLIENT_INTERFACE".U03_FACE_A_MEAS_Read.Variable.Status, in2 := -1)
      Contact( "DB16006_U3_MEAS_STA_MEAS_A_CLIENT_INTERFACE".U03_FACE_A_MEAS_Read.Variable.StorageError )
      wire#w1
      Contact( "DB7258_UNIT_3_STA_MEAS_A_ENABLE_DISABLE".ENABLED )
      wire#w3
      Coil( "DB16000_OPC_UA_TRIGGER_ALARM".CLIENT.U3_MEAS_STA_MEAS_R.ALARMS.STORAGE_A )
   END_RUNG
   RUNG wire#powerrail
      Contact( "DB16000_OPC_UA_TRIGGER_ALARM".CLIENT.U3_MEAS_STA_MEAS_R.ALARMS.STORAGE_A )
      I_Contact( "DB2120_MPP_ITC_IPC".RESET_FAULTS )
      wire#w2
      I_Contact( "DB7300_INTERLOCK_GENERAL".GENERAL_MACHINE.FROM_CELL_TO_MACHINE_GENERAL.MEAS_STA_RESET )
   END_RUNG wire#w1
   RUNG wire#w2
      I_Contact( "DB2001_MODES_GENERAL".MG_AUX_OPTIONS.AUX_BOOL[0] )
   END_RUNG wire#w1
   RUNG wire#w3
      Coil( "DB426_ALARMS_WARNINGS".ALARMS.UNIT_03.FACE_R_MEASURING."724249" )
   END_RUNG
   // the same network as SCL:
   "DB16000_OPC_UA_TRIGGER_ALARM".CLIENT.U3_MEAS_STA_MEAS_R.ALARMS.STORAGE_A := ((("DB16006_U3_MEAS_STA_MEAS_A_CLIENT_INTERFACE".U03_FACE_A_MEAS_Read.Variable.Status = (-1)) AND "DB16006_U3_MEAS_STA_MEAS_A_CLIENT_INTERFACE".U03_FACE_A_MEAS_Read.Variable.StorageError) OR ("DB16000_OPC_UA_TRIGGER_ALARM".CLIENT.U3_MEAS_STA_MEAS_R.ALARMS.STORAGE_A AND NOT "DB2120_MPP_ITC_IPC".RESET_FAULTS AND (NOT "DB7300_INTERLOCK_GENERAL".GENERAL_MACHINE.FROM_CELL_TO_MACHINE_GENERAL.MEAS_STA_RESET OR NOT "DB2001_MODES_GENERAL".MG_AUX_OPTIONS.AUX_BOOL[0]))) AND "DB7258_UNIT_3_STA_MEAS_A_ENABLE_DISABLE".ENABLED;
   "DB426_ALARMS_WARNINGS".ALARMS.UNIT_03.FACE_R_MEASURING."724249" := "DB16000_OPC_UA_TRIGGER_ALARM".CLIENT.U3_MEAS_STA_MEAS_R.ALARMS.STORAGE_A;
END_REGION

REGION Network 60: UNIT 3 MEASURING STATION FACE A MISSING CALIBRATION ALARM
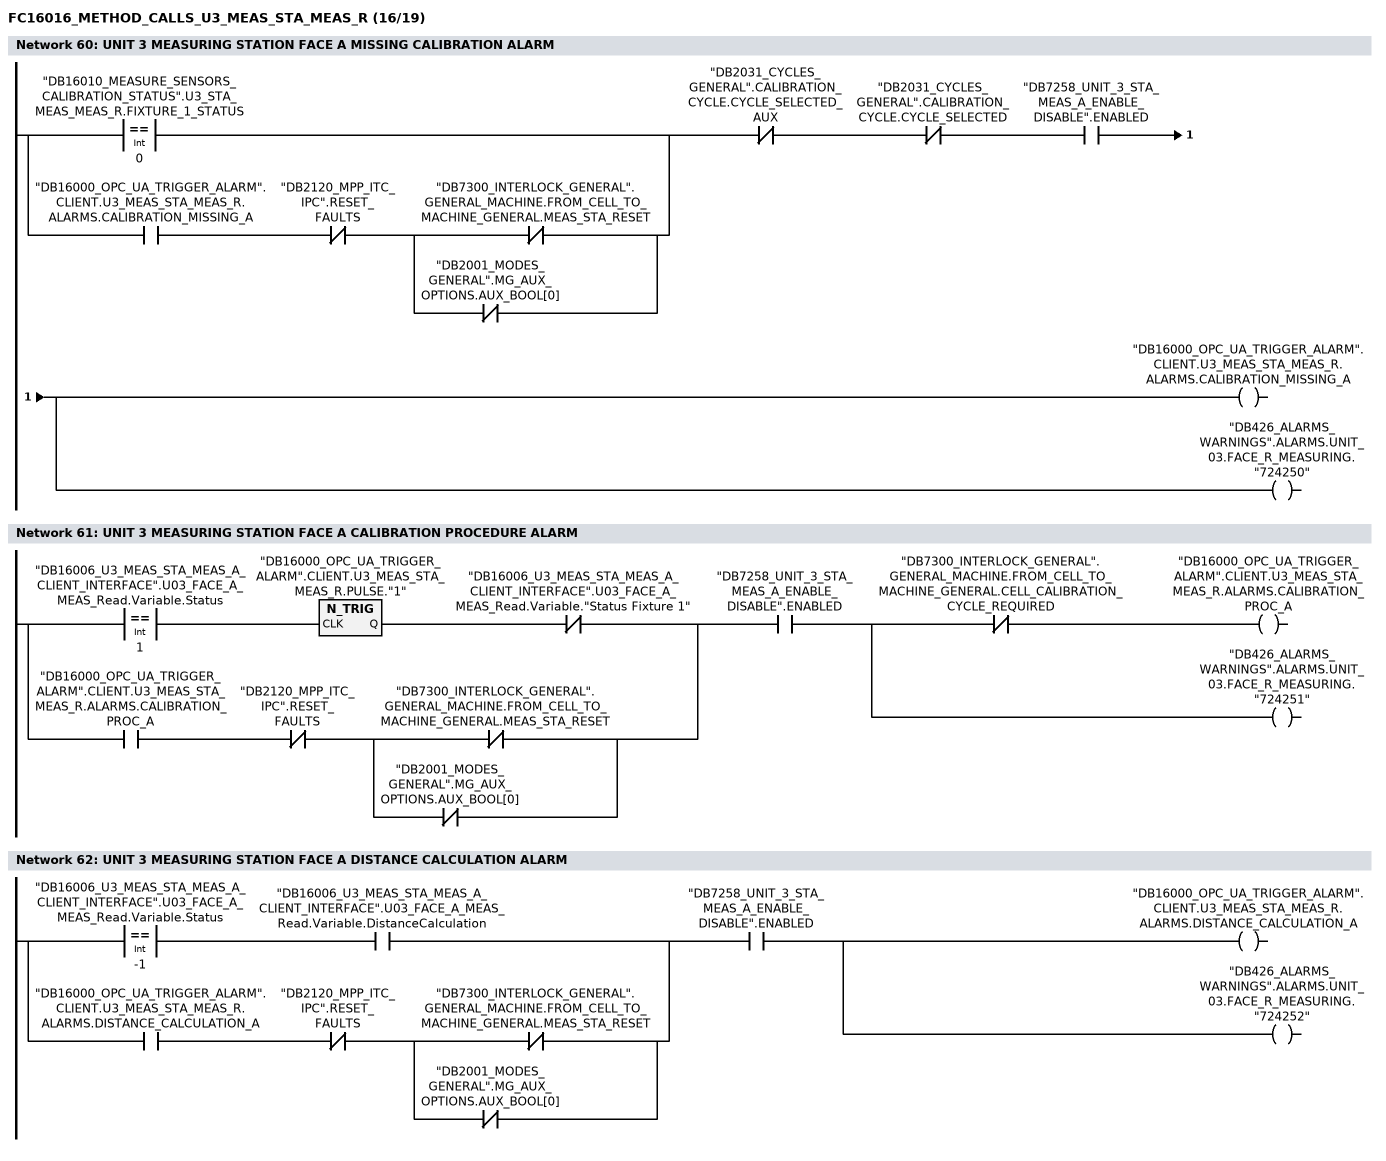
   RUNG wire#powerrail
      { S7_Templates := "SrcType := Int" } EQ_Contact(in1 := "DB16010_MEASURE_SENSORS_CALIBRATION_STATUS".U3_STA_MEAS_MEAS_R.FIXTURE_1_STATUS, in2 := 0)
      wire#w1
      I_Contact( "DB2031_CYCLES_GENERAL".CALIBRATION_CYCLE.CYCLE_SELECTED_AUX )
      I_Contact( "DB2031_CYCLES_GENERAL".CALIBRATION_CYCLE.CYCLE_SELECTED )
      Contact( "DB7258_UNIT_3_STA_MEAS_A_ENABLE_DISABLE".ENABLED )
      wire#w3
      Coil( "DB16000_OPC_UA_TRIGGER_ALARM".CLIENT.U3_MEAS_STA_MEAS_R.ALARMS.CALIBRATION_MISSING_A )
   END_RUNG
   RUNG wire#powerrail
      Contact( "DB16000_OPC_UA_TRIGGER_ALARM".CLIENT.U3_MEAS_STA_MEAS_R.ALARMS.CALIBRATION_MISSING_A )
      I_Contact( "DB2120_MPP_ITC_IPC".RESET_FAULTS )
      wire#w2
      I_Contact( "DB7300_INTERLOCK_GENERAL".GENERAL_MACHINE.FROM_CELL_TO_MACHINE_GENERAL.MEAS_STA_RESET )
   END_RUNG wire#w1
   RUNG wire#w2
      I_Contact( "DB2001_MODES_GENERAL".MG_AUX_OPTIONS.AUX_BOOL[0] )
   END_RUNG wire#w1
   RUNG wire#w3
      Coil( "DB426_ALARMS_WARNINGS".ALARMS.UNIT_03.FACE_R_MEASURING."724250" )
   END_RUNG
   // the same network as SCL:
   "DB16000_OPC_UA_TRIGGER_ALARM".CLIENT.U3_MEAS_STA_MEAS_R.ALARMS.CALIBRATION_MISSING_A := (("DB16010_MEASURE_SENSORS_CALIBRATION_STATUS".U3_STA_MEAS_MEAS_R.FIXTURE_1_STATUS = 0) OR ("DB16000_OPC_UA_TRIGGER_ALARM".CLIENT.U3_MEAS_STA_MEAS_R.ALARMS.CALIBRATION_MISSING_A AND NOT "DB2120_MPP_ITC_IPC".RESET_FAULTS AND (NOT "DB7300_INTERLOCK_GENERAL".GENERAL_MACHINE.FROM_CELL_TO_MACHINE_GENERAL.MEAS_STA_RESET OR NOT "DB2001_MODES_GENERAL".MG_AUX_OPTIONS.AUX_BOOL[0]))) AND NOT "DB2031_CYCLES_GENERAL".CALIBRATION_CYCLE.CYCLE_SELECTED_AUX AND NOT "DB2031_CYCLES_GENERAL".CALIBRATION_CYCLE.CYCLE_SELECTED AND "DB7258_UNIT_3_STA_MEAS_A_ENABLE_DISABLE".ENABLED;
   "DB426_ALARMS_WARNINGS".ALARMS.UNIT_03.FACE_R_MEASURING."724250" := "DB16000_OPC_UA_TRIGGER_ALARM".CLIENT.U3_MEAS_STA_MEAS_R.ALARMS.CALIBRATION_MISSING_A;
END_REGION

REGION Network 61: UNIT 3 MEASURING STATION FACE A CALIBRATION PROCEDURE ALARM
   RUNG wire#powerrail
      { S7_Templates := "SrcType := Int" } EQ_Contact(in1 := "DB16006_U3_MEAS_STA_MEAS_A_CLIENT_INTERFACE".U03_FACE_A_MEAS_Read.Variable.Status, in2 := 1)
      N_Trig( "DB16000_OPC_UA_TRIGGER_ALARM".CLIENT.U3_MEAS_STA_MEAS_R.PULSE."1" )
      I_Contact( "DB16006_U3_MEAS_STA_MEAS_A_CLIENT_INTERFACE".U03_FACE_A_MEAS_Read.Variable."Status Fixture 1" )
      wire#w1
      Contact( "DB7258_UNIT_3_STA_MEAS_A_ENABLE_DISABLE".ENABLED )
      wire#w3
      I_Contact( "DB7300_INTERLOCK_GENERAL".GENERAL_MACHINE.FROM_CELL_TO_MACHINE_GENERAL.CELL_CALIBRATION_CYCLE_REQUIRED )
      Coil( "DB16000_OPC_UA_TRIGGER_ALARM".CLIENT.U3_MEAS_STA_MEAS_R.ALARMS.CALIBRATION_PROC_A )
   END_RUNG
   RUNG wire#powerrail
      Contact( "DB16000_OPC_UA_TRIGGER_ALARM".CLIENT.U3_MEAS_STA_MEAS_R.ALARMS.CALIBRATION_PROC_A )
      I_Contact( "DB2120_MPP_ITC_IPC".RESET_FAULTS )
      wire#w2
      I_Contact( "DB7300_INTERLOCK_GENERAL".GENERAL_MACHINE.FROM_CELL_TO_MACHINE_GENERAL.MEAS_STA_RESET )
   END_RUNG wire#w1
   RUNG wire#w2
      I_Contact( "DB2001_MODES_GENERAL".MG_AUX_OPTIONS.AUX_BOOL[0] )
   END_RUNG wire#w1
   RUNG wire#w3
      Coil( "DB426_ALARMS_WARNINGS".ALARMS.UNIT_03.FACE_R_MEASURING."724251" )
   END_RUNG
   // the same network as SCL:
   #_w1 := "DB16006_U3_MEAS_STA_MEAS_A_CLIENT_INTERFACE".U03_FACE_A_MEAS_Read.Variable.Status = 1;
   #_w2 := NOT #_w1 AND "DB16000_OPC_UA_TRIGGER_ALARM".CLIENT.U3_MEAS_STA_MEAS_R.PULSE."1";   // falling edge
   "DB16000_OPC_UA_TRIGGER_ALARM".CLIENT.U3_MEAS_STA_MEAS_R.PULSE."1" := #_w1;
   #_w3 := ((#_w2 AND NOT "DB16006_U3_MEAS_STA_MEAS_A_CLIENT_INTERFACE".U03_FACE_A_MEAS_Read.Variable."Status Fixture 1") OR ("DB16000_OPC_UA_TRIGGER_ALARM".CLIENT.U3_MEAS_STA_MEAS_R.ALARMS.CALIBRATION_PROC_A AND NOT "DB2120_MPP_ITC_IPC".RESET_FAULTS AND (NOT "DB7300_INTERLOCK_GENERAL".GENERAL_MACHINE.FROM_CELL_TO_MACHINE_GENERAL.MEAS_STA_RESET OR NOT "DB2001_MODES_GENERAL".MG_AUX_OPTIONS.AUX_BOOL[0]))) AND "DB7258_UNIT_3_STA_MEAS_A_ENABLE_DISABLE".ENABLED;
   "DB16000_OPC_UA_TRIGGER_ALARM".CLIENT.U3_MEAS_STA_MEAS_R.ALARMS.CALIBRATION_PROC_A := #_w3 AND NOT "DB7300_INTERLOCK_GENERAL".GENERAL_MACHINE.FROM_CELL_TO_MACHINE_GENERAL.CELL_CALIBRATION_CYCLE_REQUIRED;
   "DB426_ALARMS_WARNINGS".ALARMS.UNIT_03.FACE_R_MEASURING."724251" := #_w3;
END_REGION

REGION Network 62: UNIT 3 MEASURING STATION FACE A DISTANCE CALCULATION ALARM
   RUNG wire#powerrail
      { S7_Templates := "SrcType := Int" } EQ_Contact(in1 := "DB16006_U3_MEAS_STA_MEAS_A_CLIENT_INTERFACE".U03_FACE_A_MEAS_Read.Variable.Status, in2 := -1)
      Contact( "DB16006_U3_MEAS_STA_MEAS_A_CLIENT_INTERFACE".U03_FACE_A_MEAS_Read.Variable.DistanceCalculation )
      wire#w1
      Contact( "DB7258_UNIT_3_STA_MEAS_A_ENABLE_DISABLE".ENABLED )
      wire#w3
      Coil( "DB16000_OPC_UA_TRIGGER_ALARM".CLIENT.U3_MEAS_STA_MEAS_R.ALARMS.DISTANCE_CALCULATION_A )
   END_RUNG
   RUNG wire#powerrail
      Contact( "DB16000_OPC_UA_TRIGGER_ALARM".CLIENT.U3_MEAS_STA_MEAS_R.ALARMS.DISTANCE_CALCULATION_A )
      I_Contact( "DB2120_MPP_ITC_IPC".RESET_FAULTS )
      wire#w2
      I_Contact( "DB7300_INTERLOCK_GENERAL".GENERAL_MACHINE.FROM_CELL_TO_MACHINE_GENERAL.MEAS_STA_RESET )
   END_RUNG wire#w1
   RUNG wire#w2
      I_Contact( "DB2001_MODES_GENERAL".MG_AUX_OPTIONS.AUX_BOOL[0] )
   END_RUNG wire#w1
   RUNG wire#w3
      Coil( "DB426_ALARMS_WARNINGS".ALARMS.UNIT_03.FACE_R_MEASURING."724252" )
   END_RUNG
   // the same network as SCL:
   "DB16000_OPC_UA_TRIGGER_ALARM".CLIENT.U3_MEAS_STA_MEAS_R.ALARMS.DISTANCE_CALCULATION_A := ((("DB16006_U3_MEAS_STA_MEAS_A_CLIENT_INTERFACE".U03_FACE_A_MEAS_Read.Variable.Status = (-1)) AND "DB16006_U3_MEAS_STA_MEAS_A_CLIENT_INTERFACE".U03_FACE_A_MEAS_Read.Variable.DistanceCalculation) OR ("DB16000_OPC_UA_TRIGGER_ALARM".CLIENT.U3_MEAS_STA_MEAS_R.ALARMS.DISTANCE_CALCULATION_A AND NOT "DB2120_MPP_ITC_IPC".RESET_FAULTS AND (NOT "DB7300_INTERLOCK_GENERAL".GENERAL_MACHINE.FROM_CELL_TO_MACHINE_GENERAL.MEAS_STA_RESET OR NOT "DB2001_MODES_GENERAL".MG_AUX_OPTIONS.AUX_BOOL[0]))) AND "DB7258_UNIT_3_STA_MEAS_A_ENABLE_DISABLE".ENABLED;
   "DB426_ALARMS_WARNINGS".ALARMS.UNIT_03.FACE_R_MEASURING."724252" := "DB16000_OPC_UA_TRIGGER_ALARM".CLIENT.U3_MEAS_STA_MEAS_R.ALARMS.DISTANCE_CALCULATION_A;
END_REGION

REGION Network 63: UNIT 3 MEASURING STATION FACE A DATABASE CONNECTION ALARM
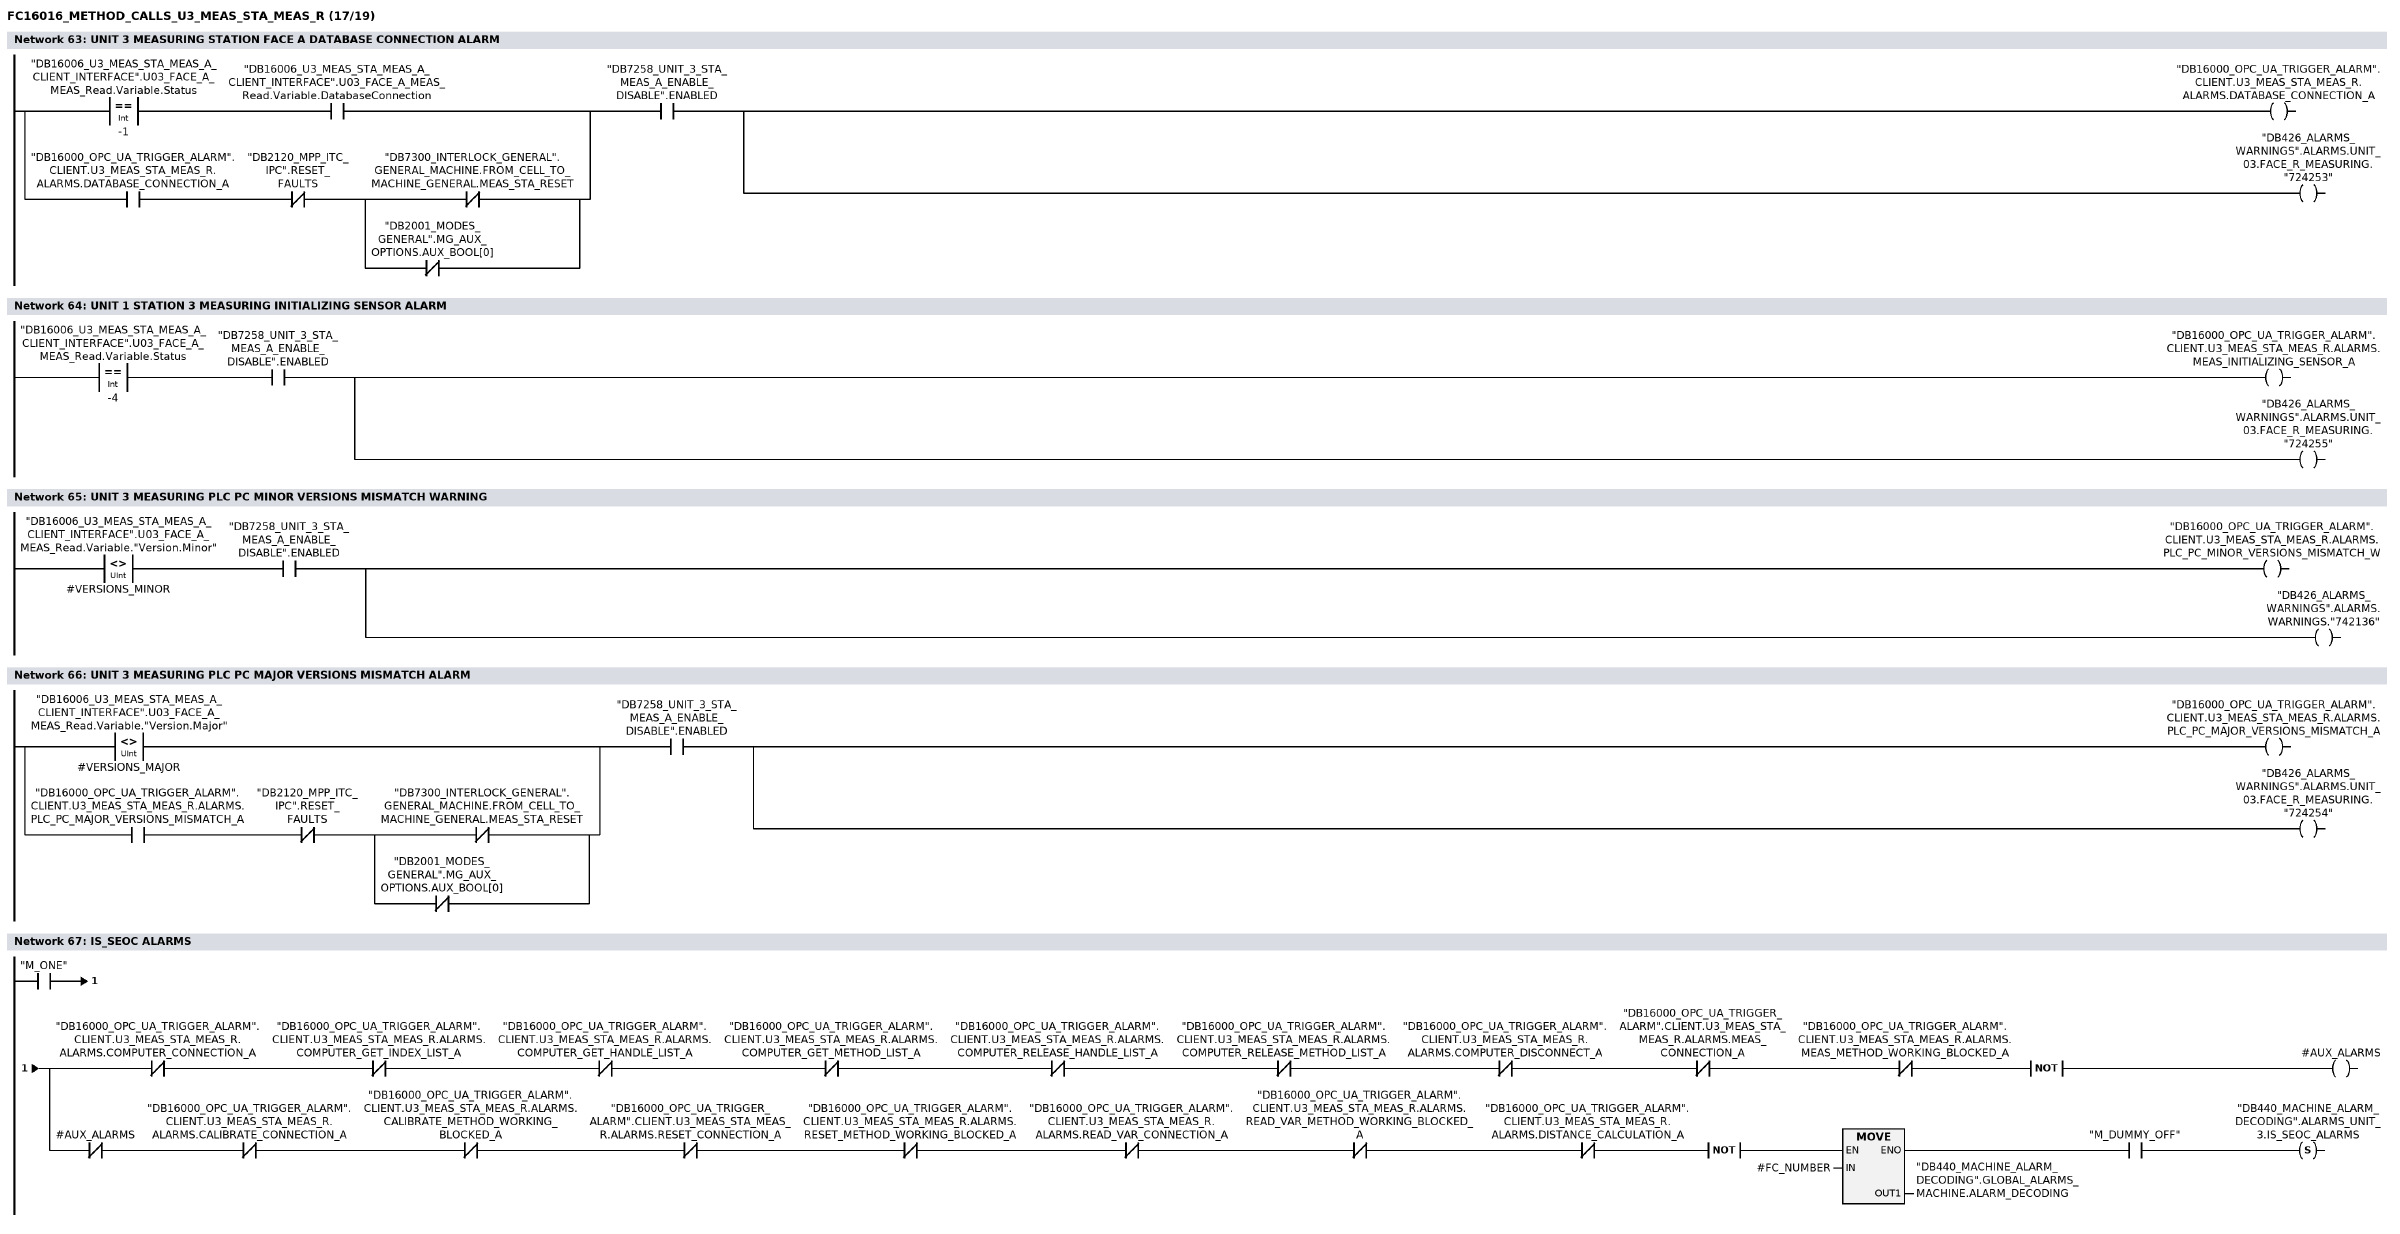
   RUNG wire#powerrail
      { S7_Templates := "SrcType := Int" } EQ_Contact(in1 := "DB16006_U3_MEAS_STA_MEAS_A_CLIENT_INTERFACE".U03_FACE_A_MEAS_Read.Variable.Status, in2 := -1)
      Contact( "DB16006_U3_MEAS_STA_MEAS_A_CLIENT_INTERFACE".U03_FACE_A_MEAS_Read.Variable.DatabaseConnection )
      wire#w1
      Contact( "DB7258_UNIT_3_STA_MEAS_A_ENABLE_DISABLE".ENABLED )
      wire#w3
      Coil( "DB16000_OPC_UA_TRIGGER_ALARM".CLIENT.U3_MEAS_STA_MEAS_R.ALARMS.DATABASE_CONNECTION_A )
   END_RUNG
   RUNG wire#powerrail
      Contact( "DB16000_OPC_UA_TRIGGER_ALARM".CLIENT.U3_MEAS_STA_MEAS_R.ALARMS.DATABASE_CONNECTION_A )
      I_Contact( "DB2120_MPP_ITC_IPC".RESET_FAULTS )
      wire#w2
      I_Contact( "DB7300_INTERLOCK_GENERAL".GENERAL_MACHINE.FROM_CELL_TO_MACHINE_GENERAL.MEAS_STA_RESET )
   END_RUNG wire#w1
   RUNG wire#w2
      I_Contact( "DB2001_MODES_GENERAL".MG_AUX_OPTIONS.AUX_BOOL[0] )
   END_RUNG wire#w1
   RUNG wire#w3
      Coil( "DB426_ALARMS_WARNINGS".ALARMS.UNIT_03.FACE_R_MEASURING."724253" )
   END_RUNG
   // the same network as SCL:
   "DB16000_OPC_UA_TRIGGER_ALARM".CLIENT.U3_MEAS_STA_MEAS_R.ALARMS.DATABASE_CONNECTION_A := ((("DB16006_U3_MEAS_STA_MEAS_A_CLIENT_INTERFACE".U03_FACE_A_MEAS_Read.Variable.Status = (-1)) AND "DB16006_U3_MEAS_STA_MEAS_A_CLIENT_INTERFACE".U03_FACE_A_MEAS_Read.Variable.DatabaseConnection) OR ("DB16000_OPC_UA_TRIGGER_ALARM".CLIENT.U3_MEAS_STA_MEAS_R.ALARMS.DATABASE_CONNECTION_A AND NOT "DB2120_MPP_ITC_IPC".RESET_FAULTS AND (NOT "DB7300_INTERLOCK_GENERAL".GENERAL_MACHINE.FROM_CELL_TO_MACHINE_GENERAL.MEAS_STA_RESET OR NOT "DB2001_MODES_GENERAL".MG_AUX_OPTIONS.AUX_BOOL[0]))) AND "DB7258_UNIT_3_STA_MEAS_A_ENABLE_DISABLE".ENABLED;
   "DB426_ALARMS_WARNINGS".ALARMS.UNIT_03.FACE_R_MEASURING."724253" := "DB16000_OPC_UA_TRIGGER_ALARM".CLIENT.U3_MEAS_STA_MEAS_R.ALARMS.DATABASE_CONNECTION_A;
END_REGION

